(* IEC 61131-3 sources: volt/packages/volt-lsp-iec/test-corpus/pro2193/Device/Plc Logic/Application/04 Physical Interfaces/Ethernet/13 Dashboard, 2 files *)

(* ---- PlcDataType.dut ---- *)
// Complete list of PlcDataTypes for all machines
{attribute 'qualified_only'}
TYPE PlcDataType :
(
	// Last changed (UTC): 17 Dec 2025 13:19
	// Total number of PlcDataTypes: 3778

	Main_RobotStatus := 23,
	Main_EnableIML := 24,
	Main_EnableHMU := 25,
	Main_EnableVision := 26,
	Main_Relays_HighVacuumPumpRunning := 27,
	Main_Relays_LowVacuumPumpRunning := 28,
	Relays_MouldAreaFree := 29,
	Relays_EnableMouldClosure := 30,
	Relays_EnableFullMouldOpening := 31,
	Relays_OperationWithRobot := 32,
	Relays_EnableEjectorBack := 33,
	Relays_EnableEjectorForward := 34,
	Relays_EnableCorePos1Back := 35,
	Relays_EnableCorePos2Forward := 36,
	Relays_GlobalReset := 37,
	Relays_MainAirValve := 38,
	Relays_YUnit_MotorCooling := 39,
	Relays_EnableFrequencyController := 40,
	Relays_SafetyGate := 41,
	YUnit_ActPos := 42,
	YUnit_ErrorId := 43,
	YUnit_AxisErrorId := 44,
	YUnit_DriveErrorId := 45,
	YUnit_DriveUtilisation := 46,
	YUnit_MotorUtilisation := 47,
	XrUnit_ActPos := 48,
	XrUnit_ErrorId := 49,
	XrUnit_AxisErrorId := 50,
	XrUnit_DriveErrorId := 51,
	XrUnit_DriveUtilisation := 52,
	XrUnit_MotorUtilisation := 53,
	XiUnit_ActPos := 54,
	XiUnit_ErrorId := 55,
	XiUnit_AxisErrorId := 56,
	XiUnit_DriveErrorId := 57,
	XiUnit_DriveUtilisation := 58,
	XiUnit_MotorUtilisation := 59,
	XuUnit_ActPos := 60,
	XuUnit_ErrorId := 61,
	XuUnit_AxisErrorId := 62,
	XuUnit_DriveErrorId := 63,
	XuUnit_DriveUtilisation := 64,
	XuUnit_MotorUtilisation := 65,
	Chain_ActPos := 66,
	Chain_ErrorId := 67,
	Chain_AxisErrorId := 68,
	Chain_DriveErrorId := 69,
	Chain_DriveUtilisation := 70,
	Chain_MotorUtilisation := 71,
	Magazine_M1_1_ActPos := 72,
	Magazine_M1_1_ErrorId := 73,
	Magazine_M1_1_AxisErrorId := 74,
	Magazine_M1_1_DriveErrorId := 75,
	Magazine_M1_1_DriveUtilisation := 76,
	Magazine_M1_1_MotorUtilisation := 77,
	Magazine_M1_2_ActPos := 78,
	Magazine_M1_2_ErrorId := 79,
	Magazine_M1_2_AxisErrorId := 80,
	Magazine_M1_2_DriveErrorId := 81,
	Magazine_M1_2_DriveUtilisation := 82,
	Magazine_M1_2_MotorUtilisation := 83,
	ZUnit_ActPos := 84,
	ZUnit_ErrorId := 85,
	ZUnit_AxisErrorId := 86,
	ZUnit_DriveErrorId := 87,
	ZUnit_DriveUtilisation := 88,
	ZUnit_MotorUtilisation := 89,
	YUnit_ActTorque := 90,
	XrUnit_ActTorque := 91,
	XiUnit_ActTorque := 92,
	XuUnit_ActTorque := 93,
	Chain_ActTorque := 94,
	Magazine_M1_1_ActTorque := 95,
	Magazine_M1_2_ActTorque := 96,
	ZUnit_ActTorque := 97,
	YUnit_CoveredDistance := 98,
	XrUnit_CoveredDistance := 99,
	XiUnit_CoveredDistance := 100,
	XuUnit_CoveredDistance := 101,
	Chain_CoveredDistance := 102,
	Magazine_M1_1_CoveredDistance := 103,
	Magazine_M1_2_CoveredDistance := 104,
	ZUnit_CoveredDistance := 105,
	CycleTimes_TimeStopped := 106,
	CycleTimes_TimeResetting := 107,
	CycleTimes_TimeIdle := 108,
	CycleTimes_TimeAutomatic := 109,
	CycleTimes_AutomaticCycleStarts := 110,
	YUnit_Alarms := 111,
	YUnit_Time_Active := 112,
	YUnit_Time_Idle := 113,
	XrUnit_Alarms := 114,
	XrUnit_Time_Active := 115,
	XrUnit_Time_Idle := 116,
	XiUnit_Alarms := 117,
	XiUnit_Time_Active := 118,
	XiUnit_Time_Idle := 119,
	XuUnit_Alarms := 120,
	XuUnit_Time_Active := 121,
	XuUnit_Time_Idle := 122,
	Chain_Alarms := 123,
	Chain_Time_Active := 124,
	Chain_Time_Idle := 125,
	Magazine_M1_1_Alarms := 126,
	Magazine_M1_1_Time_Active := 127,
	Magazine_M1_1_Time_Idle := 128,
	Magazine_M1_2_Alarms := 129,
	Magazine_M1_2_Time_Active := 130,
	Magazine_M1_2_Time_Idle := 131,
	ZUnit_Alarms := 132,
	ZUnit_Time_Active := 133,
	ZUnit_Time_Idle := 134,
	Camera_Alarms := 135,
	Camera_Time_Active := 136,
	Camera_Time_Idle := 137,
	RejectStation_Alarms := 138,
	RejectStation_Time_Active := 139,
	RejectStation_Time_Idle := 140,
	Conveyors_Alarms := 141,
	Conveyors_Time_Active := 142,
	Conveyors_Time_Idle := 143,
	IMM_CycleTimeTakeout := 144,
	IMM_CycleTimeTotal := 145,
	IMM_SavedCycleTimeByEarlyMouldClosing := 146,
	XuUnit_SensorTimes_Vacuum_1 := 147,
	XuUnit_SensorTimes_Vacuum_2 := 148,
	XuUnit_SensorTimes_Vacuum_3 := 149,
	XuUnit_SensorTimes_ShiftIn := 150,
	XuUnit_SensorTimes_ShiftOut := 151,
	Magazine_SensorTimes_Vacuum_1 := 152,
	Magazine_SensorTimes_Vacuum_2 := 153,
	Magazine_SensorTimes_Vacuum_3 := 154,
	Magazine_SensorTimes_Vacuum_4 := 155,
	Magazine_SensorTimes_FlipLabel1In := 156,
	Magazine_SensorTimes_FlipLabel1Out := 157,
	Magazine_SensorTimes_FlipLabel2In := 158,
	Magazine_SensorTimes_FlipLabel2Out := 159,
	Magazine_SensorTimes_ChangeDrawerIn := 160,
	Magazine_SensorTimes_ChangeDrawerOut := 161,
	Magazine_SensorTimes_LockDrawerIn := 162,
	Magazine_SensorTimes_LockDrawerOut := 163,
	ZUnit_SensorTimes_Vacuum_1 := 164,
	ZUnit_SensorTimes_Vacuum_2 := 165,
	ZUnit_SensorTimes_Vacuum_3 := 166,
	ZUnit_SensorTimes_Vacuum_4 := 167,
	ZUnit_SensorTimes_RotateIn := 168,
	ZUnit_SensorTimes_RotateOut := 169,
	ZUnit_SensorTimes_Extend1In := 170,
	ZUnit_SensorTimes_Extend2In := 171,
	ZUnit_SensorTimes_Extend3In := 172,
	ZUnit_SensorTimes_Extend4In := 173,
	RejectStation_SensorTimes_RejectCylinderIn := 174,
	RejectStation_SensorTimes_RejectCylinderOut := 175,
	MetaData_RejectReason_0_Description := 176,
	MetaData_RejectReason_1_Description := 177,
	MetaData_RejectReason_2_Description := 178,
	MetaData_RejectReason_3_Description := 179,
	MetaData_RejectReason_4_Description := 180,
	MetaData_RejectReason_5_Description := 181,
	MetaData_RejectReason_6_Description := 182,
	Productioncounters_Total_Produced := 183,
	Productioncounters_Total_Stacked := 184,
	Productioncounters_Total_Rejected := 185,
	Productioncounters_Total_UncountedReject := 186,
	Productioncounters_Total_RejectReason_0 := 187,
	Productioncounters_Total_RejectReason_1 := 188,
	Productioncounters_Total_RejectReason_2 := 189,
	Productioncounters_Total_RejectReason_3 := 190,
	Productioncounters_Total_RejectReason_4 := 191,
	Productioncounters_Total_RejectReason_5 := 192,
	Productioncounters_Total_RejectReason_6 := 193,
	Productioncounters_Cavity_1_Produced := 194,
	Productioncounters_Cavity_1_Stacked := 195,
	Productioncounters_Cavity_1_Rejected := 196,
	Productioncounters_Cavity_1_UncountedReject := 197,
	Productioncounters_Cavity_1_RejectReason_0 := 198,
	Productioncounters_Cavity_1_RejectReason_1 := 199,
	Productioncounters_Cavity_1_RejectReason_2 := 200,
	Productioncounters_Cavity_1_RejectReason_3 := 201,
	Productioncounters_Cavity_1_RejectReason_4 := 202,
	Productioncounters_Cavity_1_RejectReason_5 := 203,
	Productioncounters_Cavity_1_RejectReason_6 := 204,
	Productioncounters_Cavity_2_Produced := 205,
	Productioncounters_Cavity_2_Stacked := 206,
	Productioncounters_Cavity_2_Rejected := 207,
	Productioncounters_Cavity_2_UncountedReject := 208,
	Productioncounters_Cavity_2_RejectReason_0 := 209,
	Productioncounters_Cavity_2_RejectReason_1 := 210,
	Productioncounters_Cavity_2_RejectReason_2 := 211,
	Productioncounters_Cavity_2_RejectReason_3 := 212,
	Productioncounters_Cavity_2_RejectReason_4 := 213,
	Productioncounters_Cavity_2_RejectReason_5 := 214,
	Productioncounters_Cavity_2_RejectReason_6 := 215,
	Productioncounters_Cavity_3_Produced := 216,
	Productioncounters_Cavity_3_Stacked := 217,
	Productioncounters_Cavity_3_Rejected := 218,
	Productioncounters_Cavity_3_UncountedReject := 219,
	Productioncounters_Cavity_3_RejectReason_0 := 220,
	Productioncounters_Cavity_3_RejectReason_1 := 221,
	Productioncounters_Cavity_3_RejectReason_2 := 222,
	Productioncounters_Cavity_3_RejectReason_3 := 223,
	Productioncounters_Cavity_3_RejectReason_4 := 224,
	Productioncounters_Cavity_3_RejectReason_5 := 225,
	Productioncounters_Cavity_3_RejectReason_6 := 226,
	Productioncounters_Cavity_4_Produced := 227,
	Productioncounters_Cavity_4_Stacked := 228,
	Productioncounters_Cavity_4_Rejected := 229,
	Productioncounters_Cavity_4_UncountedReject := 230,
	Productioncounters_Cavity_4_RejectReason_0 := 231,
	Productioncounters_Cavity_4_RejectReason_1 := 232,
	Productioncounters_Cavity_4_RejectReason_2 := 233,
	Productioncounters_Cavity_4_RejectReason_3 := 234,
	Productioncounters_Cavity_4_RejectReason_4 := 235,
	Productioncounters_Cavity_4_RejectReason_5 := 236,
	Productioncounters_Cavity_4_RejectReason_6 := 237,
	Productioncounters_Cavity_5_Produced := 238,
	Productioncounters_Cavity_5_Stacked := 239,
	Productioncounters_Cavity_5_Rejected := 240,
	Productioncounters_Cavity_5_UncountedReject := 241,
	Productioncounters_Cavity_5_RejectReason_0 := 242,
	Productioncounters_Cavity_5_RejectReason_1 := 243,
	Productioncounters_Cavity_5_RejectReason_2 := 244,
	Productioncounters_Cavity_5_RejectReason_3 := 245,
	Productioncounters_Cavity_5_RejectReason_4 := 246,
	Productioncounters_Cavity_5_RejectReason_5 := 247,
	Productioncounters_Cavity_5_RejectReason_6 := 248,
	Productioncounters_Cavity_6_Produced := 249,
	Productioncounters_Cavity_6_Stacked := 250,
	Productioncounters_Cavity_6_Rejected := 251,
	Productioncounters_Cavity_6_UncountedReject := 252,
	Productioncounters_Cavity_6_RejectReason_0 := 253,
	Productioncounters_Cavity_6_RejectReason_1 := 254,
	Productioncounters_Cavity_6_RejectReason_2 := 255,
	Productioncounters_Cavity_6_RejectReason_3 := 256,
	Productioncounters_Cavity_6_RejectReason_4 := 257,
	Productioncounters_Cavity_6_RejectReason_5 := 258,
	Productioncounters_Cavity_6_RejectReason_6 := 259,
	Main_RecipeName := 260,
	Main_RecipeName_Cassette := 261,
	Main_ParameterChanged := 262,
	Main_AirPressureOk := 263,
	Main_GeneralAlarmActive := 264,
	Main_GeneralWarningActive := 265,
	Main_Alarms := 266,
	Main_AlarmsFuse := 267,
	Main_AlarmsIMM := 268,
	Main_Messages := 269,
	Main_Warnings := 270,
	Magazine_Alarms := 273,
	YUnit_AlarmsMotionControl := 274,
	Main_SafetyPLCStatus1 := 275,
	Main_SafetyPLCStatus2 := 276,
	Main_SafetyPLCStatus3 := 277,
	RobotConnected := 278,
	ZUnit_SensorTimes_Shift1In := 279,
	ZUnit_SensorTimes_Shift1Out := 280,
	Main_SER_State := 281,
	Main_SER_OperationMode := 282,
	Main_RecipeName_Brink := 283,
	RejectStation_SensorTimes_RejectCylinder2In := 284,
	RejectStation_SensorTimes_RejectCylinder2Out := 285,
	XuUnit_SensorTimes_ShiftHorizontalIn := 286,
	XuUnit_SensorTimes_ShiftHorizontalOut := 287,
	XuUnit_SensorTimes_ShiftVerticalIn := 288,
	XuUnit_SensorTimes_ShiftVerticalOut := 289,
	MetaData_RejectReason_7_Description := 290,
	Productioncounters_Total_RejectReason_7 := 291,
	Productioncounters_Cavity_1_RejectReason_7 := 292,
	Productioncounters_Cavity_2_RejectReason_7 := 293,
	Productioncounters_Cavity_3_RejectReason_7 := 294,
	Productioncounters_Cavity_4_RejectReason_7 := 295,
	Productioncounters_Cavity_5_RejectReason_7 := 296,
	Productioncounters_Cavity_6_RejectReason_7 := 297,
	MouldMeasurement_MaxPressure := 298,
	MouldMeasurement_MinPressure := 299,
	MouldMeasurement_IdealPressure := 300,
	MouldMeasurement_AveragePressure := 301,
	MouldMeasurement_CalculatedIdealPressure := 302,
	MouldMeasurement_HoldingPressure_TargetValue := 303,
	MouldMeasurement_HoldingPressure_ActualValue := 304,
	MouldMeasurement_SwitchOverPoint_TargetValue := 305,
	MouldMeasurement_SwitchOverPoint_ActualValue := 306,
	MouldMeasurement_Cavity_1_PeakPressure := 307,
	MouldMeasurement_Cavity_2_PeakPressure := 308,
	MouldMeasurement_Cavity_3_PeakPressure := 309,
	MouldMeasurement_Cavity_4_PeakPressure := 310,
	MouldMeasurement_Cavity_5_PeakPressure := 311,
	MouldMeasurement_Cavity_6_PeakPressure := 312,
	MouldMeasurement_Hotrunner_Cavity_1_TargetValue := 313,
	MouldMeasurement_Hotrunner_Cavity_1_ActualValue := 314,
	MouldMeasurement_Hotrunner_Cavity_2_TargetValue := 315,
	MouldMeasurement_Hotrunner_Cavity_2_ActualValue := 316,
	MouldMeasurement_Hotrunner_Cavity_3_TargetValue := 317,
	MouldMeasurement_Hotrunner_Cavity_3_ActualValue := 318,
	MouldMeasurement_Hotrunner_Cavity_4_TargetValue := 319,
	MouldMeasurement_Hotrunner_Cavity_4_ActualValue := 320,
	MouldMeasurement_Hotrunner_Cavity_5_TargetValue := 321,
	MouldMeasurement_Hotrunner_Cavity_5_ActualValue := 322,
	MouldMeasurement_Hotrunner_Cavity_6_TargetValue := 323,
	MouldMeasurement_Hotrunner_Cavity_6_ActualValue := 324,
	MetaData_RejectReason_8_Description := 325,
	Productioncounters_Total_RejectReason_8 := 326,
	Productioncounters_Cavity_1_RejectReason_8 := 327,
	Productioncounters_Cavity_2_RejectReason_8 := 328,
	Productioncounters_Cavity_3_RejectReason_8 := 329,
	Productioncounters_Cavity_4_RejectReason_8 := 330,
	Productioncounters_Cavity_5_RejectReason_8 := 331,
	Productioncounters_Cavity_6_RejectReason_8 := 332,
	MetaData_RejectReason_9_Description := 333,
	Productioncounters_Total_RejectReason_9 := 334,
	Productioncounters_Cavity_1_RejectReason_9 := 335,
	Productioncounters_Cavity_2_RejectReason_9 := 336,
	Productioncounters_Cavity_3_RejectReason_9 := 337,
	Productioncounters_Cavity_4_RejectReason_9 := 338,
	Productioncounters_Cavity_5_RejectReason_9 := 339,
	Productioncounters_Cavity_6_RejectReason_9 := 340,
	MetaData_RejectReason_10_Description := 341,
	Productioncounters_Total_RejectReason_10 := 342,
	Productioncounters_Cavity_1_RejectReason_10 := 343,
	Productioncounters_Cavity_2_RejectReason_10 := 344,
	Productioncounters_Cavity_3_RejectReason_10 := 345,
	Productioncounters_Cavity_4_RejectReason_10 := 346,
	Productioncounters_Cavity_5_RejectReason_10 := 347,
	Productioncounters_Cavity_6_RejectReason_10 := 348,
	MetaData_RejectReason_11_Description := 349,
	Productioncounters_Total_RejectReason_11 := 350,
	Productioncounters_Cavity_1_RejectReason_11 := 351,
	Productioncounters_Cavity_2_RejectReason_11 := 352,
	Productioncounters_Cavity_3_RejectReason_11 := 353,
	Productioncounters_Cavity_4_RejectReason_11 := 354,
	Productioncounters_Cavity_5_RejectReason_11 := 355,
	Productioncounters_Cavity_6_RejectReason_11 := 356,
	MetaData_RejectReason_12_Description := 357,
	Productioncounters_Total_RejectReason_12 := 358,
	Productioncounters_Cavity_1_RejectReason_12 := 359,
	Productioncounters_Cavity_2_RejectReason_12 := 360,
	Productioncounters_Cavity_3_RejectReason_12 := 361,
	Productioncounters_Cavity_4_RejectReason_12 := 362,
	Productioncounters_Cavity_5_RejectReason_12 := 363,
	Productioncounters_Cavity_6_RejectReason_12 := 364,
	MetaData_RejectReason_13_Description := 365,
	Productioncounters_Total_RejectReason_13 := 366,
	Productioncounters_Cavity_1_RejectReason_13 := 367,
	Productioncounters_Cavity_2_RejectReason_13 := 368,
	Productioncounters_Cavity_3_RejectReason_13 := 369,
	Productioncounters_Cavity_4_RejectReason_13 := 370,
	Productioncounters_Cavity_5_RejectReason_13 := 371,
	Productioncounters_Cavity_6_RejectReason_13 := 372,
	MetaData_RejectReason_14_Description := 373,
	Productioncounters_Total_RejectReason_14 := 374,
	Productioncounters_Cavity_1_RejectReason_14 := 375,
	Productioncounters_Cavity_2_RejectReason_14 := 376,
	Productioncounters_Cavity_3_RejectReason_14 := 377,
	Productioncounters_Cavity_4_RejectReason_14 := 378,
	Productioncounters_Cavity_5_RejectReason_14 := 379,
	Productioncounters_Cavity_6_RejectReason_14 := 380,
	MetaData_RejectReason_15_Description := 381,
	Productioncounters_Total_RejectReason_15 := 382,
	Productioncounters_Cavity_1_RejectReason_15 := 383,
	Productioncounters_Cavity_2_RejectReason_15 := 384,
	Productioncounters_Cavity_3_RejectReason_15 := 385,
	Productioncounters_Cavity_4_RejectReason_15 := 386,
	Productioncounters_Cavity_5_RejectReason_15 := 387,
	Productioncounters_Cavity_6_RejectReason_15 := 388,
	MetaData_RejectReason_16_Description := 389,
	Productioncounters_Total_RejectReason_16 := 390,
	Productioncounters_Cavity_1_RejectReason_16 := 391,
	Productioncounters_Cavity_2_RejectReason_16 := 392,
	Productioncounters_Cavity_3_RejectReason_16 := 393,
	Productioncounters_Cavity_4_RejectReason_16 := 394,
	Productioncounters_Cavity_5_RejectReason_16 := 395,
	Productioncounters_Cavity_6_RejectReason_16 := 396,
	MetaData_RejectReason_17_Description := 397,
	Productioncounters_Total_RejectReason_17 := 398,
	Productioncounters_Cavity_1_RejectReason_17 := 399,
	Productioncounters_Cavity_2_RejectReason_17 := 400,
	Productioncounters_Cavity_3_RejectReason_17 := 401,
	Productioncounters_Cavity_4_RejectReason_17 := 402,
	Productioncounters_Cavity_5_RejectReason_17 := 403,
	Productioncounters_Cavity_6_RejectReason_17 := 404,
	MetaData_RejectReason_18_Description := 405,
	Productioncounters_Total_RejectReason_18 := 406,
	Productioncounters_Cavity_1_RejectReason_18 := 407,
	Productioncounters_Cavity_2_RejectReason_18 := 408,
	Productioncounters_Cavity_3_RejectReason_18 := 409,
	Productioncounters_Cavity_4_RejectReason_18 := 410,
	Productioncounters_Cavity_5_RejectReason_18 := 411,
	Productioncounters_Cavity_6_RejectReason_18 := 412,
	MetaData_RejectReason_19_Description := 413,
	Productioncounters_Total_RejectReason_19 := 414,
	Productioncounters_Cavity_1_RejectReason_19 := 415,
	Productioncounters_Cavity_2_RejectReason_19 := 416,
	Productioncounters_Cavity_3_RejectReason_19 := 417,
	Productioncounters_Cavity_4_RejectReason_19 := 418,
	Productioncounters_Cavity_5_RejectReason_19 := 419,
	Productioncounters_Cavity_6_RejectReason_19 := 420,
	MetaData_RejectReason_20_Description := 421,
	Productioncounters_Total_RejectReason_20 := 422,
	Productioncounters_Cavity_1_RejectReason_20 := 423,
	Productioncounters_Cavity_2_RejectReason_20 := 424,
	Productioncounters_Cavity_3_RejectReason_20 := 425,
	Productioncounters_Cavity_4_RejectReason_20 := 426,
	Productioncounters_Cavity_5_RejectReason_20 := 427,
	Productioncounters_Cavity_6_RejectReason_20 := 428,
	Productioncounters_Cavity_7_Produced := 429,
	Productioncounters_Cavity_7_Stacked := 430,
	Productioncounters_Cavity_7_Rejected := 431,
	Productioncounters_Cavity_7_UncountedReject := 432,
	Productioncounters_Cavity_7_RejectReason_0 := 433,
	Productioncounters_Cavity_7_RejectReason_1 := 434,
	Productioncounters_Cavity_7_RejectReason_2 := 435,
	Productioncounters_Cavity_7_RejectReason_3 := 436,
	Productioncounters_Cavity_7_RejectReason_4 := 437,
	Productioncounters_Cavity_7_RejectReason_5 := 438,
	Productioncounters_Cavity_7_RejectReason_6 := 439,
	Productioncounters_Cavity_7_RejectReason_7 := 440,
	Productioncounters_Cavity_7_RejectReason_8 := 441,
	Productioncounters_Cavity_7_RejectReason_9 := 442,
	Productioncounters_Cavity_7_RejectReason_10 := 443,
	Productioncounters_Cavity_7_RejectReason_11 := 444,
	Productioncounters_Cavity_7_RejectReason_12 := 445,
	Productioncounters_Cavity_7_RejectReason_13 := 446,
	Productioncounters_Cavity_7_RejectReason_14 := 447,
	Productioncounters_Cavity_7_RejectReason_15 := 448,
	Productioncounters_Cavity_7_RejectReason_16 := 449,
	Productioncounters_Cavity_7_RejectReason_17 := 450,
	Productioncounters_Cavity_7_RejectReason_18 := 451,
	Productioncounters_Cavity_7_RejectReason_19 := 452,
	Productioncounters_Cavity_7_RejectReason_20 := 453,
	MouldMeasurement_Cavity_7_PeakPressure := 454,
	MouldMeasurement_Hotrunner_Cavity_7_TargetValue := 455,
	MouldMeasurement_Hotrunner_Cavity_7_ActualValue := 456,
	Productioncounters_Cavity_8_Produced := 457,
	Productioncounters_Cavity_8_Stacked := 458,
	Productioncounters_Cavity_8_Rejected := 459,
	Productioncounters_Cavity_8_UncountedReject := 460,
	Productioncounters_Cavity_8_RejectReason_0 := 461,
	Productioncounters_Cavity_8_RejectReason_1 := 462,
	Productioncounters_Cavity_8_RejectReason_2 := 463,
	Productioncounters_Cavity_8_RejectReason_3 := 464,
	Productioncounters_Cavity_8_RejectReason_4 := 465,
	Productioncounters_Cavity_8_RejectReason_5 := 466,
	Productioncounters_Cavity_8_RejectReason_6 := 467,
	Productioncounters_Cavity_8_RejectReason_7 := 468,
	Productioncounters_Cavity_8_RejectReason_8 := 469,
	Productioncounters_Cavity_8_RejectReason_9 := 470,
	Productioncounters_Cavity_8_RejectReason_10 := 471,
	Productioncounters_Cavity_8_RejectReason_11 := 472,
	Productioncounters_Cavity_8_RejectReason_12 := 473,
	Productioncounters_Cavity_8_RejectReason_13 := 474,
	Productioncounters_Cavity_8_RejectReason_14 := 475,
	Productioncounters_Cavity_8_RejectReason_15 := 476,
	Productioncounters_Cavity_8_RejectReason_16 := 477,
	Productioncounters_Cavity_8_RejectReason_17 := 478,
	Productioncounters_Cavity_8_RejectReason_18 := 479,
	Productioncounters_Cavity_8_RejectReason_19 := 480,
	Productioncounters_Cavity_8_RejectReason_20 := 481,
	MouldMeasurement_Cavity_8_PeakPressure := 482,
	MouldMeasurement_Hotrunner_Cavity_8_TargetValue := 483,
	MouldMeasurement_Hotrunner_Cavity_8_ActualValue := 484,
	Productioncounters_Cavity_9_Produced := 485,
	Productioncounters_Cavity_9_Stacked := 486,
	Productioncounters_Cavity_9_Rejected := 487,
	Productioncounters_Cavity_9_UncountedReject := 488,
	Productioncounters_Cavity_9_RejectReason_0 := 489,
	Productioncounters_Cavity_9_RejectReason_1 := 490,
	Productioncounters_Cavity_9_RejectReason_2 := 491,
	Productioncounters_Cavity_9_RejectReason_3 := 492,
	Productioncounters_Cavity_9_RejectReason_4 := 493,
	Productioncounters_Cavity_9_RejectReason_5 := 494,
	Productioncounters_Cavity_9_RejectReason_6 := 495,
	Productioncounters_Cavity_9_RejectReason_7 := 496,
	Productioncounters_Cavity_9_RejectReason_8 := 497,
	Productioncounters_Cavity_9_RejectReason_9 := 498,
	Productioncounters_Cavity_9_RejectReason_10 := 499,
	Productioncounters_Cavity_9_RejectReason_11 := 500,
	Productioncounters_Cavity_9_RejectReason_12 := 501,
	Productioncounters_Cavity_9_RejectReason_13 := 502,
	Productioncounters_Cavity_9_RejectReason_14 := 503,
	Productioncounters_Cavity_9_RejectReason_15 := 504,
	Productioncounters_Cavity_9_RejectReason_16 := 505,
	Productioncounters_Cavity_9_RejectReason_17 := 506,
	Productioncounters_Cavity_9_RejectReason_18 := 507,
	Productioncounters_Cavity_9_RejectReason_19 := 508,
	Productioncounters_Cavity_9_RejectReason_20 := 509,
	MouldMeasurement_Cavity_9_PeakPressure := 510,
	MouldMeasurement_Hotrunner_Cavity_9_TargetValue := 511,
	MouldMeasurement_Hotrunner_Cavity_9_ActualValue := 512,
	Productioncounters_Cavity_10_Produced := 513,
	Productioncounters_Cavity_10_Stacked := 514,
	Productioncounters_Cavity_10_Rejected := 515,
	Productioncounters_Cavity_10_UncountedReject := 516,
	Productioncounters_Cavity_10_RejectReason_0 := 517,
	Productioncounters_Cavity_10_RejectReason_1 := 518,
	Productioncounters_Cavity_10_RejectReason_2 := 519,
	Productioncounters_Cavity_10_RejectReason_3 := 520,
	Productioncounters_Cavity_10_RejectReason_4 := 521,
	Productioncounters_Cavity_10_RejectReason_5 := 522,
	Productioncounters_Cavity_10_RejectReason_6 := 523,
	Productioncounters_Cavity_10_RejectReason_7 := 524,
	Productioncounters_Cavity_10_RejectReason_8 := 525,
	Productioncounters_Cavity_10_RejectReason_9 := 526,
	Productioncounters_Cavity_10_RejectReason_10 := 527,
	Productioncounters_Cavity_10_RejectReason_11 := 528,
	Productioncounters_Cavity_10_RejectReason_12 := 529,
	Productioncounters_Cavity_10_RejectReason_13 := 530,
	Productioncounters_Cavity_10_RejectReason_14 := 531,
	Productioncounters_Cavity_10_RejectReason_15 := 532,
	Productioncounters_Cavity_10_RejectReason_16 := 533,
	Productioncounters_Cavity_10_RejectReason_17 := 534,
	Productioncounters_Cavity_10_RejectReason_18 := 535,
	Productioncounters_Cavity_10_RejectReason_19 := 536,
	Productioncounters_Cavity_10_RejectReason_20 := 537,
	MouldMeasurement_Cavity_10_PeakPressure := 538,
	MouldMeasurement_Hotrunner_Cavity_10_TargetValue := 539,
	MouldMeasurement_Hotrunner_Cavity_10_ActualValue := 540,
	Productioncounters_Cavity_11_Produced := 541,
	Productioncounters_Cavity_11_Stacked := 542,
	Productioncounters_Cavity_11_Rejected := 543,
	Productioncounters_Cavity_11_UncountedReject := 544,
	Productioncounters_Cavity_11_RejectReason_0 := 545,
	Productioncounters_Cavity_11_RejectReason_1 := 546,
	Productioncounters_Cavity_11_RejectReason_2 := 547,
	Productioncounters_Cavity_11_RejectReason_3 := 548,
	Productioncounters_Cavity_11_RejectReason_4 := 549,
	Productioncounters_Cavity_11_RejectReason_5 := 550,
	Productioncounters_Cavity_11_RejectReason_6 := 551,
	Productioncounters_Cavity_11_RejectReason_7 := 552,
	Productioncounters_Cavity_11_RejectReason_8 := 553,
	Productioncounters_Cavity_11_RejectReason_9 := 554,
	Productioncounters_Cavity_11_RejectReason_10 := 555,
	Productioncounters_Cavity_11_RejectReason_11 := 556,
	Productioncounters_Cavity_11_RejectReason_12 := 557,
	Productioncounters_Cavity_11_RejectReason_13 := 558,
	Productioncounters_Cavity_11_RejectReason_14 := 559,
	Productioncounters_Cavity_11_RejectReason_15 := 560,
	Productioncounters_Cavity_11_RejectReason_16 := 561,
	Productioncounters_Cavity_11_RejectReason_17 := 562,
	Productioncounters_Cavity_11_RejectReason_18 := 563,
	Productioncounters_Cavity_11_RejectReason_19 := 564,
	Productioncounters_Cavity_11_RejectReason_20 := 565,
	MouldMeasurement_Cavity_11_PeakPressure := 566,
	MouldMeasurement_Hotrunner_Cavity_11_TargetValue := 567,
	MouldMeasurement_Hotrunner_Cavity_11_ActualValue := 568,
	Productioncounters_Cavity_12_Produced := 569,
	Productioncounters_Cavity_12_Stacked := 570,
	Productioncounters_Cavity_12_Rejected := 571,
	Productioncounters_Cavity_12_UncountedReject := 572,
	Productioncounters_Cavity_12_RejectReason_0 := 573,
	Productioncounters_Cavity_12_RejectReason_1 := 574,
	Productioncounters_Cavity_12_RejectReason_2 := 575,
	Productioncounters_Cavity_12_RejectReason_3 := 576,
	Productioncounters_Cavity_12_RejectReason_4 := 577,
	Productioncounters_Cavity_12_RejectReason_5 := 578,
	Productioncounters_Cavity_12_RejectReason_6 := 579,
	Productioncounters_Cavity_12_RejectReason_7 := 580,
	Productioncounters_Cavity_12_RejectReason_8 := 581,
	Productioncounters_Cavity_12_RejectReason_9 := 582,
	Productioncounters_Cavity_12_RejectReason_10 := 583,
	Productioncounters_Cavity_12_RejectReason_11 := 584,
	Productioncounters_Cavity_12_RejectReason_12 := 585,
	Productioncounters_Cavity_12_RejectReason_13 := 586,
	Productioncounters_Cavity_12_RejectReason_14 := 587,
	Productioncounters_Cavity_12_RejectReason_15 := 588,
	Productioncounters_Cavity_12_RejectReason_16 := 589,
	Productioncounters_Cavity_12_RejectReason_17 := 590,
	Productioncounters_Cavity_12_RejectReason_18 := 591,
	Productioncounters_Cavity_12_RejectReason_19 := 592,
	Productioncounters_Cavity_12_RejectReason_20 := 593,
	MouldMeasurement_Cavity_12_PeakPressure := 594,
	MouldMeasurement_Hotrunner_Cavity_12_TargetValue := 595,
	MouldMeasurement_Hotrunner_Cavity_12_ActualValue := 596,
	Productioncounters_Cavity_13_Produced := 597,
	Productioncounters_Cavity_13_Stacked := 598,
	Productioncounters_Cavity_13_Rejected := 599,
	Productioncounters_Cavity_13_UncountedReject := 600,
	Productioncounters_Cavity_13_RejectReason_0 := 601,
	Productioncounters_Cavity_13_RejectReason_1 := 602,
	Productioncounters_Cavity_13_RejectReason_2 := 603,
	Productioncounters_Cavity_13_RejectReason_3 := 604,
	Productioncounters_Cavity_13_RejectReason_4 := 605,
	Productioncounters_Cavity_13_RejectReason_5 := 606,
	Productioncounters_Cavity_13_RejectReason_6 := 607,
	Productioncounters_Cavity_13_RejectReason_7 := 608,
	Productioncounters_Cavity_13_RejectReason_8 := 609,
	Productioncounters_Cavity_13_RejectReason_9 := 610,
	Productioncounters_Cavity_13_RejectReason_10 := 611,
	Productioncounters_Cavity_13_RejectReason_11 := 612,
	Productioncounters_Cavity_13_RejectReason_12 := 613,
	Productioncounters_Cavity_13_RejectReason_13 := 614,
	Productioncounters_Cavity_13_RejectReason_14 := 615,
	Productioncounters_Cavity_13_RejectReason_15 := 616,
	Productioncounters_Cavity_13_RejectReason_16 := 617,
	Productioncounters_Cavity_13_RejectReason_17 := 618,
	Productioncounters_Cavity_13_RejectReason_18 := 619,
	Productioncounters_Cavity_13_RejectReason_19 := 620,
	Productioncounters_Cavity_13_RejectReason_20 := 621,
	MouldMeasurement_Cavity_13_PeakPressure := 622,
	MouldMeasurement_Hotrunner_Cavity_13_TargetValue := 623,
	MouldMeasurement_Hotrunner_Cavity_13_ActualValue := 624,
	Productioncounters_Cavity_14_Produced := 625,
	Productioncounters_Cavity_14_Stacked := 626,
	Productioncounters_Cavity_14_Rejected := 627,
	Productioncounters_Cavity_14_UncountedReject := 628,
	Productioncounters_Cavity_14_RejectReason_0 := 629,
	Productioncounters_Cavity_14_RejectReason_1 := 630,
	Productioncounters_Cavity_14_RejectReason_2 := 631,
	Productioncounters_Cavity_14_RejectReason_3 := 632,
	Productioncounters_Cavity_14_RejectReason_4 := 633,
	Productioncounters_Cavity_14_RejectReason_5 := 634,
	Productioncounters_Cavity_14_RejectReason_6 := 635,
	Productioncounters_Cavity_14_RejectReason_7 := 636,
	Productioncounters_Cavity_14_RejectReason_8 := 637,
	Productioncounters_Cavity_14_RejectReason_9 := 638,
	Productioncounters_Cavity_14_RejectReason_10 := 639,
	Productioncounters_Cavity_14_RejectReason_11 := 640,
	Productioncounters_Cavity_14_RejectReason_12 := 641,
	Productioncounters_Cavity_14_RejectReason_13 := 642,
	Productioncounters_Cavity_14_RejectReason_14 := 643,
	Productioncounters_Cavity_14_RejectReason_15 := 644,
	Productioncounters_Cavity_14_RejectReason_16 := 645,
	Productioncounters_Cavity_14_RejectReason_17 := 646,
	Productioncounters_Cavity_14_RejectReason_18 := 647,
	Productioncounters_Cavity_14_RejectReason_19 := 648,
	Productioncounters_Cavity_14_RejectReason_20 := 649,
	MouldMeasurement_Cavity_14_PeakPressure := 650,
	MouldMeasurement_Hotrunner_Cavity_14_TargetValue := 651,
	MouldMeasurement_Hotrunner_Cavity_14_ActualValue := 652,
	Productioncounters_Cavity_15_Produced := 653,
	Productioncounters_Cavity_15_Stacked := 654,
	Productioncounters_Cavity_15_Rejected := 655,
	Productioncounters_Cavity_15_UncountedReject := 656,
	Productioncounters_Cavity_15_RejectReason_0 := 657,
	Productioncounters_Cavity_15_RejectReason_1 := 658,
	Productioncounters_Cavity_15_RejectReason_2 := 659,
	Productioncounters_Cavity_15_RejectReason_3 := 660,
	Productioncounters_Cavity_15_RejectReason_4 := 661,
	Productioncounters_Cavity_15_RejectReason_5 := 662,
	Productioncounters_Cavity_15_RejectReason_6 := 663,
	Productioncounters_Cavity_15_RejectReason_7 := 664,
	Productioncounters_Cavity_15_RejectReason_8 := 665,
	Productioncounters_Cavity_15_RejectReason_9 := 666,
	Productioncounters_Cavity_15_RejectReason_10 := 667,
	Productioncounters_Cavity_15_RejectReason_11 := 668,
	Productioncounters_Cavity_15_RejectReason_12 := 669,
	Productioncounters_Cavity_15_RejectReason_13 := 670,
	Productioncounters_Cavity_15_RejectReason_14 := 671,
	Productioncounters_Cavity_15_RejectReason_15 := 672,
	Productioncounters_Cavity_15_RejectReason_16 := 673,
	Productioncounters_Cavity_15_RejectReason_17 := 674,
	Productioncounters_Cavity_15_RejectReason_18 := 675,
	Productioncounters_Cavity_15_RejectReason_19 := 676,
	Productioncounters_Cavity_15_RejectReason_20 := 677,
	MouldMeasurement_Cavity_15_PeakPressure := 678,
	MouldMeasurement_Hotrunner_Cavity_15_TargetValue := 679,
	MouldMeasurement_Hotrunner_Cavity_15_ActualValue := 680,
	Productioncounters_Cavity_16_Produced := 681,
	Productioncounters_Cavity_16_Stacked := 682,
	Productioncounters_Cavity_16_Rejected := 683,
	Productioncounters_Cavity_16_UncountedReject := 684,
	Productioncounters_Cavity_16_RejectReason_0 := 685,
	Productioncounters_Cavity_16_RejectReason_1 := 686,
	Productioncounters_Cavity_16_RejectReason_2 := 687,
	Productioncounters_Cavity_16_RejectReason_3 := 688,
	Productioncounters_Cavity_16_RejectReason_4 := 689,
	Productioncounters_Cavity_16_RejectReason_5 := 690,
	Productioncounters_Cavity_16_RejectReason_6 := 691,
	Productioncounters_Cavity_16_RejectReason_7 := 692,
	Productioncounters_Cavity_16_RejectReason_8 := 693,
	Productioncounters_Cavity_16_RejectReason_9 := 694,
	Productioncounters_Cavity_16_RejectReason_10 := 695,
	Productioncounters_Cavity_16_RejectReason_11 := 696,
	Productioncounters_Cavity_16_RejectReason_12 := 697,
	Productioncounters_Cavity_16_RejectReason_13 := 698,
	Productioncounters_Cavity_16_RejectReason_14 := 699,
	Productioncounters_Cavity_16_RejectReason_15 := 700,
	Productioncounters_Cavity_16_RejectReason_16 := 701,
	Productioncounters_Cavity_16_RejectReason_17 := 702,
	Productioncounters_Cavity_16_RejectReason_18 := 703,
	Productioncounters_Cavity_16_RejectReason_19 := 704,
	Productioncounters_Cavity_16_RejectReason_20 := 705,
	MouldMeasurement_Cavity_16_PeakPressure := 706,
	MouldMeasurement_Hotrunner_Cavity_16_TargetValue := 707,
	MouldMeasurement_Hotrunner_Cavity_16_ActualValue := 708,
	Productioncounters_Cavity_17_Produced := 709,
	Productioncounters_Cavity_17_Stacked := 710,
	Productioncounters_Cavity_17_Rejected := 711,
	Productioncounters_Cavity_17_UncountedReject := 712,
	Productioncounters_Cavity_17_RejectReason_0 := 713,
	Productioncounters_Cavity_17_RejectReason_1 := 714,
	Productioncounters_Cavity_17_RejectReason_2 := 715,
	Productioncounters_Cavity_17_RejectReason_3 := 716,
	Productioncounters_Cavity_17_RejectReason_4 := 717,
	Productioncounters_Cavity_17_RejectReason_5 := 718,
	Productioncounters_Cavity_17_RejectReason_6 := 719,
	Productioncounters_Cavity_17_RejectReason_7 := 720,
	Productioncounters_Cavity_17_RejectReason_8 := 721,
	Productioncounters_Cavity_17_RejectReason_9 := 722,
	Productioncounters_Cavity_17_RejectReason_10 := 723,
	Productioncounters_Cavity_17_RejectReason_11 := 724,
	Productioncounters_Cavity_17_RejectReason_12 := 725,
	Productioncounters_Cavity_17_RejectReason_13 := 726,
	Productioncounters_Cavity_17_RejectReason_14 := 727,
	Productioncounters_Cavity_17_RejectReason_15 := 728,
	Productioncounters_Cavity_17_RejectReason_16 := 729,
	Productioncounters_Cavity_17_RejectReason_17 := 730,
	Productioncounters_Cavity_17_RejectReason_18 := 731,
	Productioncounters_Cavity_17_RejectReason_19 := 732,
	Productioncounters_Cavity_17_RejectReason_20 := 733,
	MouldMeasurement_Cavity_17_PeakPressure := 734,
	MouldMeasurement_Hotrunner_Cavity_17_TargetValue := 735,
	MouldMeasurement_Hotrunner_Cavity_17_ActualValue := 736,
	Productioncounters_Cavity_18_Produced := 737,
	Productioncounters_Cavity_18_Stacked := 738,
	Productioncounters_Cavity_18_Rejected := 739,
	Productioncounters_Cavity_18_UncountedReject := 740,
	Productioncounters_Cavity_18_RejectReason_0 := 741,
	Productioncounters_Cavity_18_RejectReason_1 := 742,
	Productioncounters_Cavity_18_RejectReason_2 := 743,
	Productioncounters_Cavity_18_RejectReason_3 := 744,
	Productioncounters_Cavity_18_RejectReason_4 := 745,
	Productioncounters_Cavity_18_RejectReason_5 := 746,
	Productioncounters_Cavity_18_RejectReason_6 := 747,
	Productioncounters_Cavity_18_RejectReason_7 := 748,
	Productioncounters_Cavity_18_RejectReason_8 := 749,
	Productioncounters_Cavity_18_RejectReason_9 := 750,
	Productioncounters_Cavity_18_RejectReason_10 := 751,
	Productioncounters_Cavity_18_RejectReason_11 := 752,
	Productioncounters_Cavity_18_RejectReason_12 := 753,
	Productioncounters_Cavity_18_RejectReason_13 := 754,
	Productioncounters_Cavity_18_RejectReason_14 := 755,
	Productioncounters_Cavity_18_RejectReason_15 := 756,
	Productioncounters_Cavity_18_RejectReason_16 := 757,
	Productioncounters_Cavity_18_RejectReason_17 := 758,
	Productioncounters_Cavity_18_RejectReason_18 := 759,
	Productioncounters_Cavity_18_RejectReason_19 := 760,
	Productioncounters_Cavity_18_RejectReason_20 := 761,
	MouldMeasurement_Cavity_18_PeakPressure := 762,
	MouldMeasurement_Hotrunner_Cavity_18_TargetValue := 763,
	MouldMeasurement_Hotrunner_Cavity_18_ActualValue := 764,
	Productioncounters_Cavity_19_Produced := 765,
	Productioncounters_Cavity_19_Stacked := 766,
	Productioncounters_Cavity_19_Rejected := 767,
	Productioncounters_Cavity_19_UncountedReject := 768,
	Productioncounters_Cavity_19_RejectReason_0 := 769,
	Productioncounters_Cavity_19_RejectReason_1 := 770,
	Productioncounters_Cavity_19_RejectReason_2 := 771,
	Productioncounters_Cavity_19_RejectReason_3 := 772,
	Productioncounters_Cavity_19_RejectReason_4 := 773,
	Productioncounters_Cavity_19_RejectReason_5 := 774,
	Productioncounters_Cavity_19_RejectReason_6 := 775,
	Productioncounters_Cavity_19_RejectReason_7 := 776,
	Productioncounters_Cavity_19_RejectReason_8 := 777,
	Productioncounters_Cavity_19_RejectReason_9 := 778,
	Productioncounters_Cavity_19_RejectReason_10 := 779,
	Productioncounters_Cavity_19_RejectReason_11 := 780,
	Productioncounters_Cavity_19_RejectReason_12 := 781,
	Productioncounters_Cavity_19_RejectReason_13 := 782,
	Productioncounters_Cavity_19_RejectReason_14 := 783,
	Productioncounters_Cavity_19_RejectReason_15 := 784,
	Productioncounters_Cavity_19_RejectReason_16 := 785,
	Productioncounters_Cavity_19_RejectReason_17 := 786,
	Productioncounters_Cavity_19_RejectReason_18 := 787,
	Productioncounters_Cavity_19_RejectReason_19 := 788,
	Productioncounters_Cavity_19_RejectReason_20 := 789,
	MouldMeasurement_Cavity_19_PeakPressure := 790,
	MouldMeasurement_Hotrunner_Cavity_19_TargetValue := 791,
	MouldMeasurement_Hotrunner_Cavity_19_ActualValue := 792,
	Productioncounters_Cavity_20_Produced := 793,
	Productioncounters_Cavity_20_Stacked := 794,
	Productioncounters_Cavity_20_Rejected := 795,
	Productioncounters_Cavity_20_UncountedReject := 796,
	Productioncounters_Cavity_20_RejectReason_0 := 797,
	Productioncounters_Cavity_20_RejectReason_1 := 798,
	Productioncounters_Cavity_20_RejectReason_2 := 799,
	Productioncounters_Cavity_20_RejectReason_3 := 800,
	Productioncounters_Cavity_20_RejectReason_4 := 801,
	Productioncounters_Cavity_20_RejectReason_5 := 802,
	Productioncounters_Cavity_20_RejectReason_6 := 803,
	Productioncounters_Cavity_20_RejectReason_7 := 804,
	Productioncounters_Cavity_20_RejectReason_8 := 805,
	Productioncounters_Cavity_20_RejectReason_9 := 806,
	Productioncounters_Cavity_20_RejectReason_10 := 807,
	Productioncounters_Cavity_20_RejectReason_11 := 808,
	Productioncounters_Cavity_20_RejectReason_12 := 809,
	Productioncounters_Cavity_20_RejectReason_13 := 810,
	Productioncounters_Cavity_20_RejectReason_14 := 811,
	Productioncounters_Cavity_20_RejectReason_15 := 812,
	Productioncounters_Cavity_20_RejectReason_16 := 813,
	Productioncounters_Cavity_20_RejectReason_17 := 814,
	Productioncounters_Cavity_20_RejectReason_18 := 815,
	Productioncounters_Cavity_20_RejectReason_19 := 816,
	Productioncounters_Cavity_20_RejectReason_20 := 817,
	MouldMeasurement_Cavity_20_PeakPressure := 818,
	MouldMeasurement_Hotrunner_Cavity_20_TargetValue := 819,
	MouldMeasurement_Hotrunner_Cavity_20_ActualValue := 820,
	Productioncounters_Cavity_21_Produced := 821,
	Productioncounters_Cavity_21_Stacked := 822,
	Productioncounters_Cavity_21_Rejected := 823,
	Productioncounters_Cavity_21_UncountedReject := 824,
	Productioncounters_Cavity_21_RejectReason_0 := 825,
	Productioncounters_Cavity_21_RejectReason_1 := 826,
	Productioncounters_Cavity_21_RejectReason_2 := 827,
	Productioncounters_Cavity_21_RejectReason_3 := 828,
	Productioncounters_Cavity_21_RejectReason_4 := 829,
	Productioncounters_Cavity_21_RejectReason_5 := 830,
	Productioncounters_Cavity_21_RejectReason_6 := 831,
	Productioncounters_Cavity_21_RejectReason_7 := 832,
	Productioncounters_Cavity_21_RejectReason_8 := 833,
	Productioncounters_Cavity_21_RejectReason_9 := 834,
	Productioncounters_Cavity_21_RejectReason_10 := 835,
	Productioncounters_Cavity_21_RejectReason_11 := 836,
	Productioncounters_Cavity_21_RejectReason_12 := 837,
	Productioncounters_Cavity_21_RejectReason_13 := 838,
	Productioncounters_Cavity_21_RejectReason_14 := 839,
	Productioncounters_Cavity_21_RejectReason_15 := 840,
	Productioncounters_Cavity_21_RejectReason_16 := 841,
	Productioncounters_Cavity_21_RejectReason_17 := 842,
	Productioncounters_Cavity_21_RejectReason_18 := 843,
	Productioncounters_Cavity_21_RejectReason_19 := 844,
	Productioncounters_Cavity_21_RejectReason_20 := 845,
	MouldMeasurement_Cavity_21_PeakPressure := 846,
	MouldMeasurement_Hotrunner_Cavity_21_TargetValue := 847,
	MouldMeasurement_Hotrunner_Cavity_21_ActualValue := 848,
	Productioncounters_Cavity_22_Produced := 849,
	Productioncounters_Cavity_22_Stacked := 850,
	Productioncounters_Cavity_22_Rejected := 851,
	Productioncounters_Cavity_22_UncountedReject := 852,
	Productioncounters_Cavity_22_RejectReason_0 := 853,
	Productioncounters_Cavity_22_RejectReason_1 := 854,
	Productioncounters_Cavity_22_RejectReason_2 := 855,
	Productioncounters_Cavity_22_RejectReason_3 := 856,
	Productioncounters_Cavity_22_RejectReason_4 := 857,
	Productioncounters_Cavity_22_RejectReason_5 := 858,
	Productioncounters_Cavity_22_RejectReason_6 := 859,
	Productioncounters_Cavity_22_RejectReason_7 := 860,
	Productioncounters_Cavity_22_RejectReason_8 := 861,
	Productioncounters_Cavity_22_RejectReason_9 := 862,
	Productioncounters_Cavity_22_RejectReason_10 := 863,
	Productioncounters_Cavity_22_RejectReason_11 := 864,
	Productioncounters_Cavity_22_RejectReason_12 := 865,
	Productioncounters_Cavity_22_RejectReason_13 := 866,
	Productioncounters_Cavity_22_RejectReason_14 := 867,
	Productioncounters_Cavity_22_RejectReason_15 := 868,
	Productioncounters_Cavity_22_RejectReason_16 := 869,
	Productioncounters_Cavity_22_RejectReason_17 := 870,
	Productioncounters_Cavity_22_RejectReason_18 := 871,
	Productioncounters_Cavity_22_RejectReason_19 := 872,
	Productioncounters_Cavity_22_RejectReason_20 := 873,
	MouldMeasurement_Cavity_22_PeakPressure := 874,
	MouldMeasurement_Hotrunner_Cavity_22_TargetValue := 875,
	MouldMeasurement_Hotrunner_Cavity_22_ActualValue := 876,
	Productioncounters_Cavity_23_Produced := 877,
	Productioncounters_Cavity_23_Stacked := 878,
	Productioncounters_Cavity_23_Rejected := 879,
	Productioncounters_Cavity_23_UncountedReject := 880,
	Productioncounters_Cavity_23_RejectReason_0 := 881,
	Productioncounters_Cavity_23_RejectReason_1 := 882,
	Productioncounters_Cavity_23_RejectReason_2 := 883,
	Productioncounters_Cavity_23_RejectReason_3 := 884,
	Productioncounters_Cavity_23_RejectReason_4 := 885,
	Productioncounters_Cavity_23_RejectReason_5 := 886,
	Productioncounters_Cavity_23_RejectReason_6 := 887,
	Productioncounters_Cavity_23_RejectReason_7 := 888,
	Productioncounters_Cavity_23_RejectReason_8 := 889,
	Productioncounters_Cavity_23_RejectReason_9 := 890,
	Productioncounters_Cavity_23_RejectReason_10 := 891,
	Productioncounters_Cavity_23_RejectReason_11 := 892,
	Productioncounters_Cavity_23_RejectReason_12 := 893,
	Productioncounters_Cavity_23_RejectReason_13 := 894,
	Productioncounters_Cavity_23_RejectReason_14 := 895,
	Productioncounters_Cavity_23_RejectReason_15 := 896,
	Productioncounters_Cavity_23_RejectReason_16 := 897,
	Productioncounters_Cavity_23_RejectReason_17 := 898,
	Productioncounters_Cavity_23_RejectReason_18 := 899,
	Productioncounters_Cavity_23_RejectReason_19 := 900,
	Productioncounters_Cavity_23_RejectReason_20 := 901,
	MouldMeasurement_Cavity_23_PeakPressure := 902,
	MouldMeasurement_Hotrunner_Cavity_23_TargetValue := 903,
	MouldMeasurement_Hotrunner_Cavity_23_ActualValue := 904,
	Productioncounters_Cavity_24_Produced := 905,
	Productioncounters_Cavity_24_Stacked := 906,
	Productioncounters_Cavity_24_Rejected := 907,
	Productioncounters_Cavity_24_UncountedReject := 908,
	Productioncounters_Cavity_24_RejectReason_0 := 909,
	Productioncounters_Cavity_24_RejectReason_1 := 910,
	Productioncounters_Cavity_24_RejectReason_2 := 911,
	Productioncounters_Cavity_24_RejectReason_3 := 912,
	Productioncounters_Cavity_24_RejectReason_4 := 913,
	Productioncounters_Cavity_24_RejectReason_5 := 914,
	Productioncounters_Cavity_24_RejectReason_6 := 915,
	Productioncounters_Cavity_24_RejectReason_7 := 916,
	Productioncounters_Cavity_24_RejectReason_8 := 917,
	Productioncounters_Cavity_24_RejectReason_9 := 918,
	Productioncounters_Cavity_24_RejectReason_10 := 919,
	Productioncounters_Cavity_24_RejectReason_11 := 920,
	Productioncounters_Cavity_24_RejectReason_12 := 921,
	Productioncounters_Cavity_24_RejectReason_13 := 922,
	Productioncounters_Cavity_24_RejectReason_14 := 923,
	Productioncounters_Cavity_24_RejectReason_15 := 924,
	Productioncounters_Cavity_24_RejectReason_16 := 925,
	Productioncounters_Cavity_24_RejectReason_17 := 926,
	Productioncounters_Cavity_24_RejectReason_18 := 927,
	Productioncounters_Cavity_24_RejectReason_19 := 928,
	Productioncounters_Cavity_24_RejectReason_20 := 929,
	MouldMeasurement_Cavity_24_PeakPressure := 930,
	MouldMeasurement_Hotrunner_Cavity_24_TargetValue := 931,
	MouldMeasurement_Hotrunner_Cavity_24_ActualValue := 932,
	Productioncounters_Cavity_25_Produced := 933,
	Productioncounters_Cavity_25_Stacked := 934,
	Productioncounters_Cavity_25_Rejected := 935,
	Productioncounters_Cavity_25_UncountedReject := 936,
	Productioncounters_Cavity_25_RejectReason_0 := 937,
	Productioncounters_Cavity_25_RejectReason_1 := 938,
	Productioncounters_Cavity_25_RejectReason_2 := 939,
	Productioncounters_Cavity_25_RejectReason_3 := 940,
	Productioncounters_Cavity_25_RejectReason_4 := 941,
	Productioncounters_Cavity_25_RejectReason_5 := 942,
	Productioncounters_Cavity_25_RejectReason_6 := 943,
	Productioncounters_Cavity_25_RejectReason_7 := 944,
	Productioncounters_Cavity_25_RejectReason_8 := 945,
	Productioncounters_Cavity_25_RejectReason_9 := 946,
	Productioncounters_Cavity_25_RejectReason_10 := 947,
	Productioncounters_Cavity_25_RejectReason_11 := 948,
	Productioncounters_Cavity_25_RejectReason_12 := 949,
	Productioncounters_Cavity_25_RejectReason_13 := 950,
	Productioncounters_Cavity_25_RejectReason_14 := 951,
	Productioncounters_Cavity_25_RejectReason_15 := 952,
	Productioncounters_Cavity_25_RejectReason_16 := 953,
	Productioncounters_Cavity_25_RejectReason_17 := 954,
	Productioncounters_Cavity_25_RejectReason_18 := 955,
	Productioncounters_Cavity_25_RejectReason_19 := 956,
	Productioncounters_Cavity_25_RejectReason_20 := 957,
	MouldMeasurement_Cavity_25_PeakPressure := 958,
	MouldMeasurement_Hotrunner_Cavity_25_TargetValue := 959,
	MouldMeasurement_Hotrunner_Cavity_25_ActualValue := 960,
	Productioncounters_Cavity_26_Produced := 961,
	Productioncounters_Cavity_26_Stacked := 962,
	Productioncounters_Cavity_26_Rejected := 963,
	Productioncounters_Cavity_26_UncountedReject := 964,
	Productioncounters_Cavity_26_RejectReason_0 := 965,
	Productioncounters_Cavity_26_RejectReason_1 := 966,
	Productioncounters_Cavity_26_RejectReason_2 := 967,
	Productioncounters_Cavity_26_RejectReason_3 := 968,
	Productioncounters_Cavity_26_RejectReason_4 := 969,
	Productioncounters_Cavity_26_RejectReason_5 := 970,
	Productioncounters_Cavity_26_RejectReason_6 := 971,
	Productioncounters_Cavity_26_RejectReason_7 := 972,
	Productioncounters_Cavity_26_RejectReason_8 := 973,
	Productioncounters_Cavity_26_RejectReason_9 := 974,
	Productioncounters_Cavity_26_RejectReason_10 := 975,
	Productioncounters_Cavity_26_RejectReason_11 := 976,
	Productioncounters_Cavity_26_RejectReason_12 := 977,
	Productioncounters_Cavity_26_RejectReason_13 := 978,
	Productioncounters_Cavity_26_RejectReason_14 := 979,
	Productioncounters_Cavity_26_RejectReason_15 := 980,
	Productioncounters_Cavity_26_RejectReason_16 := 981,
	Productioncounters_Cavity_26_RejectReason_17 := 982,
	Productioncounters_Cavity_26_RejectReason_18 := 983,
	Productioncounters_Cavity_26_RejectReason_19 := 984,
	Productioncounters_Cavity_26_RejectReason_20 := 985,
	MouldMeasurement_Cavity_26_PeakPressure := 986,
	MouldMeasurement_Hotrunner_Cavity_26_TargetValue := 987,
	MouldMeasurement_Hotrunner_Cavity_26_ActualValue := 988,
	Productioncounters_Cavity_27_Produced := 989,
	Productioncounters_Cavity_27_Stacked := 990,
	Productioncounters_Cavity_27_Rejected := 991,
	Productioncounters_Cavity_27_UncountedReject := 992,
	Productioncounters_Cavity_27_RejectReason_0 := 993,
	Productioncounters_Cavity_27_RejectReason_1 := 994,
	Productioncounters_Cavity_27_RejectReason_2 := 995,
	Productioncounters_Cavity_27_RejectReason_3 := 996,
	Productioncounters_Cavity_27_RejectReason_4 := 997,
	Productioncounters_Cavity_27_RejectReason_5 := 998,
	Productioncounters_Cavity_27_RejectReason_6 := 999,
	Productioncounters_Cavity_27_RejectReason_7 := 1000,
	Productioncounters_Cavity_27_RejectReason_8 := 1001,
	Productioncounters_Cavity_27_RejectReason_9 := 1002,
	Productioncounters_Cavity_27_RejectReason_10 := 1003,
	Productioncounters_Cavity_27_RejectReason_11 := 1004,
	Productioncounters_Cavity_27_RejectReason_12 := 1005,
	Productioncounters_Cavity_27_RejectReason_13 := 1006,
	Productioncounters_Cavity_27_RejectReason_14 := 1007,
	Productioncounters_Cavity_27_RejectReason_15 := 1008,
	Productioncounters_Cavity_27_RejectReason_16 := 1009,
	Productioncounters_Cavity_27_RejectReason_17 := 1010,
	Productioncounters_Cavity_27_RejectReason_18 := 1011,
	Productioncounters_Cavity_27_RejectReason_19 := 1012,
	Productioncounters_Cavity_27_RejectReason_20 := 1013,
	MouldMeasurement_Cavity_27_PeakPressure := 1014,
	MouldMeasurement_Hotrunner_Cavity_27_TargetValue := 1015,
	MouldMeasurement_Hotrunner_Cavity_27_ActualValue := 1016,
	Productioncounters_Cavity_28_Produced := 1017,
	Productioncounters_Cavity_28_Stacked := 1018,
	Productioncounters_Cavity_28_Rejected := 1019,
	Productioncounters_Cavity_28_UncountedReject := 1020,
	Productioncounters_Cavity_28_RejectReason_0 := 1021,
	Productioncounters_Cavity_28_RejectReason_1 := 1022,
	Productioncounters_Cavity_28_RejectReason_2 := 1023,
	Productioncounters_Cavity_28_RejectReason_3 := 1024,
	Productioncounters_Cavity_28_RejectReason_4 := 1025,
	Productioncounters_Cavity_28_RejectReason_5 := 1026,
	Productioncounters_Cavity_28_RejectReason_6 := 1027,
	Productioncounters_Cavity_28_RejectReason_7 := 1028,
	Productioncounters_Cavity_28_RejectReason_8 := 1029,
	Productioncounters_Cavity_28_RejectReason_9 := 1030,
	Productioncounters_Cavity_28_RejectReason_10 := 1031,
	Productioncounters_Cavity_28_RejectReason_11 := 1032,
	Productioncounters_Cavity_28_RejectReason_12 := 1033,
	Productioncounters_Cavity_28_RejectReason_13 := 1034,
	Productioncounters_Cavity_28_RejectReason_14 := 1035,
	Productioncounters_Cavity_28_RejectReason_15 := 1036,
	Productioncounters_Cavity_28_RejectReason_16 := 1037,
	Productioncounters_Cavity_28_RejectReason_17 := 1038,
	Productioncounters_Cavity_28_RejectReason_18 := 1039,
	Productioncounters_Cavity_28_RejectReason_19 := 1040,
	Productioncounters_Cavity_28_RejectReason_20 := 1041,
	MouldMeasurement_Cavity_28_PeakPressure := 1042,
	MouldMeasurement_Hotrunner_Cavity_28_TargetValue := 1043,
	MouldMeasurement_Hotrunner_Cavity_28_ActualValue := 1044,
	Productioncounters_Cavity_29_Produced := 1045,
	Productioncounters_Cavity_29_Stacked := 1046,
	Productioncounters_Cavity_29_Rejected := 1047,
	Productioncounters_Cavity_29_UncountedReject := 1048,
	Productioncounters_Cavity_29_RejectReason_0 := 1049,
	Productioncounters_Cavity_29_RejectReason_1 := 1050,
	Productioncounters_Cavity_29_RejectReason_2 := 1051,
	Productioncounters_Cavity_29_RejectReason_3 := 1052,
	Productioncounters_Cavity_29_RejectReason_4 := 1053,
	Productioncounters_Cavity_29_RejectReason_5 := 1054,
	Productioncounters_Cavity_29_RejectReason_6 := 1055,
	Productioncounters_Cavity_29_RejectReason_7 := 1056,
	Productioncounters_Cavity_29_RejectReason_8 := 1057,
	Productioncounters_Cavity_29_RejectReason_9 := 1058,
	Productioncounters_Cavity_29_RejectReason_10 := 1059,
	Productioncounters_Cavity_29_RejectReason_11 := 1060,
	Productioncounters_Cavity_29_RejectReason_12 := 1061,
	Productioncounters_Cavity_29_RejectReason_13 := 1062,
	Productioncounters_Cavity_29_RejectReason_14 := 1063,
	Productioncounters_Cavity_29_RejectReason_15 := 1064,
	Productioncounters_Cavity_29_RejectReason_16 := 1065,
	Productioncounters_Cavity_29_RejectReason_17 := 1066,
	Productioncounters_Cavity_29_RejectReason_18 := 1067,
	Productioncounters_Cavity_29_RejectReason_19 := 1068,
	Productioncounters_Cavity_29_RejectReason_20 := 1069,
	MouldMeasurement_Cavity_29_PeakPressure := 1070,
	MouldMeasurement_Hotrunner_Cavity_29_TargetValue := 1071,
	MouldMeasurement_Hotrunner_Cavity_29_ActualValue := 1072,
	Productioncounters_Cavity_30_Produced := 1073,
	Productioncounters_Cavity_30_Stacked := 1074,
	Productioncounters_Cavity_30_Rejected := 1075,
	Productioncounters_Cavity_30_UncountedReject := 1076,
	Productioncounters_Cavity_30_RejectReason_0 := 1077,
	Productioncounters_Cavity_30_RejectReason_1 := 1078,
	Productioncounters_Cavity_30_RejectReason_2 := 1079,
	Productioncounters_Cavity_30_RejectReason_3 := 1080,
	Productioncounters_Cavity_30_RejectReason_4 := 1081,
	Productioncounters_Cavity_30_RejectReason_5 := 1082,
	Productioncounters_Cavity_30_RejectReason_6 := 1083,
	Productioncounters_Cavity_30_RejectReason_7 := 1084,
	Productioncounters_Cavity_30_RejectReason_8 := 1085,
	Productioncounters_Cavity_30_RejectReason_9 := 1086,
	Productioncounters_Cavity_30_RejectReason_10 := 1087,
	Productioncounters_Cavity_30_RejectReason_11 := 1088,
	Productioncounters_Cavity_30_RejectReason_12 := 1089,
	Productioncounters_Cavity_30_RejectReason_13 := 1090,
	Productioncounters_Cavity_30_RejectReason_14 := 1091,
	Productioncounters_Cavity_30_RejectReason_15 := 1092,
	Productioncounters_Cavity_30_RejectReason_16 := 1093,
	Productioncounters_Cavity_30_RejectReason_17 := 1094,
	Productioncounters_Cavity_30_RejectReason_18 := 1095,
	Productioncounters_Cavity_30_RejectReason_19 := 1096,
	Productioncounters_Cavity_30_RejectReason_20 := 1097,
	MouldMeasurement_Cavity_30_PeakPressure := 1098,
	MouldMeasurement_Hotrunner_Cavity_30_TargetValue := 1099,
	MouldMeasurement_Hotrunner_Cavity_30_ActualValue := 1100,
	Productioncounters_Cavity_31_Produced := 1101,
	Productioncounters_Cavity_31_Stacked := 1102,
	Productioncounters_Cavity_31_Rejected := 1103,
	Productioncounters_Cavity_31_UncountedReject := 1104,
	Productioncounters_Cavity_31_RejectReason_0 := 1105,
	Productioncounters_Cavity_31_RejectReason_1 := 1106,
	Productioncounters_Cavity_31_RejectReason_2 := 1107,
	Productioncounters_Cavity_31_RejectReason_3 := 1108,
	Productioncounters_Cavity_31_RejectReason_4 := 1109,
	Productioncounters_Cavity_31_RejectReason_5 := 1110,
	Productioncounters_Cavity_31_RejectReason_6 := 1111,
	Productioncounters_Cavity_31_RejectReason_7 := 1112,
	Productioncounters_Cavity_31_RejectReason_8 := 1113,
	Productioncounters_Cavity_31_RejectReason_9 := 1114,
	Productioncounters_Cavity_31_RejectReason_10 := 1115,
	Productioncounters_Cavity_31_RejectReason_11 := 1116,
	Productioncounters_Cavity_31_RejectReason_12 := 1117,
	Productioncounters_Cavity_31_RejectReason_13 := 1118,
	Productioncounters_Cavity_31_RejectReason_14 := 1119,
	Productioncounters_Cavity_31_RejectReason_15 := 1120,
	Productioncounters_Cavity_31_RejectReason_16 := 1121,
	Productioncounters_Cavity_31_RejectReason_17 := 1122,
	Productioncounters_Cavity_31_RejectReason_18 := 1123,
	Productioncounters_Cavity_31_RejectReason_19 := 1124,
	Productioncounters_Cavity_31_RejectReason_20 := 1125,
	MouldMeasurement_Cavity_31_PeakPressure := 1126,
	MouldMeasurement_Hotrunner_Cavity_31_TargetValue := 1127,
	MouldMeasurement_Hotrunner_Cavity_31_ActualValue := 1128,
	Productioncounters_Cavity_32_Produced := 1129,
	Productioncounters_Cavity_32_Stacked := 1130,
	Productioncounters_Cavity_32_Rejected := 1131,
	Productioncounters_Cavity_32_UncountedReject := 1132,
	Productioncounters_Cavity_32_RejectReason_0 := 1133,
	Productioncounters_Cavity_32_RejectReason_1 := 1134,
	Productioncounters_Cavity_32_RejectReason_2 := 1135,
	Productioncounters_Cavity_32_RejectReason_3 := 1136,
	Productioncounters_Cavity_32_RejectReason_4 := 1137,
	Productioncounters_Cavity_32_RejectReason_5 := 1138,
	Productioncounters_Cavity_32_RejectReason_6 := 1139,
	Productioncounters_Cavity_32_RejectReason_7 := 1140,
	Productioncounters_Cavity_32_RejectReason_8 := 1141,
	Productioncounters_Cavity_32_RejectReason_9 := 1142,
	Productioncounters_Cavity_32_RejectReason_10 := 1143,
	Productioncounters_Cavity_32_RejectReason_11 := 1144,
	Productioncounters_Cavity_32_RejectReason_12 := 1145,
	Productioncounters_Cavity_32_RejectReason_13 := 1146,
	Productioncounters_Cavity_32_RejectReason_14 := 1147,
	Productioncounters_Cavity_32_RejectReason_15 := 1148,
	Productioncounters_Cavity_32_RejectReason_16 := 1149,
	Productioncounters_Cavity_32_RejectReason_17 := 1150,
	Productioncounters_Cavity_32_RejectReason_18 := 1151,
	Productioncounters_Cavity_32_RejectReason_19 := 1152,
	Productioncounters_Cavity_32_RejectReason_20 := 1153,
	MouldMeasurement_Cavity_32_PeakPressure := 1154,
	MouldMeasurement_Hotrunner_Cavity_32_TargetValue := 1155,
	MouldMeasurement_Hotrunner_Cavity_32_ActualValue := 1156,
	Productioncounters_Cavity_33_Produced := 1157,
	Productioncounters_Cavity_33_Stacked := 1158,
	Productioncounters_Cavity_33_Rejected := 1159,
	Productioncounters_Cavity_33_UncountedReject := 1160,
	Productioncounters_Cavity_33_RejectReason_0 := 1161,
	Productioncounters_Cavity_33_RejectReason_1 := 1162,
	Productioncounters_Cavity_33_RejectReason_2 := 1163,
	Productioncounters_Cavity_33_RejectReason_3 := 1164,
	Productioncounters_Cavity_33_RejectReason_4 := 1165,
	Productioncounters_Cavity_33_RejectReason_5 := 1166,
	Productioncounters_Cavity_33_RejectReason_6 := 1167,
	Productioncounters_Cavity_33_RejectReason_7 := 1168,
	Productioncounters_Cavity_33_RejectReason_8 := 1169,
	Productioncounters_Cavity_33_RejectReason_9 := 1170,
	Productioncounters_Cavity_33_RejectReason_10 := 1171,
	Productioncounters_Cavity_33_RejectReason_11 := 1172,
	Productioncounters_Cavity_33_RejectReason_12 := 1173,
	Productioncounters_Cavity_33_RejectReason_13 := 1174,
	Productioncounters_Cavity_33_RejectReason_14 := 1175,
	Productioncounters_Cavity_33_RejectReason_15 := 1176,
	Productioncounters_Cavity_33_RejectReason_16 := 1177,
	Productioncounters_Cavity_33_RejectReason_17 := 1178,
	Productioncounters_Cavity_33_RejectReason_18 := 1179,
	Productioncounters_Cavity_33_RejectReason_19 := 1180,
	Productioncounters_Cavity_33_RejectReason_20 := 1181,
	MouldMeasurement_Cavity_33_PeakPressure := 1182,
	MouldMeasurement_Hotrunner_Cavity_33_TargetValue := 1183,
	MouldMeasurement_Hotrunner_Cavity_33_ActualValue := 1184,
	Productioncounters_Cavity_34_Produced := 1185,
	Productioncounters_Cavity_34_Stacked := 1186,
	Productioncounters_Cavity_34_Rejected := 1187,
	Productioncounters_Cavity_34_UncountedReject := 1188,
	Productioncounters_Cavity_34_RejectReason_0 := 1189,
	Productioncounters_Cavity_34_RejectReason_1 := 1190,
	Productioncounters_Cavity_34_RejectReason_2 := 1191,
	Productioncounters_Cavity_34_RejectReason_3 := 1192,
	Productioncounters_Cavity_34_RejectReason_4 := 1193,
	Productioncounters_Cavity_34_RejectReason_5 := 1194,
	Productioncounters_Cavity_34_RejectReason_6 := 1195,
	Productioncounters_Cavity_34_RejectReason_7 := 1196,
	Productioncounters_Cavity_34_RejectReason_8 := 1197,
	Productioncounters_Cavity_34_RejectReason_9 := 1198,
	Productioncounters_Cavity_34_RejectReason_10 := 1199,
	Productioncounters_Cavity_34_RejectReason_11 := 1200,
	Productioncounters_Cavity_34_RejectReason_12 := 1201,
	Productioncounters_Cavity_34_RejectReason_13 := 1202,
	Productioncounters_Cavity_34_RejectReason_14 := 1203,
	Productioncounters_Cavity_34_RejectReason_15 := 1204,
	Productioncounters_Cavity_34_RejectReason_16 := 1205,
	Productioncounters_Cavity_34_RejectReason_17 := 1206,
	Productioncounters_Cavity_34_RejectReason_18 := 1207,
	Productioncounters_Cavity_34_RejectReason_19 := 1208,
	Productioncounters_Cavity_34_RejectReason_20 := 1209,
	MouldMeasurement_Cavity_34_PeakPressure := 1210,
	MouldMeasurement_Hotrunner_Cavity_34_TargetValue := 1211,
	MouldMeasurement_Hotrunner_Cavity_34_ActualValue := 1212,
	Productioncounters_Cavity_35_Produced := 1213,
	Productioncounters_Cavity_35_Stacked := 1214,
	Productioncounters_Cavity_35_Rejected := 1215,
	Productioncounters_Cavity_35_UncountedReject := 1216,
	Productioncounters_Cavity_35_RejectReason_0 := 1217,
	Productioncounters_Cavity_35_RejectReason_1 := 1218,
	Productioncounters_Cavity_35_RejectReason_2 := 1219,
	Productioncounters_Cavity_35_RejectReason_3 := 1220,
	Productioncounters_Cavity_35_RejectReason_4 := 1221,
	Productioncounters_Cavity_35_RejectReason_5 := 1222,
	Productioncounters_Cavity_35_RejectReason_6 := 1223,
	Productioncounters_Cavity_35_RejectReason_7 := 1224,
	Productioncounters_Cavity_35_RejectReason_8 := 1225,
	Productioncounters_Cavity_35_RejectReason_9 := 1226,
	Productioncounters_Cavity_35_RejectReason_10 := 1227,
	Productioncounters_Cavity_35_RejectReason_11 := 1228,
	Productioncounters_Cavity_35_RejectReason_12 := 1229,
	Productioncounters_Cavity_35_RejectReason_13 := 1230,
	Productioncounters_Cavity_35_RejectReason_14 := 1231,
	Productioncounters_Cavity_35_RejectReason_15 := 1232,
	Productioncounters_Cavity_35_RejectReason_16 := 1233,
	Productioncounters_Cavity_35_RejectReason_17 := 1234,
	Productioncounters_Cavity_35_RejectReason_18 := 1235,
	Productioncounters_Cavity_35_RejectReason_19 := 1236,
	Productioncounters_Cavity_35_RejectReason_20 := 1237,
	MouldMeasurement_Cavity_35_PeakPressure := 1238,
	MouldMeasurement_Hotrunner_Cavity_35_TargetValue := 1239,
	MouldMeasurement_Hotrunner_Cavity_35_ActualValue := 1240,
	Productioncounters_Cavity_36_Produced := 1241,
	Productioncounters_Cavity_36_Stacked := 1242,
	Productioncounters_Cavity_36_Rejected := 1243,
	Productioncounters_Cavity_36_UncountedReject := 1244,
	Productioncounters_Cavity_36_RejectReason_0 := 1245,
	Productioncounters_Cavity_36_RejectReason_1 := 1246,
	Productioncounters_Cavity_36_RejectReason_2 := 1247,
	Productioncounters_Cavity_36_RejectReason_3 := 1248,
	Productioncounters_Cavity_36_RejectReason_4 := 1249,
	Productioncounters_Cavity_36_RejectReason_5 := 1250,
	Productioncounters_Cavity_36_RejectReason_6 := 1251,
	Productioncounters_Cavity_36_RejectReason_7 := 1252,
	Productioncounters_Cavity_36_RejectReason_8 := 1253,
	Productioncounters_Cavity_36_RejectReason_9 := 1254,
	Productioncounters_Cavity_36_RejectReason_10 := 1255,
	Productioncounters_Cavity_36_RejectReason_11 := 1256,
	Productioncounters_Cavity_36_RejectReason_12 := 1257,
	Productioncounters_Cavity_36_RejectReason_13 := 1258,
	Productioncounters_Cavity_36_RejectReason_14 := 1259,
	Productioncounters_Cavity_36_RejectReason_15 := 1260,
	Productioncounters_Cavity_36_RejectReason_16 := 1261,
	Productioncounters_Cavity_36_RejectReason_17 := 1262,
	Productioncounters_Cavity_36_RejectReason_18 := 1263,
	Productioncounters_Cavity_36_RejectReason_19 := 1264,
	Productioncounters_Cavity_36_RejectReason_20 := 1265,
	MouldMeasurement_Cavity_36_PeakPressure := 1266,
	MouldMeasurement_Hotrunner_Cavity_36_TargetValue := 1267,
	MouldMeasurement_Hotrunner_Cavity_36_ActualValue := 1268,
	Productioncounters_Cavity_37_Produced := 1269,
	Productioncounters_Cavity_37_Stacked := 1270,
	Productioncounters_Cavity_37_Rejected := 1271,
	Productioncounters_Cavity_37_UncountedReject := 1272,
	Productioncounters_Cavity_37_RejectReason_0 := 1273,
	Productioncounters_Cavity_37_RejectReason_1 := 1274,
	Productioncounters_Cavity_37_RejectReason_2 := 1275,
	Productioncounters_Cavity_37_RejectReason_3 := 1276,
	Productioncounters_Cavity_37_RejectReason_4 := 1277,
	Productioncounters_Cavity_37_RejectReason_5 := 1278,
	Productioncounters_Cavity_37_RejectReason_6 := 1279,
	Productioncounters_Cavity_37_RejectReason_7 := 1280,
	Productioncounters_Cavity_37_RejectReason_8 := 1281,
	Productioncounters_Cavity_37_RejectReason_9 := 1282,
	Productioncounters_Cavity_37_RejectReason_10 := 1283,
	Productioncounters_Cavity_37_RejectReason_11 := 1284,
	Productioncounters_Cavity_37_RejectReason_12 := 1285,
	Productioncounters_Cavity_37_RejectReason_13 := 1286,
	Productioncounters_Cavity_37_RejectReason_14 := 1287,
	Productioncounters_Cavity_37_RejectReason_15 := 1288,
	Productioncounters_Cavity_37_RejectReason_16 := 1289,
	Productioncounters_Cavity_37_RejectReason_17 := 1290,
	Productioncounters_Cavity_37_RejectReason_18 := 1291,
	Productioncounters_Cavity_37_RejectReason_19 := 1292,
	Productioncounters_Cavity_37_RejectReason_20 := 1293,
	MouldMeasurement_Cavity_37_PeakPressure := 1294,
	MouldMeasurement_Hotrunner_Cavity_37_TargetValue := 1295,
	MouldMeasurement_Hotrunner_Cavity_37_ActualValue := 1296,
	Productioncounters_Cavity_38_Produced := 1297,
	Productioncounters_Cavity_38_Stacked := 1298,
	Productioncounters_Cavity_38_Rejected := 1299,
	Productioncounters_Cavity_38_UncountedReject := 1300,
	Productioncounters_Cavity_38_RejectReason_0 := 1301,
	Productioncounters_Cavity_38_RejectReason_1 := 1302,
	Productioncounters_Cavity_38_RejectReason_2 := 1303,
	Productioncounters_Cavity_38_RejectReason_3 := 1304,
	Productioncounters_Cavity_38_RejectReason_4 := 1305,
	Productioncounters_Cavity_38_RejectReason_5 := 1306,
	Productioncounters_Cavity_38_RejectReason_6 := 1307,
	Productioncounters_Cavity_38_RejectReason_7 := 1308,
	Productioncounters_Cavity_38_RejectReason_8 := 1309,
	Productioncounters_Cavity_38_RejectReason_9 := 1310,
	Productioncounters_Cavity_38_RejectReason_10 := 1311,
	Productioncounters_Cavity_38_RejectReason_11 := 1312,
	Productioncounters_Cavity_38_RejectReason_12 := 1313,
	Productioncounters_Cavity_38_RejectReason_13 := 1314,
	Productioncounters_Cavity_38_RejectReason_14 := 1315,
	Productioncounters_Cavity_38_RejectReason_15 := 1316,
	Productioncounters_Cavity_38_RejectReason_16 := 1317,
	Productioncounters_Cavity_38_RejectReason_17 := 1318,
	Productioncounters_Cavity_38_RejectReason_18 := 1319,
	Productioncounters_Cavity_38_RejectReason_19 := 1320,
	Productioncounters_Cavity_38_RejectReason_20 := 1321,
	MouldMeasurement_Cavity_38_PeakPressure := 1322,
	MouldMeasurement_Hotrunner_Cavity_38_TargetValue := 1323,
	MouldMeasurement_Hotrunner_Cavity_38_ActualValue := 1324,
	Productioncounters_Cavity_39_Produced := 1325,
	Productioncounters_Cavity_39_Stacked := 1326,
	Productioncounters_Cavity_39_Rejected := 1327,
	Productioncounters_Cavity_39_UncountedReject := 1328,
	Productioncounters_Cavity_39_RejectReason_0 := 1329,
	Productioncounters_Cavity_39_RejectReason_1 := 1330,
	Productioncounters_Cavity_39_RejectReason_2 := 1331,
	Productioncounters_Cavity_39_RejectReason_3 := 1332,
	Productioncounters_Cavity_39_RejectReason_4 := 1333,
	Productioncounters_Cavity_39_RejectReason_5 := 1334,
	Productioncounters_Cavity_39_RejectReason_6 := 1335,
	Productioncounters_Cavity_39_RejectReason_7 := 1336,
	Productioncounters_Cavity_39_RejectReason_8 := 1337,
	Productioncounters_Cavity_39_RejectReason_9 := 1338,
	Productioncounters_Cavity_39_RejectReason_10 := 1339,
	Productioncounters_Cavity_39_RejectReason_11 := 1340,
	Productioncounters_Cavity_39_RejectReason_12 := 1341,
	Productioncounters_Cavity_39_RejectReason_13 := 1342,
	Productioncounters_Cavity_39_RejectReason_14 := 1343,
	Productioncounters_Cavity_39_RejectReason_15 := 1344,
	Productioncounters_Cavity_39_RejectReason_16 := 1345,
	Productioncounters_Cavity_39_RejectReason_17 := 1346,
	Productioncounters_Cavity_39_RejectReason_18 := 1347,
	Productioncounters_Cavity_39_RejectReason_19 := 1348,
	Productioncounters_Cavity_39_RejectReason_20 := 1349,
	MouldMeasurement_Cavity_39_PeakPressure := 1350,
	MouldMeasurement_Hotrunner_Cavity_39_TargetValue := 1351,
	MouldMeasurement_Hotrunner_Cavity_39_ActualValue := 1352,
	Productioncounters_Cavity_40_Produced := 1353,
	Productioncounters_Cavity_40_Stacked := 1354,
	Productioncounters_Cavity_40_Rejected := 1355,
	Productioncounters_Cavity_40_UncountedReject := 1356,
	Productioncounters_Cavity_40_RejectReason_0 := 1357,
	Productioncounters_Cavity_40_RejectReason_1 := 1358,
	Productioncounters_Cavity_40_RejectReason_2 := 1359,
	Productioncounters_Cavity_40_RejectReason_3 := 1360,
	Productioncounters_Cavity_40_RejectReason_4 := 1361,
	Productioncounters_Cavity_40_RejectReason_5 := 1362,
	Productioncounters_Cavity_40_RejectReason_6 := 1363,
	Productioncounters_Cavity_40_RejectReason_7 := 1364,
	Productioncounters_Cavity_40_RejectReason_8 := 1365,
	Productioncounters_Cavity_40_RejectReason_9 := 1366,
	Productioncounters_Cavity_40_RejectReason_10 := 1367,
	Productioncounters_Cavity_40_RejectReason_11 := 1368,
	Productioncounters_Cavity_40_RejectReason_12 := 1369,
	Productioncounters_Cavity_40_RejectReason_13 := 1370,
	Productioncounters_Cavity_40_RejectReason_14 := 1371,
	Productioncounters_Cavity_40_RejectReason_15 := 1372,
	Productioncounters_Cavity_40_RejectReason_16 := 1373,
	Productioncounters_Cavity_40_RejectReason_17 := 1374,
	Productioncounters_Cavity_40_RejectReason_18 := 1375,
	Productioncounters_Cavity_40_RejectReason_19 := 1376,
	Productioncounters_Cavity_40_RejectReason_20 := 1377,
	MouldMeasurement_Cavity_40_PeakPressure := 1378,
	MouldMeasurement_Hotrunner_Cavity_40_TargetValue := 1379,
	MouldMeasurement_Hotrunner_Cavity_40_ActualValue := 1380,
	Productioncounters_Cavity_41_Produced := 1381,
	Productioncounters_Cavity_41_Stacked := 1382,
	Productioncounters_Cavity_41_Rejected := 1383,
	Productioncounters_Cavity_41_UncountedReject := 1384,
	Productioncounters_Cavity_41_RejectReason_0 := 1385,
	Productioncounters_Cavity_41_RejectReason_1 := 1386,
	Productioncounters_Cavity_41_RejectReason_2 := 1387,
	Productioncounters_Cavity_41_RejectReason_3 := 1388,
	Productioncounters_Cavity_41_RejectReason_4 := 1389,
	Productioncounters_Cavity_41_RejectReason_5 := 1390,
	Productioncounters_Cavity_41_RejectReason_6 := 1391,
	Productioncounters_Cavity_41_RejectReason_7 := 1392,
	Productioncounters_Cavity_41_RejectReason_8 := 1393,
	Productioncounters_Cavity_41_RejectReason_9 := 1394,
	Productioncounters_Cavity_41_RejectReason_10 := 1395,
	Productioncounters_Cavity_41_RejectReason_11 := 1396,
	Productioncounters_Cavity_41_RejectReason_12 := 1397,
	Productioncounters_Cavity_41_RejectReason_13 := 1398,
	Productioncounters_Cavity_41_RejectReason_14 := 1399,
	Productioncounters_Cavity_41_RejectReason_15 := 1400,
	Productioncounters_Cavity_41_RejectReason_16 := 1401,
	Productioncounters_Cavity_41_RejectReason_17 := 1402,
	Productioncounters_Cavity_41_RejectReason_18 := 1403,
	Productioncounters_Cavity_41_RejectReason_19 := 1404,
	Productioncounters_Cavity_41_RejectReason_20 := 1405,
	MouldMeasurement_Cavity_41_PeakPressure := 1406,
	MouldMeasurement_Hotrunner_Cavity_41_TargetValue := 1407,
	MouldMeasurement_Hotrunner_Cavity_41_ActualValue := 1408,
	Productioncounters_Cavity_42_Produced := 1409,
	Productioncounters_Cavity_42_Stacked := 1410,
	Productioncounters_Cavity_42_Rejected := 1411,
	Productioncounters_Cavity_42_UncountedReject := 1412,
	Productioncounters_Cavity_42_RejectReason_0 := 1413,
	Productioncounters_Cavity_42_RejectReason_1 := 1414,
	Productioncounters_Cavity_42_RejectReason_2 := 1415,
	Productioncounters_Cavity_42_RejectReason_3 := 1416,
	Productioncounters_Cavity_42_RejectReason_4 := 1417,
	Productioncounters_Cavity_42_RejectReason_5 := 1418,
	Productioncounters_Cavity_42_RejectReason_6 := 1419,
	Productioncounters_Cavity_42_RejectReason_7 := 1420,
	Productioncounters_Cavity_42_RejectReason_8 := 1421,
	Productioncounters_Cavity_42_RejectReason_9 := 1422,
	Productioncounters_Cavity_42_RejectReason_10 := 1423,
	Productioncounters_Cavity_42_RejectReason_11 := 1424,
	Productioncounters_Cavity_42_RejectReason_12 := 1425,
	Productioncounters_Cavity_42_RejectReason_13 := 1426,
	Productioncounters_Cavity_42_RejectReason_14 := 1427,
	Productioncounters_Cavity_42_RejectReason_15 := 1428,
	Productioncounters_Cavity_42_RejectReason_16 := 1429,
	Productioncounters_Cavity_42_RejectReason_17 := 1430,
	Productioncounters_Cavity_42_RejectReason_18 := 1431,
	Productioncounters_Cavity_42_RejectReason_19 := 1432,
	Productioncounters_Cavity_42_RejectReason_20 := 1433,
	MouldMeasurement_Cavity_42_PeakPressure := 1434,
	MouldMeasurement_Hotrunner_Cavity_42_TargetValue := 1435,
	MouldMeasurement_Hotrunner_Cavity_42_ActualValue := 1436,
	Productioncounters_Cavity_43_Produced := 1437,
	Productioncounters_Cavity_43_Stacked := 1438,
	Productioncounters_Cavity_43_Rejected := 1439,
	Productioncounters_Cavity_43_UncountedReject := 1440,
	Productioncounters_Cavity_43_RejectReason_0 := 1441,
	Productioncounters_Cavity_43_RejectReason_1 := 1442,
	Productioncounters_Cavity_43_RejectReason_2 := 1443,
	Productioncounters_Cavity_43_RejectReason_3 := 1444,
	Productioncounters_Cavity_43_RejectReason_4 := 1445,
	Productioncounters_Cavity_43_RejectReason_5 := 1446,
	Productioncounters_Cavity_43_RejectReason_6 := 1447,
	Productioncounters_Cavity_43_RejectReason_7 := 1448,
	Productioncounters_Cavity_43_RejectReason_8 := 1449,
	Productioncounters_Cavity_43_RejectReason_9 := 1450,
	Productioncounters_Cavity_43_RejectReason_10 := 1451,
	Productioncounters_Cavity_43_RejectReason_11 := 1452,
	Productioncounters_Cavity_43_RejectReason_12 := 1453,
	Productioncounters_Cavity_43_RejectReason_13 := 1454,
	Productioncounters_Cavity_43_RejectReason_14 := 1455,
	Productioncounters_Cavity_43_RejectReason_15 := 1456,
	Productioncounters_Cavity_43_RejectReason_16 := 1457,
	Productioncounters_Cavity_43_RejectReason_17 := 1458,
	Productioncounters_Cavity_43_RejectReason_18 := 1459,
	Productioncounters_Cavity_43_RejectReason_19 := 1460,
	Productioncounters_Cavity_43_RejectReason_20 := 1461,
	MouldMeasurement_Cavity_43_PeakPressure := 1462,
	MouldMeasurement_Hotrunner_Cavity_43_TargetValue := 1463,
	MouldMeasurement_Hotrunner_Cavity_43_ActualValue := 1464,
	Productioncounters_Cavity_44_Produced := 1465,
	Productioncounters_Cavity_44_Stacked := 1466,
	Productioncounters_Cavity_44_Rejected := 1467,
	Productioncounters_Cavity_44_UncountedReject := 1468,
	Productioncounters_Cavity_44_RejectReason_0 := 1469,
	Productioncounters_Cavity_44_RejectReason_1 := 1470,
	Productioncounters_Cavity_44_RejectReason_2 := 1471,
	Productioncounters_Cavity_44_RejectReason_3 := 1472,
	Productioncounters_Cavity_44_RejectReason_4 := 1473,
	Productioncounters_Cavity_44_RejectReason_5 := 1474,
	Productioncounters_Cavity_44_RejectReason_6 := 1475,
	Productioncounters_Cavity_44_RejectReason_7 := 1476,
	Productioncounters_Cavity_44_RejectReason_8 := 1477,
	Productioncounters_Cavity_44_RejectReason_9 := 1478,
	Productioncounters_Cavity_44_RejectReason_10 := 1479,
	Productioncounters_Cavity_44_RejectReason_11 := 1480,
	Productioncounters_Cavity_44_RejectReason_12 := 1481,
	Productioncounters_Cavity_44_RejectReason_13 := 1482,
	Productioncounters_Cavity_44_RejectReason_14 := 1483,
	Productioncounters_Cavity_44_RejectReason_15 := 1484,
	Productioncounters_Cavity_44_RejectReason_16 := 1485,
	Productioncounters_Cavity_44_RejectReason_17 := 1486,
	Productioncounters_Cavity_44_RejectReason_18 := 1487,
	Productioncounters_Cavity_44_RejectReason_19 := 1488,
	Productioncounters_Cavity_44_RejectReason_20 := 1489,
	MouldMeasurement_Cavity_44_PeakPressure := 1490,
	MouldMeasurement_Hotrunner_Cavity_44_TargetValue := 1491,
	MouldMeasurement_Hotrunner_Cavity_44_ActualValue := 1492,
	Productioncounters_Cavity_45_Produced := 1493,
	Productioncounters_Cavity_45_Stacked := 1494,
	Productioncounters_Cavity_45_Rejected := 1495,
	Productioncounters_Cavity_45_UncountedReject := 1496,
	Productioncounters_Cavity_45_RejectReason_0 := 1497,
	Productioncounters_Cavity_45_RejectReason_1 := 1498,
	Productioncounters_Cavity_45_RejectReason_2 := 1499,
	Productioncounters_Cavity_45_RejectReason_3 := 1500,
	Productioncounters_Cavity_45_RejectReason_4 := 1501,
	Productioncounters_Cavity_45_RejectReason_5 := 1502,
	Productioncounters_Cavity_45_RejectReason_6 := 1503,
	Productioncounters_Cavity_45_RejectReason_7 := 1504,
	Productioncounters_Cavity_45_RejectReason_8 := 1505,
	Productioncounters_Cavity_45_RejectReason_9 := 1506,
	Productioncounters_Cavity_45_RejectReason_10 := 1507,
	Productioncounters_Cavity_45_RejectReason_11 := 1508,
	Productioncounters_Cavity_45_RejectReason_12 := 1509,
	Productioncounters_Cavity_45_RejectReason_13 := 1510,
	Productioncounters_Cavity_45_RejectReason_14 := 1511,
	Productioncounters_Cavity_45_RejectReason_15 := 1512,
	Productioncounters_Cavity_45_RejectReason_16 := 1513,
	Productioncounters_Cavity_45_RejectReason_17 := 1514,
	Productioncounters_Cavity_45_RejectReason_18 := 1515,
	Productioncounters_Cavity_45_RejectReason_19 := 1516,
	Productioncounters_Cavity_45_RejectReason_20 := 1517,
	MouldMeasurement_Cavity_45_PeakPressure := 1518,
	MouldMeasurement_Hotrunner_Cavity_45_TargetValue := 1519,
	MouldMeasurement_Hotrunner_Cavity_45_ActualValue := 1520,
	Productioncounters_Cavity_46_Produced := 1521,
	Productioncounters_Cavity_46_Stacked := 1522,
	Productioncounters_Cavity_46_Rejected := 1523,
	Productioncounters_Cavity_46_UncountedReject := 1524,
	Productioncounters_Cavity_46_RejectReason_0 := 1525,
	Productioncounters_Cavity_46_RejectReason_1 := 1526,
	Productioncounters_Cavity_46_RejectReason_2 := 1527,
	Productioncounters_Cavity_46_RejectReason_3 := 1528,
	Productioncounters_Cavity_46_RejectReason_4 := 1529,
	Productioncounters_Cavity_46_RejectReason_5 := 1530,
	Productioncounters_Cavity_46_RejectReason_6 := 1531,
	Productioncounters_Cavity_46_RejectReason_7 := 1532,
	Productioncounters_Cavity_46_RejectReason_8 := 1533,
	Productioncounters_Cavity_46_RejectReason_9 := 1534,
	Productioncounters_Cavity_46_RejectReason_10 := 1535,
	Productioncounters_Cavity_46_RejectReason_11 := 1536,
	Productioncounters_Cavity_46_RejectReason_12 := 1537,
	Productioncounters_Cavity_46_RejectReason_13 := 1538,
	Productioncounters_Cavity_46_RejectReason_14 := 1539,
	Productioncounters_Cavity_46_RejectReason_15 := 1540,
	Productioncounters_Cavity_46_RejectReason_16 := 1541,
	Productioncounters_Cavity_46_RejectReason_17 := 1542,
	Productioncounters_Cavity_46_RejectReason_18 := 1543,
	Productioncounters_Cavity_46_RejectReason_19 := 1544,
	Productioncounters_Cavity_46_RejectReason_20 := 1545,
	MouldMeasurement_Cavity_46_PeakPressure := 1546,
	MouldMeasurement_Hotrunner_Cavity_46_TargetValue := 1547,
	MouldMeasurement_Hotrunner_Cavity_46_ActualValue := 1548,
	Productioncounters_Cavity_47_Produced := 1549,
	Productioncounters_Cavity_47_Stacked := 1550,
	Productioncounters_Cavity_47_Rejected := 1551,
	Productioncounters_Cavity_47_UncountedReject := 1552,
	Productioncounters_Cavity_47_RejectReason_0 := 1553,
	Productioncounters_Cavity_47_RejectReason_1 := 1554,
	Productioncounters_Cavity_47_RejectReason_2 := 1555,
	Productioncounters_Cavity_47_RejectReason_3 := 1556,
	Productioncounters_Cavity_47_RejectReason_4 := 1557,
	Productioncounters_Cavity_47_RejectReason_5 := 1558,
	Productioncounters_Cavity_47_RejectReason_6 := 1559,
	Productioncounters_Cavity_47_RejectReason_7 := 1560,
	Productioncounters_Cavity_47_RejectReason_8 := 1561,
	Productioncounters_Cavity_47_RejectReason_9 := 1562,
	Productioncounters_Cavity_47_RejectReason_10 := 1563,
	Productioncounters_Cavity_47_RejectReason_11 := 1564,
	Productioncounters_Cavity_47_RejectReason_12 := 1565,
	Productioncounters_Cavity_47_RejectReason_13 := 1566,
	Productioncounters_Cavity_47_RejectReason_14 := 1567,
	Productioncounters_Cavity_47_RejectReason_15 := 1568,
	Productioncounters_Cavity_47_RejectReason_16 := 1569,
	Productioncounters_Cavity_47_RejectReason_17 := 1570,
	Productioncounters_Cavity_47_RejectReason_18 := 1571,
	Productioncounters_Cavity_47_RejectReason_19 := 1572,
	Productioncounters_Cavity_47_RejectReason_20 := 1573,
	MouldMeasurement_Cavity_47_PeakPressure := 1574,
	MouldMeasurement_Hotrunner_Cavity_47_TargetValue := 1575,
	MouldMeasurement_Hotrunner_Cavity_47_ActualValue := 1576,
	Productioncounters_Cavity_48_Produced := 1577,
	Productioncounters_Cavity_48_Stacked := 1578,
	Productioncounters_Cavity_48_Rejected := 1579,
	Productioncounters_Cavity_48_UncountedReject := 1580,
	Productioncounters_Cavity_48_RejectReason_0 := 1581,
	Productioncounters_Cavity_48_RejectReason_1 := 1582,
	Productioncounters_Cavity_48_RejectReason_2 := 1583,
	Productioncounters_Cavity_48_RejectReason_3 := 1584,
	Productioncounters_Cavity_48_RejectReason_4 := 1585,
	Productioncounters_Cavity_48_RejectReason_5 := 1586,
	Productioncounters_Cavity_48_RejectReason_6 := 1587,
	Productioncounters_Cavity_48_RejectReason_7 := 1588,
	Productioncounters_Cavity_48_RejectReason_8 := 1589,
	Productioncounters_Cavity_48_RejectReason_9 := 1590,
	Productioncounters_Cavity_48_RejectReason_10 := 1591,
	Productioncounters_Cavity_48_RejectReason_11 := 1592,
	Productioncounters_Cavity_48_RejectReason_12 := 1593,
	Productioncounters_Cavity_48_RejectReason_13 := 1594,
	Productioncounters_Cavity_48_RejectReason_14 := 1595,
	Productioncounters_Cavity_48_RejectReason_15 := 1596,
	Productioncounters_Cavity_48_RejectReason_16 := 1597,
	Productioncounters_Cavity_48_RejectReason_17 := 1598,
	Productioncounters_Cavity_48_RejectReason_18 := 1599,
	Productioncounters_Cavity_48_RejectReason_19 := 1600,
	Productioncounters_Cavity_48_RejectReason_20 := 1601,
	MouldMeasurement_Cavity_48_PeakPressure := 1602,
	MouldMeasurement_Hotrunner_Cavity_48_TargetValue := 1603,
	MouldMeasurement_Hotrunner_Cavity_48_ActualValue := 1604,
	Productioncounters_Cavity_49_Produced := 1605,
	Productioncounters_Cavity_49_Stacked := 1606,
	Productioncounters_Cavity_49_Rejected := 1607,
	Productioncounters_Cavity_49_UncountedReject := 1608,
	Productioncounters_Cavity_49_RejectReason_0 := 1609,
	Productioncounters_Cavity_49_RejectReason_1 := 1610,
	Productioncounters_Cavity_49_RejectReason_2 := 1611,
	Productioncounters_Cavity_49_RejectReason_3 := 1612,
	Productioncounters_Cavity_49_RejectReason_4 := 1613,
	Productioncounters_Cavity_49_RejectReason_5 := 1614,
	Productioncounters_Cavity_49_RejectReason_6 := 1615,
	Productioncounters_Cavity_49_RejectReason_7 := 1616,
	Productioncounters_Cavity_49_RejectReason_8 := 1617,
	Productioncounters_Cavity_49_RejectReason_9 := 1618,
	Productioncounters_Cavity_49_RejectReason_10 := 1619,
	Productioncounters_Cavity_49_RejectReason_11 := 1620,
	Productioncounters_Cavity_49_RejectReason_12 := 1621,
	Productioncounters_Cavity_49_RejectReason_13 := 1622,
	Productioncounters_Cavity_49_RejectReason_14 := 1623,
	Productioncounters_Cavity_49_RejectReason_15 := 1624,
	Productioncounters_Cavity_49_RejectReason_16 := 1625,
	Productioncounters_Cavity_49_RejectReason_17 := 1626,
	Productioncounters_Cavity_49_RejectReason_18 := 1627,
	Productioncounters_Cavity_49_RejectReason_19 := 1628,
	Productioncounters_Cavity_49_RejectReason_20 := 1629,
	MouldMeasurement_Cavity_49_PeakPressure := 1630,
	MouldMeasurement_Hotrunner_Cavity_49_TargetValue := 1631,
	MouldMeasurement_Hotrunner_Cavity_49_ActualValue := 1632,
	Productioncounters_Cavity_50_Produced := 1633,
	Productioncounters_Cavity_50_Stacked := 1634,
	Productioncounters_Cavity_50_Rejected := 1635,
	Productioncounters_Cavity_50_UncountedReject := 1636,
	Productioncounters_Cavity_50_RejectReason_0 := 1637,
	Productioncounters_Cavity_50_RejectReason_1 := 1638,
	Productioncounters_Cavity_50_RejectReason_2 := 1639,
	Productioncounters_Cavity_50_RejectReason_3 := 1640,
	Productioncounters_Cavity_50_RejectReason_4 := 1641,
	Productioncounters_Cavity_50_RejectReason_5 := 1642,
	Productioncounters_Cavity_50_RejectReason_6 := 1643,
	Productioncounters_Cavity_50_RejectReason_7 := 1644,
	Productioncounters_Cavity_50_RejectReason_8 := 1645,
	Productioncounters_Cavity_50_RejectReason_9 := 1646,
	Productioncounters_Cavity_50_RejectReason_10 := 1647,
	Productioncounters_Cavity_50_RejectReason_11 := 1648,
	Productioncounters_Cavity_50_RejectReason_12 := 1649,
	Productioncounters_Cavity_50_RejectReason_13 := 1650,
	Productioncounters_Cavity_50_RejectReason_14 := 1651,
	Productioncounters_Cavity_50_RejectReason_15 := 1652,
	Productioncounters_Cavity_50_RejectReason_16 := 1653,
	Productioncounters_Cavity_50_RejectReason_17 := 1654,
	Productioncounters_Cavity_50_RejectReason_18 := 1655,
	Productioncounters_Cavity_50_RejectReason_19 := 1656,
	Productioncounters_Cavity_50_RejectReason_20 := 1657,
	MouldMeasurement_Cavity_50_PeakPressure := 1658,
	MouldMeasurement_Hotrunner_Cavity_50_TargetValue := 1659,
	MouldMeasurement_Hotrunner_Cavity_50_ActualValue := 1660,
	Productioncounters_Cavity_51_Produced := 1661,
	Productioncounters_Cavity_51_Stacked := 1662,
	Productioncounters_Cavity_51_Rejected := 1663,
	Productioncounters_Cavity_51_UncountedReject := 1664,
	Productioncounters_Cavity_51_RejectReason_0 := 1665,
	Productioncounters_Cavity_51_RejectReason_1 := 1666,
	Productioncounters_Cavity_51_RejectReason_2 := 1667,
	Productioncounters_Cavity_51_RejectReason_3 := 1668,
	Productioncounters_Cavity_51_RejectReason_4 := 1669,
	Productioncounters_Cavity_51_RejectReason_5 := 1670,
	Productioncounters_Cavity_51_RejectReason_6 := 1671,
	Productioncounters_Cavity_51_RejectReason_7 := 1672,
	Productioncounters_Cavity_51_RejectReason_8 := 1673,
	Productioncounters_Cavity_51_RejectReason_9 := 1674,
	Productioncounters_Cavity_51_RejectReason_10 := 1675,
	Productioncounters_Cavity_51_RejectReason_11 := 1676,
	Productioncounters_Cavity_51_RejectReason_12 := 1677,
	Productioncounters_Cavity_51_RejectReason_13 := 1678,
	Productioncounters_Cavity_51_RejectReason_14 := 1679,
	Productioncounters_Cavity_51_RejectReason_15 := 1680,
	Productioncounters_Cavity_51_RejectReason_16 := 1681,
	Productioncounters_Cavity_51_RejectReason_17 := 1682,
	Productioncounters_Cavity_51_RejectReason_18 := 1683,
	Productioncounters_Cavity_51_RejectReason_19 := 1684,
	Productioncounters_Cavity_51_RejectReason_20 := 1685,
	MouldMeasurement_Cavity_51_PeakPressure := 1686,
	MouldMeasurement_Hotrunner_Cavity_51_TargetValue := 1687,
	MouldMeasurement_Hotrunner_Cavity_51_ActualValue := 1688,
	Productioncounters_Cavity_52_Produced := 1689,
	Productioncounters_Cavity_52_Stacked := 1690,
	Productioncounters_Cavity_52_Rejected := 1691,
	Productioncounters_Cavity_52_UncountedReject := 1692,
	Productioncounters_Cavity_52_RejectReason_0 := 1693,
	Productioncounters_Cavity_52_RejectReason_1 := 1694,
	Productioncounters_Cavity_52_RejectReason_2 := 1695,
	Productioncounters_Cavity_52_RejectReason_3 := 1696,
	Productioncounters_Cavity_52_RejectReason_4 := 1697,
	Productioncounters_Cavity_52_RejectReason_5 := 1698,
	Productioncounters_Cavity_52_RejectReason_6 := 1699,
	Productioncounters_Cavity_52_RejectReason_7 := 1700,
	Productioncounters_Cavity_52_RejectReason_8 := 1701,
	Productioncounters_Cavity_52_RejectReason_9 := 1702,
	Productioncounters_Cavity_52_RejectReason_10 := 1703,
	Productioncounters_Cavity_52_RejectReason_11 := 1704,
	Productioncounters_Cavity_52_RejectReason_12 := 1705,
	Productioncounters_Cavity_52_RejectReason_13 := 1706,
	Productioncounters_Cavity_52_RejectReason_14 := 1707,
	Productioncounters_Cavity_52_RejectReason_15 := 1708,
	Productioncounters_Cavity_52_RejectReason_16 := 1709,
	Productioncounters_Cavity_52_RejectReason_17 := 1710,
	Productioncounters_Cavity_52_RejectReason_18 := 1711,
	Productioncounters_Cavity_52_RejectReason_19 := 1712,
	Productioncounters_Cavity_52_RejectReason_20 := 1713,
	MouldMeasurement_Cavity_52_PeakPressure := 1714,
	MouldMeasurement_Hotrunner_Cavity_52_TargetValue := 1715,
	MouldMeasurement_Hotrunner_Cavity_52_ActualValue := 1716,
	Productioncounters_Cavity_53_Produced := 1717,
	Productioncounters_Cavity_53_Stacked := 1718,
	Productioncounters_Cavity_53_Rejected := 1719,
	Productioncounters_Cavity_53_UncountedReject := 1720,
	Productioncounters_Cavity_53_RejectReason_0 := 1721,
	Productioncounters_Cavity_53_RejectReason_1 := 1722,
	Productioncounters_Cavity_53_RejectReason_2 := 1723,
	Productioncounters_Cavity_53_RejectReason_3 := 1724,
	Productioncounters_Cavity_53_RejectReason_4 := 1725,
	Productioncounters_Cavity_53_RejectReason_5 := 1726,
	Productioncounters_Cavity_53_RejectReason_6 := 1727,
	Productioncounters_Cavity_53_RejectReason_7 := 1728,
	Productioncounters_Cavity_53_RejectReason_8 := 1729,
	Productioncounters_Cavity_53_RejectReason_9 := 1730,
	Productioncounters_Cavity_53_RejectReason_10 := 1731,
	Productioncounters_Cavity_53_RejectReason_11 := 1732,
	Productioncounters_Cavity_53_RejectReason_12 := 1733,
	Productioncounters_Cavity_53_RejectReason_13 := 1734,
	Productioncounters_Cavity_53_RejectReason_14 := 1735,
	Productioncounters_Cavity_53_RejectReason_15 := 1736,
	Productioncounters_Cavity_53_RejectReason_16 := 1737,
	Productioncounters_Cavity_53_RejectReason_17 := 1738,
	Productioncounters_Cavity_53_RejectReason_18 := 1739,
	Productioncounters_Cavity_53_RejectReason_19 := 1740,
	Productioncounters_Cavity_53_RejectReason_20 := 1741,
	MouldMeasurement_Cavity_53_PeakPressure := 1742,
	MouldMeasurement_Hotrunner_Cavity_53_TargetValue := 1743,
	MouldMeasurement_Hotrunner_Cavity_53_ActualValue := 1744,
	Productioncounters_Cavity_54_Produced := 1745,
	Productioncounters_Cavity_54_Stacked := 1746,
	Productioncounters_Cavity_54_Rejected := 1747,
	Productioncounters_Cavity_54_UncountedReject := 1748,
	Productioncounters_Cavity_54_RejectReason_0 := 1749,
	Productioncounters_Cavity_54_RejectReason_1 := 1750,
	Productioncounters_Cavity_54_RejectReason_2 := 1751,
	Productioncounters_Cavity_54_RejectReason_3 := 1752,
	Productioncounters_Cavity_54_RejectReason_4 := 1753,
	Productioncounters_Cavity_54_RejectReason_5 := 1754,
	Productioncounters_Cavity_54_RejectReason_6 := 1755,
	Productioncounters_Cavity_54_RejectReason_7 := 1756,
	Productioncounters_Cavity_54_RejectReason_8 := 1757,
	Productioncounters_Cavity_54_RejectReason_9 := 1758,
	Productioncounters_Cavity_54_RejectReason_10 := 1759,
	Productioncounters_Cavity_54_RejectReason_11 := 1760,
	Productioncounters_Cavity_54_RejectReason_12 := 1761,
	Productioncounters_Cavity_54_RejectReason_13 := 1762,
	Productioncounters_Cavity_54_RejectReason_14 := 1763,
	Productioncounters_Cavity_54_RejectReason_15 := 1764,
	Productioncounters_Cavity_54_RejectReason_16 := 1765,
	Productioncounters_Cavity_54_RejectReason_17 := 1766,
	Productioncounters_Cavity_54_RejectReason_18 := 1767,
	Productioncounters_Cavity_54_RejectReason_19 := 1768,
	Productioncounters_Cavity_54_RejectReason_20 := 1769,
	MouldMeasurement_Cavity_54_PeakPressure := 1770,
	MouldMeasurement_Hotrunner_Cavity_54_TargetValue := 1771,
	MouldMeasurement_Hotrunner_Cavity_54_ActualValue := 1772,
	Productioncounters_Cavity_55_Produced := 1773,
	Productioncounters_Cavity_55_Stacked := 1774,
	Productioncounters_Cavity_55_Rejected := 1775,
	Productioncounters_Cavity_55_UncountedReject := 1776,
	Productioncounters_Cavity_55_RejectReason_0 := 1777,
	Productioncounters_Cavity_55_RejectReason_1 := 1778,
	Productioncounters_Cavity_55_RejectReason_2 := 1779,
	Productioncounters_Cavity_55_RejectReason_3 := 1780,
	Productioncounters_Cavity_55_RejectReason_4 := 1781,
	Productioncounters_Cavity_55_RejectReason_5 := 1782,
	Productioncounters_Cavity_55_RejectReason_6 := 1783,
	Productioncounters_Cavity_55_RejectReason_7 := 1784,
	Productioncounters_Cavity_55_RejectReason_8 := 1785,
	Productioncounters_Cavity_55_RejectReason_9 := 1786,
	Productioncounters_Cavity_55_RejectReason_10 := 1787,
	Productioncounters_Cavity_55_RejectReason_11 := 1788,
	Productioncounters_Cavity_55_RejectReason_12 := 1789,
	Productioncounters_Cavity_55_RejectReason_13 := 1790,
	Productioncounters_Cavity_55_RejectReason_14 := 1791,
	Productioncounters_Cavity_55_RejectReason_15 := 1792,
	Productioncounters_Cavity_55_RejectReason_16 := 1793,
	Productioncounters_Cavity_55_RejectReason_17 := 1794,
	Productioncounters_Cavity_55_RejectReason_18 := 1795,
	Productioncounters_Cavity_55_RejectReason_19 := 1796,
	Productioncounters_Cavity_55_RejectReason_20 := 1797,
	MouldMeasurement_Cavity_55_PeakPressure := 1798,
	MouldMeasurement_Hotrunner_Cavity_55_TargetValue := 1799,
	MouldMeasurement_Hotrunner_Cavity_55_ActualValue := 1800,
	Productioncounters_Cavity_56_Produced := 1801,
	Productioncounters_Cavity_56_Stacked := 1802,
	Productioncounters_Cavity_56_Rejected := 1803,
	Productioncounters_Cavity_56_UncountedReject := 1804,
	Productioncounters_Cavity_56_RejectReason_0 := 1805,
	Productioncounters_Cavity_56_RejectReason_1 := 1806,
	Productioncounters_Cavity_56_RejectReason_2 := 1807,
	Productioncounters_Cavity_56_RejectReason_3 := 1808,
	Productioncounters_Cavity_56_RejectReason_4 := 1809,
	Productioncounters_Cavity_56_RejectReason_5 := 1810,
	Productioncounters_Cavity_56_RejectReason_6 := 1811,
	Productioncounters_Cavity_56_RejectReason_7 := 1812,
	Productioncounters_Cavity_56_RejectReason_8 := 1813,
	Productioncounters_Cavity_56_RejectReason_9 := 1814,
	Productioncounters_Cavity_56_RejectReason_10 := 1815,
	Productioncounters_Cavity_56_RejectReason_11 := 1816,
	Productioncounters_Cavity_56_RejectReason_12 := 1817,
	Productioncounters_Cavity_56_RejectReason_13 := 1818,
	Productioncounters_Cavity_56_RejectReason_14 := 1819,
	Productioncounters_Cavity_56_RejectReason_15 := 1820,
	Productioncounters_Cavity_56_RejectReason_16 := 1821,
	Productioncounters_Cavity_56_RejectReason_17 := 1822,
	Productioncounters_Cavity_56_RejectReason_18 := 1823,
	Productioncounters_Cavity_56_RejectReason_19 := 1824,
	Productioncounters_Cavity_56_RejectReason_20 := 1825,
	MouldMeasurement_Cavity_56_PeakPressure := 1826,
	MouldMeasurement_Hotrunner_Cavity_56_TargetValue := 1827,
	MouldMeasurement_Hotrunner_Cavity_56_ActualValue := 1828,
	Productioncounters_Cavity_57_Produced := 1829,
	Productioncounters_Cavity_57_Stacked := 1830,
	Productioncounters_Cavity_57_Rejected := 1831,
	Productioncounters_Cavity_57_UncountedReject := 1832,
	Productioncounters_Cavity_57_RejectReason_0 := 1833,
	Productioncounters_Cavity_57_RejectReason_1 := 1834,
	Productioncounters_Cavity_57_RejectReason_2 := 1835,
	Productioncounters_Cavity_57_RejectReason_3 := 1836,
	Productioncounters_Cavity_57_RejectReason_4 := 1837,
	Productioncounters_Cavity_57_RejectReason_5 := 1838,
	Productioncounters_Cavity_57_RejectReason_6 := 1839,
	Productioncounters_Cavity_57_RejectReason_7 := 1840,
	Productioncounters_Cavity_57_RejectReason_8 := 1841,
	Productioncounters_Cavity_57_RejectReason_9 := 1842,
	Productioncounters_Cavity_57_RejectReason_10 := 1843,
	Productioncounters_Cavity_57_RejectReason_11 := 1844,
	Productioncounters_Cavity_57_RejectReason_12 := 1845,
	Productioncounters_Cavity_57_RejectReason_13 := 1846,
	Productioncounters_Cavity_57_RejectReason_14 := 1847,
	Productioncounters_Cavity_57_RejectReason_15 := 1848,
	Productioncounters_Cavity_57_RejectReason_16 := 1849,
	Productioncounters_Cavity_57_RejectReason_17 := 1850,
	Productioncounters_Cavity_57_RejectReason_18 := 1851,
	Productioncounters_Cavity_57_RejectReason_19 := 1852,
	Productioncounters_Cavity_57_RejectReason_20 := 1853,
	MouldMeasurement_Cavity_57_PeakPressure := 1854,
	MouldMeasurement_Hotrunner_Cavity_57_TargetValue := 1855,
	MouldMeasurement_Hotrunner_Cavity_57_ActualValue := 1856,
	Productioncounters_Cavity_58_Produced := 1857,
	Productioncounters_Cavity_58_Stacked := 1858,
	Productioncounters_Cavity_58_Rejected := 1859,
	Productioncounters_Cavity_58_UncountedReject := 1860,
	Productioncounters_Cavity_58_RejectReason_0 := 1861,
	Productioncounters_Cavity_58_RejectReason_1 := 1862,
	Productioncounters_Cavity_58_RejectReason_2 := 1863,
	Productioncounters_Cavity_58_RejectReason_3 := 1864,
	Productioncounters_Cavity_58_RejectReason_4 := 1865,
	Productioncounters_Cavity_58_RejectReason_5 := 1866,
	Productioncounters_Cavity_58_RejectReason_6 := 1867,
	Productioncounters_Cavity_58_RejectReason_7 := 1868,
	Productioncounters_Cavity_58_RejectReason_8 := 1869,
	Productioncounters_Cavity_58_RejectReason_9 := 1870,
	Productioncounters_Cavity_58_RejectReason_10 := 1871,
	Productioncounters_Cavity_58_RejectReason_11 := 1872,
	Productioncounters_Cavity_58_RejectReason_12 := 1873,
	Productioncounters_Cavity_58_RejectReason_13 := 1874,
	Productioncounters_Cavity_58_RejectReason_14 := 1875,
	Productioncounters_Cavity_58_RejectReason_15 := 1876,
	Productioncounters_Cavity_58_RejectReason_16 := 1877,
	Productioncounters_Cavity_58_RejectReason_17 := 1878,
	Productioncounters_Cavity_58_RejectReason_18 := 1879,
	Productioncounters_Cavity_58_RejectReason_19 := 1880,
	Productioncounters_Cavity_58_RejectReason_20 := 1881,
	MouldMeasurement_Cavity_58_PeakPressure := 1882,
	MouldMeasurement_Hotrunner_Cavity_58_TargetValue := 1883,
	MouldMeasurement_Hotrunner_Cavity_58_ActualValue := 1884,
	Productioncounters_Cavity_59_Produced := 1885,
	Productioncounters_Cavity_59_Stacked := 1886,
	Productioncounters_Cavity_59_Rejected := 1887,
	Productioncounters_Cavity_59_UncountedReject := 1888,
	Productioncounters_Cavity_59_RejectReason_0 := 1889,
	Productioncounters_Cavity_59_RejectReason_1 := 1890,
	Productioncounters_Cavity_59_RejectReason_2 := 1891,
	Productioncounters_Cavity_59_RejectReason_3 := 1892,
	Productioncounters_Cavity_59_RejectReason_4 := 1893,
	Productioncounters_Cavity_59_RejectReason_5 := 1894,
	Productioncounters_Cavity_59_RejectReason_6 := 1895,
	Productioncounters_Cavity_59_RejectReason_7 := 1896,
	Productioncounters_Cavity_59_RejectReason_8 := 1897,
	Productioncounters_Cavity_59_RejectReason_9 := 1898,
	Productioncounters_Cavity_59_RejectReason_10 := 1899,
	Productioncounters_Cavity_59_RejectReason_11 := 1900,
	Productioncounters_Cavity_59_RejectReason_12 := 1901,
	Productioncounters_Cavity_59_RejectReason_13 := 1902,
	Productioncounters_Cavity_59_RejectReason_14 := 1903,
	Productioncounters_Cavity_59_RejectReason_15 := 1904,
	Productioncounters_Cavity_59_RejectReason_16 := 1905,
	Productioncounters_Cavity_59_RejectReason_17 := 1906,
	Productioncounters_Cavity_59_RejectReason_18 := 1907,
	Productioncounters_Cavity_59_RejectReason_19 := 1908,
	Productioncounters_Cavity_59_RejectReason_20 := 1909,
	MouldMeasurement_Cavity_59_PeakPressure := 1910,
	MouldMeasurement_Hotrunner_Cavity_59_TargetValue := 1911,
	MouldMeasurement_Hotrunner_Cavity_59_ActualValue := 1912,
	Productioncounters_Cavity_60_Produced := 1913,
	Productioncounters_Cavity_60_Stacked := 1914,
	Productioncounters_Cavity_60_Rejected := 1915,
	Productioncounters_Cavity_60_UncountedReject := 1916,
	Productioncounters_Cavity_60_RejectReason_0 := 1917,
	Productioncounters_Cavity_60_RejectReason_1 := 1918,
	Productioncounters_Cavity_60_RejectReason_2 := 1919,
	Productioncounters_Cavity_60_RejectReason_3 := 1920,
	Productioncounters_Cavity_60_RejectReason_4 := 1921,
	Productioncounters_Cavity_60_RejectReason_5 := 1922,
	Productioncounters_Cavity_60_RejectReason_6 := 1923,
	Productioncounters_Cavity_60_RejectReason_7 := 1924,
	Productioncounters_Cavity_60_RejectReason_8 := 1925,
	Productioncounters_Cavity_60_RejectReason_9 := 1926,
	Productioncounters_Cavity_60_RejectReason_10 := 1927,
	Productioncounters_Cavity_60_RejectReason_11 := 1928,
	Productioncounters_Cavity_60_RejectReason_12 := 1929,
	Productioncounters_Cavity_60_RejectReason_13 := 1930,
	Productioncounters_Cavity_60_RejectReason_14 := 1931,
	Productioncounters_Cavity_60_RejectReason_15 := 1932,
	Productioncounters_Cavity_60_RejectReason_16 := 1933,
	Productioncounters_Cavity_60_RejectReason_17 := 1934,
	Productioncounters_Cavity_60_RejectReason_18 := 1935,
	Productioncounters_Cavity_60_RejectReason_19 := 1936,
	Productioncounters_Cavity_60_RejectReason_20 := 1937,
	MouldMeasurement_Cavity_60_PeakPressure := 1938,
	MouldMeasurement_Hotrunner_Cavity_60_TargetValue := 1939,
	MouldMeasurement_Hotrunner_Cavity_60_ActualValue := 1940,
	Productioncounters_Cavity_61_Produced := 1941,
	Productioncounters_Cavity_61_Stacked := 1942,
	Productioncounters_Cavity_61_Rejected := 1943,
	Productioncounters_Cavity_61_UncountedReject := 1944,
	Productioncounters_Cavity_61_RejectReason_0 := 1945,
	Productioncounters_Cavity_61_RejectReason_1 := 1946,
	Productioncounters_Cavity_61_RejectReason_2 := 1947,
	Productioncounters_Cavity_61_RejectReason_3 := 1948,
	Productioncounters_Cavity_61_RejectReason_4 := 1949,
	Productioncounters_Cavity_61_RejectReason_5 := 1950,
	Productioncounters_Cavity_61_RejectReason_6 := 1951,
	Productioncounters_Cavity_61_RejectReason_7 := 1952,
	Productioncounters_Cavity_61_RejectReason_8 := 1953,
	Productioncounters_Cavity_61_RejectReason_9 := 1954,
	Productioncounters_Cavity_61_RejectReason_10 := 1955,
	Productioncounters_Cavity_61_RejectReason_11 := 1956,
	Productioncounters_Cavity_61_RejectReason_12 := 1957,
	Productioncounters_Cavity_61_RejectReason_13 := 1958,
	Productioncounters_Cavity_61_RejectReason_14 := 1959,
	Productioncounters_Cavity_61_RejectReason_15 := 1960,
	Productioncounters_Cavity_61_RejectReason_16 := 1961,
	Productioncounters_Cavity_61_RejectReason_17 := 1962,
	Productioncounters_Cavity_61_RejectReason_18 := 1963,
	Productioncounters_Cavity_61_RejectReason_19 := 1964,
	Productioncounters_Cavity_61_RejectReason_20 := 1965,
	MouldMeasurement_Cavity_61_PeakPressure := 1966,
	MouldMeasurement_Hotrunner_Cavity_61_TargetValue := 1967,
	MouldMeasurement_Hotrunner_Cavity_61_ActualValue := 1968,
	Productioncounters_Cavity_62_Produced := 1969,
	Productioncounters_Cavity_62_Stacked := 1970,
	Productioncounters_Cavity_62_Rejected := 1971,
	Productioncounters_Cavity_62_UncountedReject := 1972,
	Productioncounters_Cavity_62_RejectReason_0 := 1973,
	Productioncounters_Cavity_62_RejectReason_1 := 1974,
	Productioncounters_Cavity_62_RejectReason_2 := 1975,
	Productioncounters_Cavity_62_RejectReason_3 := 1976,
	Productioncounters_Cavity_62_RejectReason_4 := 1977,
	Productioncounters_Cavity_62_RejectReason_5 := 1978,
	Productioncounters_Cavity_62_RejectReason_6 := 1979,
	Productioncounters_Cavity_62_RejectReason_7 := 1980,
	Productioncounters_Cavity_62_RejectReason_8 := 1981,
	Productioncounters_Cavity_62_RejectReason_9 := 1982,
	Productioncounters_Cavity_62_RejectReason_10 := 1983,
	Productioncounters_Cavity_62_RejectReason_11 := 1984,
	Productioncounters_Cavity_62_RejectReason_12 := 1985,
	Productioncounters_Cavity_62_RejectReason_13 := 1986,
	Productioncounters_Cavity_62_RejectReason_14 := 1987,
	Productioncounters_Cavity_62_RejectReason_15 := 1988,
	Productioncounters_Cavity_62_RejectReason_16 := 1989,
	Productioncounters_Cavity_62_RejectReason_17 := 1990,
	Productioncounters_Cavity_62_RejectReason_18 := 1991,
	Productioncounters_Cavity_62_RejectReason_19 := 1992,
	Productioncounters_Cavity_62_RejectReason_20 := 1993,
	MouldMeasurement_Cavity_62_PeakPressure := 1994,
	MouldMeasurement_Hotrunner_Cavity_62_TargetValue := 1995,
	MouldMeasurement_Hotrunner_Cavity_62_ActualValue := 1996,
	Productioncounters_Cavity_63_Produced := 1997,
	Productioncounters_Cavity_63_Stacked := 1998,
	Productioncounters_Cavity_63_Rejected := 1999,
	Productioncounters_Cavity_63_UncountedReject := 2000,
	Productioncounters_Cavity_63_RejectReason_0 := 2001,
	Productioncounters_Cavity_63_RejectReason_1 := 2002,
	Productioncounters_Cavity_63_RejectReason_2 := 2003,
	Productioncounters_Cavity_63_RejectReason_3 := 2004,
	Productioncounters_Cavity_63_RejectReason_4 := 2005,
	Productioncounters_Cavity_63_RejectReason_5 := 2006,
	Productioncounters_Cavity_63_RejectReason_6 := 2007,
	Productioncounters_Cavity_63_RejectReason_7 := 2008,
	Productioncounters_Cavity_63_RejectReason_8 := 2009,
	Productioncounters_Cavity_63_RejectReason_9 := 2010,
	Productioncounters_Cavity_63_RejectReason_10 := 2011,
	Productioncounters_Cavity_63_RejectReason_11 := 2012,
	Productioncounters_Cavity_63_RejectReason_12 := 2013,
	Productioncounters_Cavity_63_RejectReason_13 := 2014,
	Productioncounters_Cavity_63_RejectReason_14 := 2015,
	Productioncounters_Cavity_63_RejectReason_15 := 2016,
	Productioncounters_Cavity_63_RejectReason_16 := 2017,
	Productioncounters_Cavity_63_RejectReason_17 := 2018,
	Productioncounters_Cavity_63_RejectReason_18 := 2019,
	Productioncounters_Cavity_63_RejectReason_19 := 2020,
	Productioncounters_Cavity_63_RejectReason_20 := 2021,
	MouldMeasurement_Cavity_63_PeakPressure := 2022,
	MouldMeasurement_Hotrunner_Cavity_63_TargetValue := 2023,
	MouldMeasurement_Hotrunner_Cavity_63_ActualValue := 2024,
	Productioncounters_Cavity_64_Produced := 2025,
	Productioncounters_Cavity_64_Stacked := 2026,
	Productioncounters_Cavity_64_Rejected := 2027,
	Productioncounters_Cavity_64_UncountedReject := 2028,
	Productioncounters_Cavity_64_RejectReason_0 := 2029,
	Productioncounters_Cavity_64_RejectReason_1 := 2030,
	Productioncounters_Cavity_64_RejectReason_2 := 2031,
	Productioncounters_Cavity_64_RejectReason_3 := 2032,
	Productioncounters_Cavity_64_RejectReason_4 := 2033,
	Productioncounters_Cavity_64_RejectReason_5 := 2034,
	Productioncounters_Cavity_64_RejectReason_6 := 2035,
	Productioncounters_Cavity_64_RejectReason_7 := 2036,
	Productioncounters_Cavity_64_RejectReason_8 := 2037,
	Productioncounters_Cavity_64_RejectReason_9 := 2038,
	Productioncounters_Cavity_64_RejectReason_10 := 2039,
	Productioncounters_Cavity_64_RejectReason_11 := 2040,
	Productioncounters_Cavity_64_RejectReason_12 := 2041,
	Productioncounters_Cavity_64_RejectReason_13 := 2042,
	Productioncounters_Cavity_64_RejectReason_14 := 2043,
	Productioncounters_Cavity_64_RejectReason_15 := 2044,
	Productioncounters_Cavity_64_RejectReason_16 := 2045,
	Productioncounters_Cavity_64_RejectReason_17 := 2046,
	Productioncounters_Cavity_64_RejectReason_18 := 2047,
	Productioncounters_Cavity_64_RejectReason_19 := 2048,
	Productioncounters_Cavity_64_RejectReason_20 := 2049,
	MouldMeasurement_Cavity_64_PeakPressure := 2050,
	MouldMeasurement_Hotrunner_Cavity_64_TargetValue := 2051,
	MouldMeasurement_Hotrunner_Cavity_64_ActualValue := 2052,
	CycleTimes_TargetCycleTime := 2053,
	Magazine_SensorTimes_Vacuum_5 := 2054,
	Magazine_SensorTimes_Vacuum_6 := 2055,
	Magazine_SensorTimes_Vacuum_7 := 2056,
	Magazine_SensorTimes_Vacuum_8 := 2057,
	BoxConveyor_Alarms := 2058,
	Fanuc_Alarms := 2059,
	Magazine_SensorTimes_RotateIn := 2060,
	Magazine_SensorTimes_RotateOut := 2061,
	Magazine_SensorTimes_ShiftIn := 2062,
	Magazine_SensorTimes_ShiftOut := 2063,
	YUnit_BFU_CoveredDistance := 2064,
	ZUnit_BFU_CoveredDistance := 2065,
	ZUnit_BFU_ErrorId := 2066,
	YUnit_BFU_ErrorId := 2067,
	ZUnit_BFU_AxisErrorId := 2068,
	YUnit_BFU_AxisErrorId := 2069,
	ZUnit_BFU_DriveUtilisation := 2070,
	YUnit_BFU_DriveUtilisation := 2071,
	YUnit_BFU_MotorUtilisation := 2072,
	ZUnit_BFU_MotorUtilisation := 2073,
	YUnit_BFU_Alarms := 2074,
	ZUnit_BFU_Alarms := 2075,
	BoxConveyor_SensorTimes_LiftIn := 2076,
	BoxConveyor_SensorTimes_LiftOut := 2077,
	BoxConveyor_SensorTimes_OpenBoxLongSideIn := 2078,
	BoxConveyor_SensorTimes_OpenBoxLongSideOut := 2079,
	BoxConveyor_SensorTimes_OpenBoxShortSideIn := 2080,
	BoxConveyor_SensorTimes_OpenBoxShortSideOut := 2081,
	BFU_PickAndPlace_SensorTimes_ClampIn := 2082,
	BFU_PickAndPlace_SensorTimes_ClampOut := 2083,
	BFU_PickAndPlace_SensorTimes_PatternizerPusherIn := 2084,
	BFU_PickAndPlace_SensorTimes_PatternizerPusherOut := 2085,
	BFU_PickAndPlace_SensorTimes_PatternizerExtendIn := 2086,
	BFU_PickAndPlace_SensorTimes_PatternizerExtendOut := 2087,
	YUnit_BFU_DriveErrorId := 2088,
	ZUnit_BFU_DriveErrorId := 2089,
	BFU_PickAndPlace_Alarms := 2090,
	BoxConveyor_SensorTimes_ClampSecondBoxOut := 2091,
	BoxConveyor_SensorTimes_ClampSecondBoxIn := 2092,
	BoxConveyor_SensorTimes_BoxStopperOut := 2093,
	BoxConveyor_SensorTimes_BoxStopperIn := 2094,
	Conveyors_BFU_DriveUtilisation := 2095,
	Conveyors_BFU_MotorUtilisation := 2096,
	Conveyors_BFU_DriveErrorId := 2097,
	Conveyors_BFU_AxisErrorId := 2098,
	Conveyors_BFU_ErrorId := 2099,
	Conveyors_BFU_CoveredDistance := 2100,
	Magazine_ActiveDrawer := 2101,
	Main_ProductWeight := 2102,
	Patternizer_Alarms := 2103,
	OutfeedTransfer_Alarms := 2104,
	Camera_YUnit_Alarms := 2105,
	ZUnit_SensorTimes_Extend1Out := 2106,
	ZUnit_SensorTimes_Extend2Out := 2107,
	ZUnit_SensorTimes_Extend3Out := 2108,
	ZUnit_SensorTimes_Extend4Out := 2109,
	ZUnit_SensorTimes_BlockStackIn := 2110,
	ZUnit_SensorTimes_BlockStackOut := 2111,
	Camera_2_Alarms := 2112,
	Camera_2_Time_Active := 2113,
	Camera_2_Time_Idle := 2114,
	Z1Unit_Alarms := 2115,
	Z2Unit_Alarms := 2116,
	ZrUnit_Zr1_Alarms := 2117,
	HMU_Alarms := 2118,
	ZrUnit_Zr2_Alarms := 2119,
	PrUnit_Alarms := 2120,
	LUnit_Alarms := 2121,
	Magazine_CoveredDistance := 2122,
	Z1Unit_CoveredDistance := 2123,
	PrUnit_CoveredDistance := 2124,
	Z2Unit_CoveredDistance := 2125,
	LUnit_L1_CoveredDistance := 2126,
	LUnit_L2_CoveredDistance := 2127,
	LUnit_L3_CoveredDistance := 2128,
	LUnit_L4_CoveredDistance := 2129,
	Magazine_ErrorId := 2130,
	Z1Unit_ErrorId := 2131,
	PrUnit_ErrorId := 2132,
	Z2Unit_ErrorId := 2133,
	LUnit_L1_ErrorId := 2134,
	LUnit_L2_ErrorId := 2135,
	LUnit_L3_ErrorId := 2136,
	LUnit_L4_ErrorId := 2137,
	ZrUnit_Zr3_Alarms := 2138,
	ZrUnit_Zr4_Alarms := 2139,
	Magazine_AxisErrorId := 2140,
	Z1Unit_AxisErrorId := 2141,
	ZrUnit_Zr1_AxisErrorId := 2142,
	ZrUnit_Zr2_AxisErrorId := 2143,
	ZrUnit_Zr3_AxisErrorId := 2144,
	ZrUnit_Zr4_AxisErrorId := 2145,
	PrUnit_AxisErrorId := 2146,
	Z2Unit_AxisErrorId := 2147,
	LUnit_L1_AxisErrorId := 2148,
	LUnit_L2_AxisErrorId := 2149,
	LUnit_L3_AxisErrorId := 2150,
	LUnit_L4_AxisErrorId := 2151,
	Magazine_DriveErrorId := 2152,
	Z1Unit_DriveErrorId := 2153,
	ZrUnit_Zr1_DriveErrorId := 2154,
	ZrUnit_Zr2_DriveErrorId := 2155,
	ZrUnit_Zr3_DriveErrorId := 2156,
	ZrUnit_Zr4_DriveErrorId := 2157,
	PrUnit_DriveErrorId := 2158,
	Z2Unit_DriveErrorId := 2159,
	LUnit_L1_DriveErrorId := 2160,
	LUnit_L2_DriveErrorId := 2161,
	LUnit_L3_DriveErrorId := 2162,
	LUnit_L4_DriveErrorId := 2163,
	Magazine_DriveUtilisation := 2164,
	Z1Unit_DriveUtilisation := 2165,
	PrUnit_DriveUtilisation := 2166,
	Z2Unit_DriveUtilisation := 2167,
	LUnit_L1_DriveUtilisation := 2168,
	LUnit_L2_DriveUtilisation := 2169,
	LUnit_L3_DriveUtilisation := 2170,
	LUnit_L4_DriveUtilisation := 2171,
	Magazine_MotorUtilisation := 2172,
	Z1Unit_MotorUtilisation := 2173,
	PrUnit_MotorUtilisation := 2174,
	Z2Unit_MotorUtilisation := 2175,
	LUnit_L1_MotorUtilisation := 2176,
	LUnit_L2_MotorUtilisation := 2177,
	LUnit_L3_MotorUtilisation := 2178,
	LUnit_L4_MotorUtilisation := 2179,
	Magazine_SensorTimes_ExtendIn := 2180,
	Magazine_SensorTimes_ExtendOut := 2181,
	HMU_SensorTimes_FixedBufferIn := 2182,
	HMU_SensorTimes_FixedBufferOut := 2183,
	HMU_SensorTimes_MovingBufferIn := 2184,
	HMU_SensorTimes_MovingBufferOut := 2185,
	HMU_SensorTimes_BufferUpDownIn := 2186,
	HMU_SensorTimes_BufferUpDownOut := 2187,
	HMU_SensorTimes_LockCylinderIn := 2188,
	HMU_SensorTimes_LockCylinderOut := 2189,
	Chain_SensorTimes_Vacuum_1 := 2190,
	Chain_SensorTimes_Vacuum_2 := 2191,
	Chain_SensorTimes_Vacuum_3 := 2192,
	Chain_SensorTimes_Vacuum_4 := 2193,
	Chain_SensorTimes_ExtendIn := 2194,
	Chain_SensorTimes_ExtendOut := 2195,
	Z2Unit_SensorTimes_Vacuum_1 := 2196,
	Z2Unit_SensorTimes_Vacuum_2 := 2197,
	Z2Unit_SensorTimes_Vacuum_3 := 2198,
	Z2Unit_SensorTimes_Vacuum_4 := 2199,
	Z2Unit_SensorTimes_RejectVacuum_1 := 2200,
	Z2Unit_SensorTimes_RejectVacuum_2 := 2201,
	Z2Unit_SensorTimes_RejectVacuum_3 := 2202,
	Z2Unit_SensorTimes_RejectVacuum_4 := 2203,
	Magazine_Time_Idle := 2204,
	HMU_Time_Idle := 2205,
	Z1Unit_Time_Idle := 2206,
	PrUnit_Time_Idle := 2207,
	Z2Unit_Time_Idle := 2208,
	LUnit_L1_Time_Idle := 2209,
	LUnit_L2_Time_Idle := 2210,
	LUnit_L3_Time_Idle := 2211,
	LUnit_L4_Time_Idle := 2212,
	Conveyors_C1_Time_Idle := 2213,
	Conveyors_C2_Time_Idle := 2214,
	Conveyors_C3_Time_Idle := 2215,
	Conveyors_C4_Time_Idle := 2216,
	Magazine_Time_Active := 2217,
	HMU_Time_Active := 2218,
	Z1Unit_Time_Active := 2219,
	PrUnit_Time_Active := 2220,
	Z2Unit_Time_Active := 2221,
	LUnit_L1_Time_Active := 2222,
	LUnit_L2_Time_Active := 2223,
	LUnit_L3_Time_Active := 2224,
	LUnit_L4_Time_Active := 2225,
	Conveyors_C1_Time_Active := 2226,
	Conveyors_C2_Time_Active := 2227,
	Conveyors_C3_Time_Active := 2228,
	Conveyors_C4_Time_Active := 2229,
	Conveyors_C2_Alarms := 2230,
	Conveyors_C3_Alarms := 2231,
	Conveyors_C4_Alarms := 2232,
	LUnit_L2_Alarms := 2233,
	LUnit_L3_Alarms := 2234,
	LUnit_L4_Alarms := 2235,
	Productioncounters_Total_CratesProduced := 2236,
	Productioncounters_Total_ReceivedPatterns := 2237,
	Productioncounters_Total_ReceivedPackablePatterns := 2238,
	Productioncounters_Total_PacksPlacedInCrate := 2239,
	Productioncounters_Total_PacksSealed := 2240,
	Productioncounters_Total_StacksPlacedInPusher := 2241,
	DrawerMagazine_Alarms := 2242,
	Main_BSF_EnableSealbar := 2243,
	Illig_EnablePlaceNewPattern := 2244,
	Illig_EnablePlaceNewPatternBusy := 2245,
	Illig_PackablePatternPlaced := 2246,
	Illig_RequestPlaceNewPattern := 2247,
	Relays_MainAirValve2 := 2248,
	Relays_MainAirValveCrate1 := 2249,
	Relays_MainAirValveCrate2 := 2250,
	Relays_SafetyGateCrate1 := 2251,
	Relays_SafetyGateCrate2 := 2252,
	InfeedConveyor_StackTooHighSensor := 2253,
	InfeedConveyor_Alarms := 2256,
	StackUnit_Alarms := 2257,
	Fanuc1_Alarms := 2258,
	Pusher_Alarms := 2259,
	RejectStation_BSF_Alarms := 2260,
	SealUnit_FoilMagazine_Alarms := 2261,
	SealUnit_TransportAndSealBag_Alarms := 2262,
	SealUnit_PrepareAndFillBag_Alarms := 2263,
	SealUnit_Frame_Alarms := 2264,
	CrateUnit_Fanuc2_Alarms := 2265,
	CrateUnit_Crates_Alarms := 2266,
	InfeedConveyor_CoveredDistance := 2267,
	StackUnit_CoveredDistance := 2268,
	Pusher_CoveredDistance := 2269,
	SealUnit_FoilMagazine_CoveredDistance := 2270,
	SealUnit_TransportAndSealBag_Motor1_CoveredDistance := 2271,
	SealUnit_TransportAndSealBag_Motor2_CoveredDistance := 2272,
	SealUnit_PrepareAndFillBag_CoveredDistance := 2273,
	InfeedConveyor_ErrorId := 2274,
	StackUnit_ErrorId := 2275,
	Pusher_ErrorId := 2276,
	SealUnit_FoilMagazine_ErrorId := 2277,
	SealUnit_TransportAndSealBag_Motor1_ErrorId := 2278,
	SealUnit_TransportAndSealBag_Motor2_ErrorId := 2279,
	SealUnit_PrepareAndFillBag_ErrorId := 2280,
	InfeedConveyor_AxisErrorId := 2281,
	StackUnit_AxisErrorId := 2282,
	Pusher_AxisErrorId := 2283,
	SealUnit_FoilMagazine_AxisErrorId := 2284,
	SealUnit_PrepareAndFillBag_AxisErrorId := 2285,
	SealUnit_TransportAndSealBag_Motor1_AxisErrorId := 2286,
	SealUnit_TransportAndSealBag_Motor2_AxisErrorId := 2287,
	InfeedConveyor_DriveErrorId := 2288,
	StackUnit_DriveErrorId := 2289,
	Pusher_DriveErrorId := 2290,
	SealUnit_FoilMagazine_DriveErrorId := 2291,
	SealUnit_PrepareAndFillBag_DriveErrorId := 2292,
	SealUnit_TransportAndSealBag_Main_DriveErrorId := 2293,
	SealUnit_TransportAndSealBag_Motor2_DriveErrorId := 2294,
	SealUnit_TransportAndSealBag_Motor1_DriveErrorId := 2295,
	InfeedConveyor_DriveUtilisation := 2296,
	StackUnit_DriveUtilisation := 2297,
	Pusher_DriveUtilisation := 2298,
	SealUnit_FoilMagazine_DriveUtilisation := 2299,
	SealUnit_PrepareAndFillBag_DriveUtilisation := 2300,
	SealUnit_TransportAndSealBag_Motor1_DriveUtilisation := 2301,
	SealUnit_TransportAndSealBag_Motor2_DriveUtilisation := 2302,
	InfeedConveyor_MotorUtilisation := 2303,
	StackUnit_MotorUtilisation := 2304,
	Pusher_MotorUtilisation := 2305,
	SealUnit_FoilMagazine_MotorUtilisation := 2306,
	SealUnit_PrepareAndFillBag_MotorUtilisation := 2307,
	SealUnit_TransportAndSealBag_Motor1_MotorUtilisation := 2308,
	SealUnit_TransportAndSealBag_Motor2_MotorUtilisation := 2309,
	StackUnit_SensorTimes_StackPlate1In := 2310,
	StackUnit_SensorTimes_StackPlate1Out := 2311,
	StackUnit_SensorTimes_StackPlate2In := 2312,
	StackUnit_SensorTimes_StackPlate2Out := 2313,
	StackUnit_SensorTimes_BufferPlate1In := 2314,
	StackUnit_SensorTimes_BufferPlate1Out := 2315,
	StackUnit_SensorTimes_BufferPlate2In := 2316,
	StackUnit_SensorTimes_BufferPlate2Out := 2317,
	StackUnit_SensorTimes_RejectStackIn := 2318,
	StackUnit_SensorTimes_RejectStackOut := 2319,
	StackUnit_SensorTimes_ShiftStackUnitIn := 2320,
	StackUnit_SensorTimes_ShiftStackUnitOut := 2321,
	Fanuc1_SensorTimes_ClampIn := 2322,
	Fanuc1_SensorTimes_ClampOut := 2323,
	Pusher_SensorTimes_PusherPlateIn := 2324,
	Pusher_SensorTimes_PusherPlateOut := 2325,
	SealUnit_FoilMagazine_FoilRoll1_SensorTimes_ClampFoilOut := 2326,
	SealUnit_FoilMagazine_FoilRoll1_SensorTimes_ClampFoilIn := 2327,
	SealUnit_FoilMagazine_FoilRoll2_SensorTimes_ClampFoilOut := 2328,
	SealUnit_FoilMagazine_FoilRoll2_SensorTimes_ClampFoilIn := 2329,
	SealUnit_FoilMagazine_FoilRoll1_SensorTimes_EnableFoilOut := 2330,
	SealUnit_FoilMagazine_FoilRoll1_SensorTimes_EnableFoilIn := 2331,
	SealUnit_FoilMagazine_FoilRoll2_SensorTimes_EnableFoilOut := 2332,
	SealUnit_FoilMagazine_FoilRoll2_SensorTimes_EnableFoilIn := 2333,
	SealUnit_TransportAndSealBag_SensorTimes_ShiftVacuumBar1In := 2334,
	SealUnit_TransportAndSealBag_SensorTimes_ShiftVacuumBar1Out := 2335,
	SealUnit_TransportAndSealBag_SensorTimes_ShiftVacuumBar2In := 2336,
	SealUnit_TransportAndSealBag_SensorTimes_ShiftVacuumBar2Out := 2337,
	SealUnit_TransportAndSealBag_SensorTimes_ExtendVacuumBarIn := 2338,
	SealUnit_TransportAndSealBag_SensorTimes_ExtendVacuumBarOut := 2339,
	SealUnit_TransportAndSealBag_SensorTimes_ExtendSealBar1In := 2340,
	SealUnit_TransportAndSealBag_SensorTimes_ExtendSealBar1Out := 2341,
	SealUnit_TransportAndSealBag_SensorTimes_ExtendSealBar2In := 2342,
	SealUnit_TransportAndSealBag_SensorTimes_ExtendSealBar2Out := 2343,
	SealUnit_TransportAndSealBag_SensorTimes_KnifeIn := 2344,
	SealUnit_TransportAndSealBag_SensorTimes_KnifeOut := 2345,
	SealUnit_TransportAndSealBag_SensorTimes_LockSealBarIn := 2346,
	SealUnit_TransportAndSealBag_SensorTimes_LockSealBarOut := 2347,
	SealUnit_TransportAndSealBag_SensorTimes_FoldBagSupportIn := 2348,
	SealUnit_TransportAndSealBag_SensorTimes_FoldBagSupportOut := 2349,
	SealUnit_PrepareAndFillBag_SensorTimes_ExtendFormBagIn := 2350,
	SealUnit_PrepareAndFillBag_SensorTimes_ExtendFormBagOut := 2351,
	SealUnit_PrepareAndFillBag_SensorTimes_RotateFormBagIn := 2352,
	SealUnit_PrepareAndFillBag_SensorTimes_RotateFormBagOut := 2353,
	SealUnit_PrepareAndFillBag_SensorTimes_RotateBlowPanelIn := 2354,
	SealUnit_PrepareAndFillBag_SensorTimes_RotateBlowPanelOut := 2355,
	SealUnit_PrepareAndFillBag_SensorTimes_ExtendBlowPanelIn := 2356,
	SealUnit_PrepareAndFillBag_SensorTimes_ExtendBlowPanelOut := 2357,
	SealUnit_PrepareAndFillBag_SensorTimes_RotateVacuumUnitIn := 2358,
	SealUnit_PrepareAndFillBag_SensorTimes_RotateVacuumUnitOut := 2359,
	SealUnit_PrepareAndFillBag_SensorTimes_ExtendVacuumHeadIn := 2360,
	SealUnit_PrepareAndFillBag_SensorTimes_ExtendVacuumHeadOut := 2361,
	SealUnit_PrepareAndFillBag_SensorTimes_FoldUpBagIn := 2362,
	SealUnit_PrepareAndFillBag_SensorTimes_FoldUpBagOut := 2363,
	SealUnit_Frame_SensorTimes_TiltSealUnitIn := 2364,
	SealUnit_Frame_SensorTimes_TiltSealUnitOut := 2365,
	CrateUnit_Fanuc2_SensorTimes_ExtendIn := 2366,
	CrateUnit_Fanuc2_SensorTimes_ExtendOut := 2367,
	CrateUnit_Fanuc2_SensorTimes_ClampIn := 2368,
	CrateUnit_Fanuc2_SensorTimes_ClampOut := 2369,
	CrateUnit_Crates_SensorTimes_GateCrateCoverIn := 2370,
	CrateUnit_Crates_SensorTimes_GateCrateCoverOut := 2371,
	CrateUnit_Crates_Crate1_SensorTimes_LiftIn := 2372,
	CrateUnit_Crates_Crate1_SensorTimes_LiftOut := 2373,
	CrateUnit_Crates_Crate1_SensorTimes_BlockHorizontalIn := 2374,
	CrateUnit_Crates_Crate1_SensorTimes_BlockHorizontalOut := 2375,
	CrateUnit_Crates_Crate1_SensorTimes_BlockVerticalIn := 2376,
	CrateUnit_Crates_Crate1_SensorTimes_BlockVerticalOut := 2377,
	CrateUnit_Crates_Crate2_SensorTimes_LiftIn := 2378,
	CrateUnit_Crates_Crate2_SensorTimes_LiftOut := 2379,
	CrateUnit_Crates_Crate2_SensorTimes_BlockHorizontalIn := 2380,
	CrateUnit_Crates_Crate2_SensorTimes_BlockHorizontalOut := 2381,
	CrateUnit_Crates_Crate2_SensorTimes_BlockVerticalIn := 2382,
	CrateUnit_Crates_Crate2_SensorTimes_BlockVerticalOut := 2383,
	InfeedConveyor_Time_Idle := 2384,
	StackUnit_Time_Idle := 2385,
	Pusher_Time_Idle := 2386,
	SealUnit_FoilMagazine_Time_Idle := 2387,
	Fanuc1_Time_Idle := 2388,
	SealUnit_TransportAndSealBag_Time_Idle := 2389,
	SealUnit_PrepareAndFillBag_Time_Idle := 2390,
	SealUnit_Frame_Time_Idle := 2391,
	CrateUnit_Fanuc2_Time_Idle := 2392,
	CrateUnit_Crates_Time_Idle := 2393,
	InfeedConveyor_Time_Active := 2394,
	StackUnit_Time_Active := 2395,
	Fanuc1_Time_Active := 2396,
	Pusher_Time_Active := 2397,
	SealUnit_TransportAndSealBag_Time_Active := 2398,
	SealUnit_FoilMagazine_Time_Active := 2399,
	SealUnit_PrepareAndFillBag_Time_Active := 2400,
	SealUnit_Frame_Time_Active := 2401,
	CrateUnit_Fanuc2_Time_Active := 2402,
	CrateUnit_Crates_Time_Active := 2403,
	SealUnit_TransportAndSealBag_SealBarActTemperature := 2404,
	SealUnit_TransportAndSealBag_SealBarSetTemperature := 2405,
	SealUnit_TransportAndSealBag_SensorTimes_VacuumFoil := 2406,
	SealUnit_PrepareAndFillBag_SensorTimes_VacuumBag := 2407,
	SealUnit_FoilMagazine_FoilRoll1_UnrolledFoilLength := 2408,
	SealUnit_FoilMagazine_FoilRoll2_UnrolledFoilLength := 2409,
	SealUnit_FoilMagazine_FoilRoll1_TakeFoilFailed := 2410,
	SealUnit_FoilMagazine_FoilRoll2_TakeFoilFailed := 2411,
	SealUnit_FoilMagazine_FoilRoll1_State := 2412,
	SealUnit_FoilMagazine_FoilRoll2_State := 2413,
	SealUnit_FoilMagazine_FoilRoll1_RollSupportMotor1 := 2414,
	SealUnit_FoilMagazine_FoilRoll1_RollSupportMotor2 := 2415,
	SealUnit_FoilMagazine_FoilRoll2_RollSupportMotor1 := 2416,
	SealUnit_FoilMagazine_FoilRoll2_RollSupportMotor2 := 2417,
	CrateUnit_Crates_Crate1_State := 2418,
	CrateUnit_Crates_Crate2_State := 2419,
	CrateUnit_Crates_RecipeName_Crate := 2420,
	RejectStation_RejectCount := 2421,
	SealUnit_TransportAndSealBag_Motor1_Alarms := 2422,
	SealUnit_TransportAndSealBag_Motor2_Alarms := 2423,
	CrateDataProvider_Alarms := 2424,
	Magazine_2_ActiveDrawer := 2425,
	BFU_PickAndPlace_SensorTimes_GuidingIn := 2426,
	BFU_PickAndPlace_SensorTimes_GuidingOut := 2427,
	BFU_PickAndPlace_Messages := 2428,
	ZUnit_SensorTimes_Shift2In := 2429,
	ZUnit_SensorTimes_Shift2Out := 2430,
	Main_DCbusVoltage := 2431,
	Main_DCbusVoltageFiltered := 2432,
	Main_Relays_HighVacuumPump2Running := 2433,
	Relays_RequestForOpeningSafetyGate := 2434,
	Relays_AcknowledgeSafetyGates := 2435,
	Y2Unit_Alarms := 2436,
	Xi2Unit_Alarms := 2437,
	Xu2Unit_Alarms := 2438,
	Magazine_2_Alarms := 2439,
	Magazine_2_M2_1_Alarms := 2440,
	Magazine_2_M2_2_Alarms := 2441,
	SUnit_Alarms := 2442,
	Y3Unit_Alarms := 2443,
	TUnit_Alarms := 2444,
	AUnit_Alarms := 2445,
	BoxFillStation_Alarms := 2446,
	BoxInfeed_Alarms := 2447,
	BoxOutfeed_Alarms := 2448,
	SheetMagazine_Alarms := 2449,
	Upstacker_Alarms := 2450,
	Y2Unit_CoveredDistance := 2451,
	Xi2Unit_CoveredDistance := 2452,
	Xu2Unit_CoveredDistance := 2453,
	Magazine_2_M2_1_CoveredDistance := 2454,
	Magazine_2_M2_2_CoveredDistance := 2455,
	SUnit_CoveredDistance := 2456,
	Y3Unit_CoveredDistance := 2457,
	TUnit_CoveredDistance := 2458,
	AUnit_CoveredDistance := 2459,
	Y2Unit_ErrorId := 2460,
	Xi2Unit_ErrorId := 2461,
	Xu2Unit_ErrorId := 2462,
	Magazine_2_M2_1_ErrorId := 2463,
	Magazine_2_M2_2_ErrorId := 2464,
	SUnit_ErrorId := 2465,
	Y3Unit_ErrorId := 2466,
	TUnit_ErrorId := 2467,
	AUnit_ErrorId := 2468,
	Y2Unit_AxisErrorId := 2469,
	Xi2Unit_AxisErrorId := 2470,
	Xu2Unit_AxisErrorId := 2471,
	Magazine_2_M2_1_AxisErrorId := 2472,
	Magazine_2_M2_2_AxisErrorId := 2473,
	TUnit_AxisErrorId := 2474,
	Y3Unit_AxisErrorId := 2475,
	AUnit_AxisErrorId := 2476,
	SUnit_AxisErrorId := 2477,
	Y2Unit_DriveErrorId := 2478,
	Xi2Unit_DriveErrorId := 2479,
	Xu2Unit_DriveErrorId := 2480,
	Magazine_2_M2_1_DriveErrorId := 2481,
	Magazine_2_M2_2_DriveErrorId := 2482,
	SUnit_DriveErrorId := 2483,
	TUnit_DriveErrorId := 2484,
	Y3Unit_DriveErrorId := 2485,
	AUnit_DriveErrorId := 2486,
	Y2Unit_DriveUtilisation := 2487,
	Xi2Unit_DriveUtilisation := 2488,
	Xu2Unit_DriveUtilisation := 2489,
	Magazine_2_M2_1_DriveUtilisation := 2490,
	Magazine_2_M2_2_DriveUtilisation := 2491,
	SUnit_DriveUtilisation := 2492,
	Y3Unit_DriveUtilisation := 2493,
	TUnit_DriveUtilisation := 2494,
	AUnit_DriveUtilisation := 2495,
	Y2Unit_MotorUtilisation := 2496,
	Xi2Unit_MotorUtilisation := 2497,
	Xu2Unit_MotorUtilisation := 2498,
	Magazine_2_M2_1_MotorUtilisation := 2499,
	Magazine_2_M2_2_MotorUtilisation := 2500,
	TUnit_MotorUtilisation := 2501,
	SUnit_MotorUtilisation := 2502,
	Y3Unit_MotorUtilisation := 2503,
	AUnit_MotorUtilisation := 2504,
	XuUnit_SensorTimes_Vacuum_4 := 2505,
	XuUnit_SensorTimes_Vacuum_5 := 2506,
	XuUnit_SensorTimes_Vacuum_6 := 2507,
	XuUnit_SensorTimes_Vacuum_7 := 2508,
	XuUnit_SensorTimes_Vacuum_8 := 2509,
	XuUnit_SensorTimes_Vacuum_9 := 2510,
	XuUnit_SensorTimes_Vacuum_10 := 2511,
	XuUnit_SensorTimes_Vacuum_11 := 2512,
	XuUnit_SensorTimes_Vacuum_12 := 2513,
	XuUnit_SensorTimes_Vacuum_13 := 2514,
	XuUnit_SensorTimes_Vacuum_14 := 2515,
	XuUnit_SensorTimes_Vacuum_15 := 2516,
	XuUnit_SensorTimes_Vacuum_16 := 2517,
	XuUnit_SensorTimes_Vacuum_17 := 2518,
	XuUnit_SensorTimes_Vacuum_18 := 2519,
	XuUnit_SensorTimes_Vacuum_19 := 2520,
	XuUnit_SensorTimes_Vacuum_20 := 2521,
	XuUnit_SensorTimes_Vacuum_21 := 2522,
	XuUnit_SensorTimes_Vacuum_22 := 2523,
	XuUnit_SensorTimes_Vacuum_23 := 2524,
	XuUnit_SensorTimes_Vacuum_24 := 2525,
	XuUnit_SensorTimes_Vacuum_25 := 2526,
	XuUnit_SensorTimes_Vacuum_26 := 2527,
	XuUnit_SensorTimes_Vacuum_27 := 2528,
	XuUnit_SensorTimes_Vacuum_28 := 2529,
	XuUnit_SensorTimes_Vacuum_29 := 2530,
	XuUnit_SensorTimes_Vacuum_30 := 2531,
	XuUnit_SensorTimes_Vacuum_31 := 2532,
	XuUnit_SensorTimes_Vacuum_32 := 2533,
	Xu2Unit_SensorTimes_Vacuum_1 := 2534,
	Xu2Unit_SensorTimes_Vacuum_2 := 2535,
	Xu2Unit_SensorTimes_Vacuum_3 := 2536,
	Xu2Unit_SensorTimes_Vacuum_4 := 2537,
	Xu2Unit_SensorTimes_Vacuum_5 := 2538,
	Xu2Unit_SensorTimes_Vacuum_6 := 2539,
	Xu2Unit_SensorTimes_Vacuum_7 := 2540,
	Xu2Unit_SensorTimes_Vacuum_8 := 2541,
	Xu2Unit_SensorTimes_Vacuum_9 := 2542,
	Xu2Unit_SensorTimes_Vacuum_10 := 2543,
	Xu2Unit_SensorTimes_Vacuum_11 := 2544,
	Xu2Unit_SensorTimes_Vacuum_12 := 2545,
	Xu2Unit_SensorTimes_Vacuum_13 := 2546,
	Xu2Unit_SensorTimes_Vacuum_14 := 2547,
	Xu2Unit_SensorTimes_Vacuum_15 := 2548,
	Xu2Unit_SensorTimes_Vacuum_16 := 2549,
	Xu2Unit_SensorTimes_Vacuum_17 := 2550,
	Xu2Unit_SensorTimes_Vacuum_18 := 2551,
	Xu2Unit_SensorTimes_Vacuum_19 := 2552,
	Xu2Unit_SensorTimes_Vacuum_20 := 2553,
	Xu2Unit_SensorTimes_Vacuum_21 := 2554,
	Xu2Unit_SensorTimes_Vacuum_22 := 2555,
	Xu2Unit_SensorTimes_Vacuum_23 := 2556,
	Xu2Unit_SensorTimes_Vacuum_24 := 2557,
	Xu2Unit_SensorTimes_Vacuum_25 := 2558,
	Xu2Unit_SensorTimes_Vacuum_26 := 2559,
	Xu2Unit_SensorTimes_Vacuum_27 := 2560,
	Xu2Unit_SensorTimes_Vacuum_28 := 2561,
	Xu2Unit_SensorTimes_Vacuum_29 := 2562,
	Xu2Unit_SensorTimes_Vacuum_30 := 2563,
	Xu2Unit_SensorTimes_Vacuum_31 := 2564,
	Xu2Unit_SensorTimes_Vacuum_32 := 2565,
	Magazine_SensorTimes_Vacuum_9 := 2566,
	Magazine_SensorTimes_Vacuum_10 := 2567,
	Magazine_SensorTimes_Vacuum_11 := 2568,
	Magazine_SensorTimes_Vacuum_12 := 2569,
	Magazine_SensorTimes_Vacuum_13 := 2570,
	Magazine_SensorTimes_Vacuum_14 := 2571,
	Magazine_SensorTimes_Vacuum_15 := 2572,
	Magazine_SensorTimes_Vacuum_16 := 2573,
	Magazine_SensorTimes_Vacuum_17 := 2574,
	Magazine_SensorTimes_Vacuum_18 := 2575,
	Magazine_SensorTimes_Vacuum_19 := 2576,
	Magazine_SensorTimes_Vacuum_20 := 2577,
	Magazine_SensorTimes_Vacuum_21 := 2578,
	Magazine_SensorTimes_Vacuum_22 := 2579,
	Magazine_SensorTimes_Vacuum_23 := 2580,
	Magazine_SensorTimes_Vacuum_24 := 2581,
	Magazine_SensorTimes_Vacuum_25 := 2582,
	Magazine_SensorTimes_Vacuum_26 := 2583,
	Magazine_SensorTimes_Vacuum_27 := 2584,
	Magazine_SensorTimes_Vacuum_28 := 2585,
	Magazine_SensorTimes_Vacuum_29 := 2586,
	Magazine_SensorTimes_Vacuum_30 := 2587,
	Magazine_SensorTimes_Vacuum_31 := 2588,
	Magazine_SensorTimes_Vacuum_32 := 2589,
	Magazine_2_SensorTimes_Vacuum_1 := 2590,
	Magazine_2_SensorTimes_Vacuum_2 := 2591,
	Magazine_2_SensorTimes_Vacuum_3 := 2592,
	Magazine_2_SensorTimes_Vacuum_4 := 2593,
	Magazine_2_SensorTimes_Vacuum_5 := 2594,
	Magazine_2_SensorTimes_Vacuum_6 := 2595,
	Magazine_2_SensorTimes_Vacuum_7 := 2596,
	Magazine_2_SensorTimes_Vacuum_8 := 2597,
	Magazine_2_SensorTimes_Vacuum_9 := 2598,
	Magazine_2_SensorTimes_Vacuum_10 := 2599,
	Magazine_2_SensorTimes_Vacuum_11 := 2600,
	Magazine_2_SensorTimes_Vacuum_12 := 2601,
	Magazine_2_SensorTimes_Vacuum_13 := 2602,
	Magazine_2_SensorTimes_Vacuum_14 := 2603,
	Magazine_2_SensorTimes_Vacuum_15 := 2604,
	Magazine_2_SensorTimes_Vacuum_16 := 2605,
	Magazine_2_SensorTimes_Vacuum_17 := 2606,
	Magazine_2_SensorTimes_Vacuum_18 := 2607,
	Magazine_2_SensorTimes_Vacuum_19 := 2608,
	Magazine_2_SensorTimes_Vacuum_20 := 2609,
	Magazine_2_SensorTimes_Vacuum_22 := 2610,
	Magazine_2_SensorTimes_Vacuum_21 := 2611,
	Magazine_2_SensorTimes_Vacuum_26 := 2612,
	Magazine_2_SensorTimes_Vacuum_23 := 2613,
	Magazine_2_SensorTimes_Vacuum_24 := 2614,
	Magazine_2_SensorTimes_Vacuum_25 := 2615,
	Magazine_2_SensorTimes_Vacuum_27 := 2616,
	Magazine_2_SensorTimes_Vacuum_28 := 2617,
	Magazine_2_SensorTimes_Vacuum_29 := 2618,
	Magazine_2_SensorTimes_Vacuum_30 := 2619,
	Magazine_2_SensorTimes_Vacuum_31 := 2620,
	Magazine_2_SensorTimes_Vacuum_32 := 2621,
	Magazine_2_SensorTimes_ShiftIn := 2622,
	Magazine_2_SensorTimes_ShiftOut := 2623,
	Magazine_2_SensorTimes_ChangeDrawerIn := 2624,
	Magazine_2_SensorTimes_ChangeDrawerOut := 2625,
	Magazine_2_SensorTimes_LockDrawerIn := 2626,
	Magazine_2_SensorTimes_LockDrawerOut := 2627,
	Y3Unit_SensorTimes_ShiftIn := 2628,
	Y3Unit_SensorTimes_ShiftOut := 2629,
	TUnit_SensorTimes_Vacuum_2_2 := 2630,
	TUnit_SensorTimes_Vacuum_1_1 := 2631,
	TUnit_SensorTimes_Vacuum_1_2 := 2632,
	TUnit_SensorTimes_Vacuum_1_3 := 2633,
	TUnit_SensorTimes_Vacuum_1_4 := 2634,
	TUnit_SensorTimes_Vacuum_2_1 := 2635,
	TUnit_SensorTimes_Vacuum_2_3 := 2636,
	TUnit_SensorTimes_Vacuum_2_4 := 2637,
	TUnit_SensorTimes_ExtendIn := 2638,
	TUnit_SensorTimes_ExtendOut := 2639,
	TUnit_SensorTimes_RotateIn := 2640,
	TUnit_SensorTimes_RotateOut := 2641,
	TUnit_SensorTimes_CloseLidIn := 2642,
	TUnit_SensorTimes_CloseLidOut := 2643,
	Upstacker_1_1_SensorTimes_LiftIn := 2644,
	Upstacker_1_1_SensorTimes_LiftOut := 2645,
	Upstacker_1_1_SensorTimes_LowerStackPlateIn := 2646,
	Upstacker_1_1_SensorTimes_LowerStackPlateOut := 2647,
	Upstacker_1_1_SensorTimes_UpperStackPlateOut := 2648,
	Upstacker_1_1_SensorTimes_UpperStackPlateIn := 2649,
	Upstacker_2_1_SensorTimes_LiftIn := 2650,
	Upstacker_2_1_SensorTimes_LiftOut := 2651,
	Upstacker_2_1_SensorTimes_LowerStackPlateIn := 2652,
	Upstacker_2_1_SensorTimes_LowerStackPlateOut := 2653,
	Upstacker_2_1_SensorTimes_UpperStackPlateOut := 2654,
	Upstacker_2_1_SensorTimes_UpperStackPlateIn := 2655,
	Upstacker_3_1_SensorTimes_LiftIn := 2656,
	Upstacker_3_1_SensorTimes_LiftOut := 2657,
	Upstacker_3_1_SensorTimes_LowerStackPlateIn := 2658,
	Upstacker_3_1_SensorTimes_LowerStackPlateOut := 2659,
	Upstacker_3_1_SensorTimes_UpperStackPlateOut := 2660,
	Upstacker_3_1_SensorTimes_UpperStackPlateIn := 2661,
	Upstacker_4_1_SensorTimes_LiftIn := 2662,
	Upstacker_4_1_SensorTimes_LiftOut := 2663,
	Upstacker_4_1_SensorTimes_LowerStackPlateIn := 2664,
	Upstacker_4_1_SensorTimes_LowerStackPlateOut := 2665,
	Upstacker_4_1_SensorTimes_UpperStackPlateOut := 2666,
	Upstacker_4_1_SensorTimes_UpperStackPlateIn := 2667,
	Upstacker_5_1_SensorTimes_LiftIn := 2668,
	Upstacker_5_1_SensorTimes_LiftOut := 2669,
	Upstacker_5_1_SensorTimes_LowerStackPlateIn := 2670,
	Upstacker_5_1_SensorTimes_LowerStackPlateOut := 2671,
	Upstacker_5_1_SensorTimes_UpperStackPlateOut := 2672,
	Upstacker_5_1_SensorTimes_UpperStackPlateIn := 2673,
	Upstacker_6_1_SensorTimes_LiftIn := 2674,
	Upstacker_6_1_SensorTimes_LiftOut := 2675,
	Upstacker_6_1_SensorTimes_LowerStackPlateIn := 2676,
	Upstacker_6_1_SensorTimes_LowerStackPlateOut := 2677,
	Upstacker_6_1_SensorTimes_UpperStackPlateOut := 2678,
	Upstacker_6_1_SensorTimes_UpperStackPlateIn := 2679,
	Upstacker_7_1_SensorTimes_LiftIn := 2680,
	Upstacker_7_1_SensorTimes_LiftOut := 2681,
	Upstacker_7_1_SensorTimes_LowerStackPlateIn := 2682,
	Upstacker_7_1_SensorTimes_LowerStackPlateOut := 2683,
	Upstacker_7_1_SensorTimes_UpperStackPlateOut := 2684,
	Upstacker_7_1_SensorTimes_UpperStackPlateIn := 2685,
	Upstacker_8_1_SensorTimes_LiftIn := 2686,
	Upstacker_8_1_SensorTimes_LiftOut := 2687,
	Upstacker_8_1_SensorTimes_LowerStackPlateIn := 2688,
	Upstacker_8_1_SensorTimes_LowerStackPlateOut := 2689,
	Upstacker_8_1_SensorTimes_UpperStackPlateOut := 2690,
	Upstacker_8_1_SensorTimes_UpperStackPlateIn := 2691,
	Upstacker_1_2_SensorTimes_LiftIn := 2692,
	Upstacker_1_2_SensorTimes_LiftOut := 2693,
	Upstacker_1_2_SensorTimes_LowerStackPlateIn := 2694,
	Upstacker_1_2_SensorTimes_LowerStackPlateOut := 2695,
	Upstacker_1_2_SensorTimes_UpperStackPlateOut := 2696,
	Upstacker_1_2_SensorTimes_UpperStackPlateIn := 2697,
	Upstacker_2_2_SensorTimes_LiftIn := 2698,
	Upstacker_2_2_SensorTimes_LiftOut := 2699,
	Upstacker_2_2_SensorTimes_LowerStackPlateIn := 2700,
	Upstacker_2_2_SensorTimes_LowerStackPlateOut := 2701,
	Upstacker_2_2_SensorTimes_UpperStackPlateOut := 2702,
	Upstacker_2_2_SensorTimes_UpperStackPlateIn := 2703,
	Upstacker_3_2_SensorTimes_LiftIn := 2704,
	Upstacker_3_2_SensorTimes_LiftOut := 2705,
	Upstacker_3_2_SensorTimes_LowerStackPlateIn := 2706,
	Upstacker_3_2_SensorTimes_LowerStackPlateOut := 2707,
	Upstacker_3_2_SensorTimes_UpperStackPlateOut := 2708,
	Upstacker_3_2_SensorTimes_UpperStackPlateIn := 2709,
	Upstacker_4_2_SensorTimes_LiftIn := 2710,
	Upstacker_4_2_SensorTimes_LiftOut := 2711,
	Upstacker_4_2_SensorTimes_LowerStackPlateIn := 2712,
	Upstacker_4_2_SensorTimes_LowerStackPlateOut := 2713,
	Upstacker_4_2_SensorTimes_UpperStackPlateOut := 2714,
	Upstacker_4_2_SensorTimes_UpperStackPlateIn := 2715,
	Upstacker_5_2_SensorTimes_LiftIn := 2716,
	Upstacker_5_2_SensorTimes_LiftOut := 2717,
	Upstacker_5_2_SensorTimes_LowerStackPlateIn := 2718,
	Upstacker_5_2_SensorTimes_LowerStackPlateOut := 2719,
	Upstacker_5_2_SensorTimes_UpperStackPlateOut := 2720,
	Upstacker_5_2_SensorTimes_UpperStackPlateIn := 2721,
	Upstacker_6_2_SensorTimes_LiftIn := 2722,
	Upstacker_6_2_SensorTimes_LiftOut := 2723,
	Upstacker_6_2_SensorTimes_LowerStackPlateIn := 2724,
	Upstacker_6_2_SensorTimes_LowerStackPlateOut := 2725,
	Upstacker_6_2_SensorTimes_UpperStackPlateOut := 2726,
	Upstacker_6_2_SensorTimes_UpperStackPlateIn := 2727,
	Upstacker_7_2_SensorTimes_LiftIn := 2728,
	Upstacker_7_2_SensorTimes_LiftOut := 2729,
	Upstacker_7_2_SensorTimes_LowerStackPlateIn := 2730,
	Upstacker_7_2_SensorTimes_LowerStackPlateOut := 2731,
	Upstacker_7_2_SensorTimes_UpperStackPlateOut := 2732,
	Upstacker_7_2_SensorTimes_UpperStackPlateIn := 2733,
	Upstacker_8_2_SensorTimes_LiftIn := 2734,
	Upstacker_8_2_SensorTimes_LiftOut := 2735,
	Upstacker_8_2_SensorTimes_LowerStackPlateIn := 2736,
	Upstacker_8_2_SensorTimes_LowerStackPlateOut := 2737,
	Upstacker_8_2_SensorTimes_UpperStackPlateOut := 2738,
	Upstacker_8_2_SensorTimes_UpperStackPlateIn := 2739,
	Fanuc_SensorTimes_ClampLongSideIn := 2740,
	Fanuc_SensorTimes_ClampLongSideOut := 2741,
	Fanuc_SensorTimes_ClampShortSideIn := 2742,
	Fanuc_SensorTimes_ClampShortSideOut := 2743,
	Patternizer_SensorTimes_ClampStack1In := 2744,
	Patternizer_SensorTimes_ClampStack2In := 2745,
	Patternizer_SensorTimes_ClampStack3In := 2746,
	Patternizer_SensorTimes_ClampStack4In := 2747,
	Patternizer_SensorTimes_ClampStack1Out := 2748,
	Patternizer_SensorTimes_ClampStack2Out := 2749,
	Patternizer_SensorTimes_ClampStack3Out := 2750,
	Patternizer_SensorTimes_ClampStack4Out := 2751,
	Gripper_SensorTimes_ExtendIn := 2752,
	Gripper_SensorTimes_ExtendOut := 2753,
	Gripper_SensorTimes_PusherIn := 2754,
	Gripper_SensorTimes_PusherOut := 2755,
	Gripper_SensorTimes_ClampStack10mmIn := 2756,
	Gripper_SensorTimes_ClampStack10mmOut := 2757,
	Gripper_SensorTimes_ClampStack20mmIn := 2758,
	Gripper_SensorTimes_ClampStack20mmOut := 2759,
	Gripper_SensorTimes_ClampStackLongSideIn := 2760,
	Gripper_SensorTimes_ClampStackLongSideOut := 2761,
	Gripper_SensorTimes_Vacuum := 2762,
	SheetMagazine_SensorTimes_SlidingPanelIn := 2763,
	ExtendOut1_dontUse1 := 2764,
	ExtendOut1_dontUse := 2765,
	SheetMagazine_SensorTimes_SlidingPanelOut := 2766,
	BoxInfeed_SensorTimes_ClampSecondBoxIn := 2767,
	BoxInfeed_SensorTimes_ClampSecondBoxOut := 2768,
	BoxInfeed_SensorTimes_PusherOut := 2769,
	BoxInfeed_SensorTimes_PusherIn := 2770,
	BoxFillStation_SensorTimes_OpenBoxSide1In := 2771,
	BoxFillStation_SensorTimes_OpenBoxSide1Out := 2772,
	BoxFillStation_SensorTimes_OpenBoxSide2In := 2773,
	BoxFillStation_SensorTimes_OpenBoxSide2Out := 2774,
	BoxFillStation_SensorTimes_OpenBoxSide3In := 2775,
	BoxFillStation_SensorTimes_OpenBoxSide3Out := 2776,
	BoxFillStation_SensorTimes_OpenBoxSide4In := 2777,
	BoxFillStation_SensorTimes_OpenBoxSide4Out := 2778,
	Y2Unit_Time_Idle := 2779,
	Y3Unit_Time_Idle := 2780,
	Xi2Unit_Time_Idle := 2781,
	Xu2Unit_Time_Idle := 2782,
	Magazine_2_Time_Idle := 2783,
	SUnit_Time_Idle := 2784,
	TUnit_Time_Idle := 2785,
	AUnit_Time_Idle := 2786,
	Upstacker_1_1_Time_Idle := 2787,
	Upstacker_2_1_Time_Idle := 2788,
	Upstacker_3_1_Time_Idle := 2789,
	Upstacker_4_1_Time_Idle := 2790,
	Upstacker_5_1_Time_Idle := 2791,
	Upstacker_6_1_Time_Idle := 2792,
	Upstacker_7_1_Time_Idle := 2793,
	Upstacker_8_1_Time_Idle := 2794,
	Upstacker_1_2_Time_Idle := 2795,
	Upstacker_2_2_Time_Idle := 2796,
	Upstacker_3_2_Time_Idle := 2797,
	Upstacker_4_2_Time_Idle := 2798,
	Upstacker_5_2_Time_Idle := 2799,
	Upstacker_6_2_Time_Idle := 2800,
	Upstacker_7_2_Time_Idle := 2801,
	Upstacker_8_2_Time_Idle := 2802,
	Fanuc_Time_Idle := 2803,
	Patternizer_Time_Idle := 2804,
	Gripper_Time_Idle := 2805,
	BFU_YUnit_Time_Idle := 2806,
	SheetMagazine_Time_Idle := 2807,
	BoxInfeed_Time_Idle := 2808,
	BoxFillStation_Time_Idle := 2809,
	BoxOutfeed_Time_Idle := 2810,
	PickProductsFromUpstacker_Time_Idle := 2811,
	PlaceProductsOnPatternizer_Time_Idle := 2812,
	RejectProducts_Time_Idle := 2813,
	PickPlaceProducts_Time_Idle := 2814,
	PickPlaceY_Time_Idle := 2815,
	PickPlaceSheets_Time_Idle := 2816,
	SheetRefilling_Time_Idle := 2817,
	BoxFilling_Time_Idle := 2818,
	BoxTransport_Time_Idle := 2819,
	Y2Unit_Time_Active := 2820,
	Xi2Unit_Time_Active := 2821,
	Magazine_2_Time_Active := 2822,
	Xu2Unit_Time_Active := 2823,
	SUnit_Time_Active := 2824,
	Y3Unit_Time_Active := 2825,
	TUnit_Time_Active := 2826,
	AUnit_Time_Active := 2827,
	BoxFillStation_Time_Active := 2828,
	BoxInfeed_Time_Active := 2829,
	BoxOutfeed_Time_Active := 2830,
	SheetMagazine_Time_Active := 2831,
	Upstacker_1_1_Time_Active := 2832,
	Upstacker_2_1_Time_Active := 2833,
	Upstacker_3_1_Time_Active := 2834,
	Upstacker_4_1_Time_Active := 2835,
	Upstacker_5_1_Time_Active := 2836,
	Upstacker_6_1_Time_Active := 2837,
	Upstacker_7_1_Time_Active := 2838,
	Upstacker_8_1_Time_Active := 2839,
	Upstacker_1_2_Time_Active := 2840,
	Upstacker_2_2_Time_Active := 2841,
	Upstacker_3_2_Time_Active := 2842,
	Upstacker_4_2_Time_Active := 2843,
	Upstacker_5_2_Time_Active := 2844,
	Upstacker_6_2_Time_Active := 2845,
	Upstacker_7_2_Time_Active := 2846,
	Upstacker_8_2_Time_Active := 2847,
	Fanuc_Time_Active := 2848,
	Patternizer_Time_Active := 2849,
	Gripper_Time_Active := 2850,
	BFU_YUnit_Time_Active := 2851,
	PickProductsFromUpstacker_Time_Active := 2852,
	PlaceProductsOnPatternizer_Time_Active := 2853,
	RejectProducts_Time_Active := 2854,
	PickPlaceProducts_Time_Active := 2855,
	PickPlaceY_Time_Active := 2856,
	PickPlaceSheets_Time_Active := 2857,
	SheetRefilling_Time_Active := 2858,
	BoxFilling_Time_Active := 2859,
	BoxTransport_Time_Active := 2860,
	DrawerMagazine_2_Alarms := 2861,
	XUnit_Alarms := 2862,
	BFU_Turner_Alarms := 2863,
	XUnit_BFU_Alarms := 2864,
	Conveyors_BFU_Alarms := 2865,
	XUnit_CoveredDistance := 2866,
	ZrUnit_Zr1_CoveredDistance := 2867,
	XUnit_BFU_CoveredDistance := 2868,
	XUnit_ErrorID := 2869,
	ZrUnit_Zr1_ErrorID := 2870,
	XUnit_BFU_ErrorID := 2871,
	XUnit_AxisErrorId := 2872,
	XUnit_BFU_AxisErrorId := 2873,
	XUnit_DriveErrorId := 2874,
	XUnit_BFU_DriveErrorId := 2875,
	XUnit_DriveUtilisation := 2876,
	ZrUnit_Zr1_DriveUtilisation := 2877,
	XUnit_BFU_DriveUtilisation := 2878,
	XUnit_MotorUtilisation := 2879,
	ZrUnit_Zr1_MotorUtilisation := 2880,
	XUnit_BFU_MotorUtilisation := 2881,
	XUnit_SensorTimes_VacuumLid_1 := 2882,
	XUnit_SensorTimes_VacuumLid_2 := 2883,
	XUnit_SensorTimes_VacuumScoop_1 := 2884,
	XUnit_SensorTimes_VacuumScoop_2 := 2885,
	XUnit_SensorTimes_RotateScoopIn := 2886,
	XUnit_SensorTimes_RotateScoopOut := 2887,
	XUnit_SensorTimes_ClampLidIn_1 := 2888,
	XUnit_SensorTimes_ClampLidIn_2 := 2889,
	TXUnit_Alarms := 2890,
	TXUnit_CoveredDistance := 2891,
	TXUnit_ErrorID := 2892,
	TXUnit_AxisErrorId := 2893,
	TXUnit_DriveErrorId := 2894,
	TXUnit_DriveUtilisation := 2895,
	TXUnit_MotorUtilisation := 2896,
	ZUnit_SensorTimes_CloseLidIn := 2897,
	ZUnit_SensorTimes_CloseLidOut := 2898,
	ZUnit_SensorTimes_FlipCapIn := 2899,
	ZUnit_SensorTimes_FlipCapOut := 2900,
	TXUnit_SensorTimes_LiftIn_1 := 2901,
	TXUnit_SensorTimes_LiftIn_2 := 2902,
	TXUnit_SensorTimes_LiftIn_3 := 2903,
	TXUnit_SensorTimes_LiftOut_1 := 2904,
	TXUnit_SensorTimes_LiftOut_2 := 2905,
	TXUnit_SensorTimes_LiftOut_3 := 2906,
	TXUnit_SensorTimes_ExtendIn := 2907,
	TXUnit_SensorTimes_ExtendOut := 2908,
	ZUnit_SensorTimes_LockZrIn := 2909,
	ZUnit_SensorTimes_LockZrOut := 2910,
	BFU_PickAndPlace_SensorTimes_Vacuum_1 := 2911,
	BFU_PickAndPlace_SensorTimes_Shift := 2912,
	BFU_PickAndPlace_SensorTimes_ShiftCenterIn := 2913,
	BFU_PickAndPlace_SensorTimes_ShiftCenterOut := 2914,
	BoxConveyor_SensorTimes_ClampBoxIn := 2915,
	BoxConveyor_SensorTimes_ClampBoxOut := 2916,
	BoxConveyor_SensorTimes_VacuumPusher := 2917,
	BoxConveyor_SensorTimes_PusherInfeedIn := 2918,
	BoxConveyor_SensorTimes_PusherInfeedOut := 2919,
	BoxConveyor_SensorTimes_PusherOutfeedIn := 2920,
	BoxConveyor_SensorTimes_PusherOutfeedOut := 2921,
	Turner_BFU_SensorTimes_Vacuum := 2922,
	Turner_BFU_SensorTimes_RotateIn := 2923,
	Turner_BFU_SensorTimes_RotateOut := 2924,
	BoxConveyor_SensorTimes_BoxCenterIn := 2925,
	BoxConveyor_SensorTimes_BoxCenterOut := 2926,
	XUnit_Time_Idle := 2927,
	Camera_YUnit_Time_Idle := 2928,
	ZrUnit_Zr1_Time_Idle := 2929,
	BFU_PickAndPlace_Time_Idle := 2930,
	Turner_BFU_Time_Idle := 2931,
	BoxConveyor_Time_Idle := 2932,
	XUnit_Time_Active := 2933,
	Camera_YUnit_Time_Active := 2934,
	ZrUnit_Zr1_Time_Active := 2935,
	BFU_PickAndPlace_Time_Active := 2936,
	Turner_BFU_Time_Active := 2937,
	BoxConveyor_Time_Active := 2938,
	Conveyors_CoveredDistance := 2939,
	Conveyors_ErrorId := 2940,
	Conveyors_AxisErrorId := 2941,
	Conveyors_DriveErrorId := 2942,
	Conveyors_DriveUtilisation := 2943,
	Conveyors_MotorUtilisation := 2944,
	Main_StepByStepActive := 2945,
	LabelAdjustment_Magazine_Drawer_1_Cassette_1_Position_1 := 2947,
	LabelAdjustment_Magazine_Drawer_1_Cassette_1_Position_2 := 2948,
	LabelAdjustment_Magazine_Drawer_1_Cassette_1_Position_3 := 2949,
	LabelAdjustment_Magazine_Drawer_1_Cassette_2_Position_1 := 2950,
	LabelAdjustment_Magazine_Drawer_1_Cassette_2_Position_2 := 2951,
	LabelAdjustment_Magazine_Drawer_1_Cassette_2_Position_3 := 2952,
	LabelAdjustment_Magazine_Drawer_1_Cassette_3_Position_1 := 2953,
	LabelAdjustment_Magazine_Drawer_1_Cassette_3_Position_2 := 2954,
	LabelAdjustment_Magazine_Drawer_1_Cassette_3_Position_3 := 2955,
	LabelAdjustment_Magazine_Drawer_1_Cassette_4_Position_1 := 2956,
	LabelAdjustment_Magazine_Drawer_1_Cassette_4_Position_2 := 2957,
	LabelAdjustment_Magazine_Drawer_1_Cassette_4_Position_3 := 2958,
	LabelAdjustment_Magazine_Drawer_1_Cassette_5_Position_1 := 2959,
	LabelAdjustment_Magazine_Drawer_1_Cassette_5_Position_2 := 2960,
	LabelAdjustment_Magazine_Drawer_1_Cassette_5_Position_3 := 2961,
	LabelAdjustment_Magazine_Drawer_1_Cassette_6_Position_1 := 2962,
	LabelAdjustment_Magazine_Drawer_1_Cassette_6_Position_2 := 2963,
	LabelAdjustment_Magazine_Drawer_1_Cassette_6_Position_3 := 2964,
	LabelAdjustment_Magazine_Drawer_1_Cassette_7_Position_1 := 2965,
	LabelAdjustment_Magazine_Drawer_1_Cassette_7_Position_2 := 2966,
	LabelAdjustment_Magazine_Drawer_1_Cassette_7_Position_3 := 2967,
	LabelAdjustment_Magazine_Drawer_1_Cassette_8_Position_1 := 2968,
	LabelAdjustment_Magazine_Drawer_1_Cassette_8_Position_2 := 2969,
	LabelAdjustment_Magazine_Drawer_1_Cassette_8_Position_3 := 2970,
	LabelAdjustment_Magazine_Drawer_1_Cassette_9_Position_1 := 2971,
	LabelAdjustment_Magazine_Drawer_1_Cassette_9_Position_2 := 2972,
	LabelAdjustment_Magazine_Drawer_1_Cassette_9_Position_3 := 2973,
	LabelAdjustment_Magazine_Drawer_1_Cassette_10_Position_1 := 2974,
	LabelAdjustment_Magazine_Drawer_1_Cassette_10_Position_2 := 2975,
	LabelAdjustment_Magazine_Drawer_1_Cassette_10_Position_3 := 2976,
	LabelAdjustment_Magazine_Drawer_1_Cassette_11_Position_1 := 2977,
	LabelAdjustment_Magazine_Drawer_1_Cassette_11_Position_2 := 2978,
	LabelAdjustment_Magazine_Drawer_1_Cassette_11_Position_3 := 2979,
	LabelAdjustment_Magazine_Drawer_1_Cassette_12_Position_1 := 2980,
	LabelAdjustment_Magazine_Drawer_1_Cassette_12_Position_2 := 2981,
	LabelAdjustment_Magazine_Drawer_1_Cassette_12_Position_3 := 2982,
	LabelAdjustment_Magazine_Drawer_1_Cassette_13_Position_1 := 2983,
	LabelAdjustment_Magazine_Drawer_1_Cassette_13_Position_2 := 2984,
	LabelAdjustment_Magazine_Drawer_1_Cassette_13_Position_3 := 2985,
	LabelAdjustment_Magazine_Drawer_1_Cassette_14_Position_1 := 2986,
	LabelAdjustment_Magazine_Drawer_1_Cassette_14_Position_2 := 2987,
	LabelAdjustment_Magazine_Drawer_1_Cassette_14_Position_3 := 2988,
	LabelAdjustment_Magazine_Drawer_1_Cassette_15_Position_1 := 2989,
	LabelAdjustment_Magazine_Drawer_1_Cassette_15_Position_2 := 2990,
	LabelAdjustment_Magazine_Drawer_1_Cassette_15_Position_3 := 2991,
	LabelAdjustment_Magazine_Drawer_1_Cassette_16_Position_1 := 2992,
	LabelAdjustment_Magazine_Drawer_1_Cassette_16_Position_2 := 2993,
	LabelAdjustment_Magazine_Drawer_1_Cassette_16_Position_3 := 2994,
	LabelAdjustment_Magazine_Drawer_1_Cassette_17_Position_1 := 2995,
	LabelAdjustment_Magazine_Drawer_1_Cassette_17_Position_2 := 2996,
	LabelAdjustment_Magazine_Drawer_1_Cassette_17_Position_3 := 2997,
	LabelAdjustment_Magazine_Drawer_1_Cassette_18_Position_1 := 2998,
	LabelAdjustment_Magazine_Drawer_1_Cassette_18_Position_2 := 2999,
	LabelAdjustment_Magazine_Drawer_1_Cassette_18_Position_3 := 3000,
	LabelAdjustment_Magazine_Drawer_1_Cassette_19_Position_1 := 3001,
	LabelAdjustment_Magazine_Drawer_1_Cassette_19_Position_2 := 3002,
	LabelAdjustment_Magazine_Drawer_1_Cassette_19_Position_3 := 3003,
	LabelAdjustment_Magazine_Drawer_1_Cassette_20_Position_1 := 3004,
	LabelAdjustment_Magazine_Drawer_1_Cassette_20_Position_2 := 3005,
	LabelAdjustment_Magazine_Drawer_1_Cassette_20_Position_3 := 3006,
	LabelAdjustment_Magazine_Drawer_1_Cassette_21_Position_1 := 3007,
	LabelAdjustment_Magazine_Drawer_1_Cassette_21_Position_2 := 3008,
	LabelAdjustment_Magazine_Drawer_1_Cassette_21_Position_3 := 3009,
	LabelAdjustment_Magazine_Drawer_1_Cassette_22_Position_1 := 3010,
	LabelAdjustment_Magazine_Drawer_1_Cassette_22_Position_2 := 3011,
	LabelAdjustment_Magazine_Drawer_1_Cassette_22_Position_3 := 3012,
	LabelAdjustment_Magazine_Drawer_1_Cassette_23_Position_1 := 3013,
	LabelAdjustment_Magazine_Drawer_1_Cassette_23_Position_2 := 3014,
	LabelAdjustment_Magazine_Drawer_1_Cassette_23_Position_3 := 3015,
	LabelAdjustment_Magazine_Drawer_1_Cassette_24_Position_1 := 3016,
	LabelAdjustment_Magazine_Drawer_1_Cassette_24_Position_2 := 3017,
	LabelAdjustment_Magazine_Drawer_1_Cassette_24_Position_3 := 3018,
	LabelAdjustment_Magazine_Drawer_1_Cassette_25_Position_1 := 3019,
	LabelAdjustment_Magazine_Drawer_1_Cassette_25_Position_2 := 3020,
	LabelAdjustment_Magazine_Drawer_1_Cassette_25_Position_3 := 3021,
	LabelAdjustment_Magazine_Drawer_1_Cassette_26_Position_1 := 3022,
	LabelAdjustment_Magazine_Drawer_1_Cassette_26_Position_2 := 3023,
	LabelAdjustment_Magazine_Drawer_1_Cassette_26_Position_3 := 3024,
	LabelAdjustment_Magazine_Drawer_1_Cassette_27_Position_1 := 3025,
	LabelAdjustment_Magazine_Drawer_1_Cassette_27_Position_2 := 3026,
	LabelAdjustment_Magazine_Drawer_1_Cassette_27_Position_3 := 3027,
	LabelAdjustment_Magazine_Drawer_1_Cassette_28_Position_1 := 3028,
	LabelAdjustment_Magazine_Drawer_1_Cassette_28_Position_2 := 3029,
	LabelAdjustment_Magazine_Drawer_1_Cassette_28_Position_3 := 3030,
	LabelAdjustment_Magazine_Drawer_1_Cassette_29_Position_1 := 3031,
	LabelAdjustment_Magazine_Drawer_1_Cassette_29_Position_2 := 3032,
	LabelAdjustment_Magazine_Drawer_1_Cassette_29_Position_3 := 3033,
	LabelAdjustment_Magazine_Drawer_1_Cassette_30_Position_1 := 3034,
	LabelAdjustment_Magazine_Drawer_1_Cassette_30_Position_2 := 3035,
	LabelAdjustment_Magazine_Drawer_1_Cassette_30_Position_3 := 3036,
	LabelAdjustment_Magazine_Drawer_1_Cassette_31_Position_1 := 3037,
	LabelAdjustment_Magazine_Drawer_1_Cassette_31_Position_2 := 3038,
	LabelAdjustment_Magazine_Drawer_1_Cassette_31_Position_3 := 3039,
	LabelAdjustment_Magazine_Drawer_1_Cassette_32_Position_1 := 3040,
	LabelAdjustment_Magazine_Drawer_1_Cassette_32_Position_2 := 3041,
	LabelAdjustment_Magazine_Drawer_1_Cassette_32_Position_3 := 3042,
	LabelAdjustment_Magazine_Drawer_2_Cassette_1_Position_1 := 3043,
	LabelAdjustment_Magazine_Drawer_2_Cassette_1_Position_2 := 3044,
	LabelAdjustment_Magazine_Drawer_2_Cassette_1_Position_3 := 3045,
	LabelAdjustment_Magazine_Drawer_2_Cassette_2_Position_1 := 3046,
	LabelAdjustment_Magazine_Drawer_2_Cassette_2_Position_2 := 3047,
	LabelAdjustment_Magazine_Drawer_2_Cassette_2_Position_3 := 3048,
	LabelAdjustment_Magazine_Drawer_2_Cassette_3_Position_1 := 3049,
	LabelAdjustment_Magazine_Drawer_2_Cassette_3_Position_2 := 3050,
	LabelAdjustment_Magazine_Drawer_2_Cassette_3_Position_3 := 3051,
	LabelAdjustment_Magazine_Drawer_2_Cassette_4_Position_1 := 3052,
	LabelAdjustment_Magazine_Drawer_2_Cassette_4_Position_2 := 3053,
	LabelAdjustment_Magazine_Drawer_2_Cassette_4_Position_3 := 3054,
	LabelAdjustment_Magazine_Drawer_2_Cassette_5_Position_1 := 3055,
	LabelAdjustment_Magazine_Drawer_2_Cassette_5_Position_2 := 3056,
	LabelAdjustment_Magazine_Drawer_2_Cassette_5_Position_3 := 3057,
	LabelAdjustment_Magazine_Drawer_2_Cassette_6_Position_1 := 3058,
	LabelAdjustment_Magazine_Drawer_2_Cassette_6_Position_2 := 3059,
	LabelAdjustment_Magazine_Drawer_2_Cassette_6_Position_3 := 3060,
	LabelAdjustment_Magazine_Drawer_2_Cassette_7_Position_1 := 3061,
	LabelAdjustment_Magazine_Drawer_2_Cassette_7_Position_2 := 3062,
	LabelAdjustment_Magazine_Drawer_2_Cassette_7_Position_3 := 3063,
	LabelAdjustment_Magazine_Drawer_2_Cassette_8_Position_1 := 3064,
	LabelAdjustment_Magazine_Drawer_2_Cassette_8_Position_2 := 3065,
	LabelAdjustment_Magazine_Drawer_2_Cassette_8_Position_3 := 3066,
	LabelAdjustment_Magazine_Drawer_2_Cassette_9_Position_1 := 3067,
	LabelAdjustment_Magazine_Drawer_2_Cassette_9_Position_2 := 3068,
	LabelAdjustment_Magazine_Drawer_2_Cassette_9_Position_3 := 3069,
	LabelAdjustment_Magazine_Drawer_2_Cassette_10_Position_1 := 3070,
	LabelAdjustment_Magazine_Drawer_2_Cassette_10_Position_2 := 3071,
	LabelAdjustment_Magazine_Drawer_2_Cassette_10_Position_3 := 3072,
	LabelAdjustment_Magazine_Drawer_2_Cassette_11_Position_1 := 3073,
	LabelAdjustment_Magazine_Drawer_2_Cassette_11_Position_2 := 3074,
	LabelAdjustment_Magazine_Drawer_2_Cassette_11_Position_3 := 3075,
	LabelAdjustment_Magazine_Drawer_2_Cassette_12_Position_1 := 3076,
	LabelAdjustment_Magazine_Drawer_2_Cassette_12_Position_2 := 3077,
	LabelAdjustment_Magazine_Drawer_2_Cassette_12_Position_3 := 3078,
	LabelAdjustment_Magazine_Drawer_2_Cassette_13_Position_1 := 3079,
	LabelAdjustment_Magazine_Drawer_2_Cassette_13_Position_2 := 3080,
	LabelAdjustment_Magazine_Drawer_2_Cassette_13_Position_3 := 3081,
	LabelAdjustment_Magazine_Drawer_2_Cassette_14_Position_1 := 3082,
	LabelAdjustment_Magazine_Drawer_2_Cassette_14_Position_2 := 3083,
	LabelAdjustment_Magazine_Drawer_2_Cassette_14_Position_3 := 3084,
	LabelAdjustment_Magazine_Drawer_2_Cassette_15_Position_1 := 3085,
	LabelAdjustment_Magazine_Drawer_2_Cassette_15_Position_2 := 3086,
	LabelAdjustment_Magazine_Drawer_2_Cassette_15_Position_3 := 3087,
	LabelAdjustment_Magazine_Drawer_2_Cassette_16_Position_1 := 3088,
	LabelAdjustment_Magazine_Drawer_2_Cassette_16_Position_2 := 3089,
	LabelAdjustment_Magazine_Drawer_2_Cassette_16_Position_3 := 3090,
	LabelAdjustment_Magazine_Drawer_2_Cassette_17_Position_1 := 3091,
	LabelAdjustment_Magazine_Drawer_2_Cassette_17_Position_2 := 3092,
	LabelAdjustment_Magazine_Drawer_2_Cassette_17_Position_3 := 3093,
	LabelAdjustment_Magazine_Drawer_2_Cassette_18_Position_1 := 3094,
	LabelAdjustment_Magazine_Drawer_2_Cassette_18_Position_2 := 3095,
	LabelAdjustment_Magazine_Drawer_2_Cassette_18_Position_3 := 3096,
	LabelAdjustment_Magazine_Drawer_2_Cassette_19_Position_1 := 3097,
	LabelAdjustment_Magazine_Drawer_2_Cassette_19_Position_2 := 3098,
	LabelAdjustment_Magazine_Drawer_2_Cassette_19_Position_3 := 3099,
	LabelAdjustment_Magazine_Drawer_2_Cassette_20_Position_1 := 3100,
	LabelAdjustment_Magazine_Drawer_2_Cassette_20_Position_2 := 3101,
	LabelAdjustment_Magazine_Drawer_2_Cassette_20_Position_3 := 3102,
	LabelAdjustment_Magazine_Drawer_2_Cassette_21_Position_1 := 3103,
	LabelAdjustment_Magazine_Drawer_2_Cassette_21_Position_2 := 3104,
	LabelAdjustment_Magazine_Drawer_2_Cassette_21_Position_3 := 3105,
	LabelAdjustment_Magazine_Drawer_2_Cassette_22_Position_1 := 3106,
	LabelAdjustment_Magazine_Drawer_2_Cassette_22_Position_2 := 3107,
	LabelAdjustment_Magazine_Drawer_2_Cassette_22_Position_3 := 3108,
	LabelAdjustment_Magazine_Drawer_2_Cassette_23_Position_1 := 3109,
	LabelAdjustment_Magazine_Drawer_2_Cassette_23_Position_2 := 3110,
	LabelAdjustment_Magazine_Drawer_2_Cassette_23_Position_3 := 3111,
	LabelAdjustment_Magazine_Drawer_2_Cassette_24_Position_1 := 3112,
	LabelAdjustment_Magazine_Drawer_2_Cassette_24_Position_2 := 3113,
	LabelAdjustment_Magazine_Drawer_2_Cassette_24_Position_3 := 3114,
	LabelAdjustment_Magazine_Drawer_2_Cassette_25_Position_1 := 3115,
	LabelAdjustment_Magazine_Drawer_2_Cassette_25_Position_2 := 3116,
	LabelAdjustment_Magazine_Drawer_2_Cassette_25_Position_3 := 3117,
	LabelAdjustment_Magazine_Drawer_2_Cassette_26_Position_1 := 3118,
	LabelAdjustment_Magazine_Drawer_2_Cassette_26_Position_2 := 3119,
	LabelAdjustment_Magazine_Drawer_2_Cassette_26_Position_3 := 3120,
	LabelAdjustment_Magazine_Drawer_2_Cassette_27_Position_1 := 3121,
	LabelAdjustment_Magazine_Drawer_2_Cassette_27_Position_2 := 3122,
	LabelAdjustment_Magazine_Drawer_2_Cassette_27_Position_3 := 3123,
	LabelAdjustment_Magazine_Drawer_2_Cassette_28_Position_1 := 3124,
	LabelAdjustment_Magazine_Drawer_2_Cassette_28_Position_2 := 3125,
	LabelAdjustment_Magazine_Drawer_2_Cassette_28_Position_3 := 3126,
	LabelAdjustment_Magazine_Drawer_2_Cassette_29_Position_1 := 3127,
	LabelAdjustment_Magazine_Drawer_2_Cassette_29_Position_2 := 3128,
	LabelAdjustment_Magazine_Drawer_2_Cassette_29_Position_3 := 3129,
	LabelAdjustment_Magazine_Drawer_2_Cassette_30_Position_1 := 3130,
	LabelAdjustment_Magazine_Drawer_2_Cassette_30_Position_2 := 3131,
	LabelAdjustment_Magazine_Drawer_2_Cassette_30_Position_3 := 3132,
	LabelAdjustment_Magazine_Drawer_2_Cassette_31_Position_1 := 3133,
	LabelAdjustment_Magazine_Drawer_2_Cassette_31_Position_2 := 3134,
	LabelAdjustment_Magazine_Drawer_2_Cassette_31_Position_3 := 3135,
	LabelAdjustment_Magazine_Drawer_2_Cassette_32_Position_1 := 3136,
	LabelAdjustment_Magazine_Drawer_2_Cassette_32_Position_2 := 3137,
	LabelAdjustment_Magazine_Drawer_2_Cassette_32_Position_3 := 3138,
	LabelAdjustment_Magazine_2_Drawer_1_Cassette_1_Position_1 := 3139,
	LabelAdjustment_Magazine_2_Drawer_1_Cassette_1_Position_2 := 3140,
	LabelAdjustment_Magazine_2_Drawer_1_Cassette_1_Position_3 := 3141,
	LabelAdjustment_Magazine_2_Drawer_1_Cassette_2_Position_1 := 3142,
	LabelAdjustment_Magazine_2_Drawer_1_Cassette_2_Position_2 := 3143,
	LabelAdjustment_Magazine_2_Drawer_1_Cassette_2_Position_3 := 3144,
	LabelAdjustment_Magazine_2_Drawer_1_Cassette_3_Position_1 := 3145,
	LabelAdjustment_Magazine_2_Drawer_1_Cassette_3_Position_2 := 3146,
	LabelAdjustment_Magazine_2_Drawer_1_Cassette_3_Position_3 := 3147,
	LabelAdjustment_Magazine_2_Drawer_1_Cassette_4_Position_1 := 3148,
	LabelAdjustment_Magazine_2_Drawer_1_Cassette_4_Position_2 := 3149,
	LabelAdjustment_Magazine_2_Drawer_1_Cassette_4_Position_3 := 3150,
	LabelAdjustment_Magazine_2_Drawer_1_Cassette_5_Position_1 := 3151,
	LabelAdjustment_Magazine_2_Drawer_1_Cassette_5_Position_2 := 3152,
	LabelAdjustment_Magazine_2_Drawer_1_Cassette_5_Position_3 := 3153,
	LabelAdjustment_Magazine_2_Drawer_1_Cassette_6_Position_1 := 3154,
	LabelAdjustment_Magazine_2_Drawer_1_Cassette_6_Position_2 := 3155,
	LabelAdjustment_Magazine_2_Drawer_1_Cassette_6_Position_3 := 3156,
	LabelAdjustment_Magazine_2_Drawer_1_Cassette_7_Position_1 := 3157,
	LabelAdjustment_Magazine_2_Drawer_1_Cassette_7_Position_2 := 3158,
	LabelAdjustment_Magazine_2_Drawer_1_Cassette_7_Position_3 := 3159,
	LabelAdjustment_Magazine_2_Drawer_1_Cassette_8_Position_1 := 3160,
	LabelAdjustment_Magazine_2_Drawer_1_Cassette_8_Position_2 := 3161,
	LabelAdjustment_Magazine_2_Drawer_1_Cassette_8_Position_3 := 3162,
	LabelAdjustment_Magazine_2_Drawer_1_Cassette_9_Position_1 := 3163,
	LabelAdjustment_Magazine_2_Drawer_1_Cassette_9_Position_2 := 3164,
	LabelAdjustment_Magazine_2_Drawer_1_Cassette_9_Position_3 := 3165,
	LabelAdjustment_Magazine_2_Drawer_1_Cassette_10_Position_1 := 3166,
	LabelAdjustment_Magazine_2_Drawer_1_Cassette_10_Position_2 := 3167,
	LabelAdjustment_Magazine_2_Drawer_1_Cassette_10_Position_3 := 3168,
	LabelAdjustment_Magazine_2_Drawer_1_Cassette_11_Position_1 := 3169,
	LabelAdjustment_Magazine_2_Drawer_1_Cassette_11_Position_2 := 3170,
	LabelAdjustment_Magazine_2_Drawer_1_Cassette_11_Position_3 := 3171,
	LabelAdjustment_Magazine_2_Drawer_1_Cassette_12_Position_1 := 3172,
	LabelAdjustment_Magazine_2_Drawer_1_Cassette_12_Position_2 := 3173,
	LabelAdjustment_Magazine_2_Drawer_1_Cassette_12_Position_3 := 3174,
	LabelAdjustment_Magazine_2_Drawer_1_Cassette_13_Position_1 := 3175,
	LabelAdjustment_Magazine_2_Drawer_1_Cassette_13_Position_2 := 3176,
	LabelAdjustment_Magazine_2_Drawer_1_Cassette_13_Position_3 := 3177,
	LabelAdjustment_Magazine_2_Drawer_1_Cassette_14_Position_1 := 3178,
	LabelAdjustment_Magazine_2_Drawer_1_Cassette_14_Position_2 := 3179,
	LabelAdjustment_Magazine_2_Drawer_1_Cassette_14_Position_3 := 3180,
	LabelAdjustment_Magazine_2_Drawer_1_Cassette_15_Position_1 := 3181,
	LabelAdjustment_Magazine_2_Drawer_1_Cassette_15_Position_2 := 3182,
	LabelAdjustment_Magazine_2_Drawer_1_Cassette_15_Position_3 := 3183,
	LabelAdjustment_Magazine_2_Drawer_1_Cassette_16_Position_1 := 3184,
	LabelAdjustment_Magazine_2_Drawer_1_Cassette_16_Position_2 := 3185,
	LabelAdjustment_Magazine_2_Drawer_1_Cassette_16_Position_3 := 3186,
	LabelAdjustment_Magazine_2_Drawer_1_Cassette_17_Position_1 := 3187,
	LabelAdjustment_Magazine_2_Drawer_1_Cassette_17_Position_2 := 3188,
	LabelAdjustment_Magazine_2_Drawer_1_Cassette_17_Position_3 := 3189,
	LabelAdjustment_Magazine_2_Drawer_1_Cassette_18_Position_1 := 3190,
	LabelAdjustment_Magazine_2_Drawer_1_Cassette_18_Position_2 := 3191,
	LabelAdjustment_Magazine_2_Drawer_1_Cassette_18_Position_3 := 3192,
	LabelAdjustment_Magazine_2_Drawer_1_Cassette_19_Position_1 := 3193,
	LabelAdjustment_Magazine_2_Drawer_1_Cassette_19_Position_2 := 3194,
	LabelAdjustment_Magazine_2_Drawer_1_Cassette_19_Position_3 := 3195,
	LabelAdjustment_Magazine_2_Drawer_1_Cassette_20_Position_1 := 3196,
	LabelAdjustment_Magazine_2_Drawer_1_Cassette_20_Position_2 := 3197,
	LabelAdjustment_Magazine_2_Drawer_1_Cassette_20_Position_3 := 3198,
	LabelAdjustment_Magazine_2_Drawer_1_Cassette_21_Position_1 := 3199,
	LabelAdjustment_Magazine_2_Drawer_1_Cassette_21_Position_2 := 3200,
	LabelAdjustment_Magazine_2_Drawer_1_Cassette_21_Position_3 := 3201,
	LabelAdjustment_Magazine_2_Drawer_1_Cassette_22_Position_1 := 3202,
	LabelAdjustment_Magazine_2_Drawer_1_Cassette_22_Position_2 := 3203,
	LabelAdjustment_Magazine_2_Drawer_1_Cassette_22_Position_3 := 3204,
	LabelAdjustment_Magazine_2_Drawer_1_Cassette_23_Position_1 := 3205,
	LabelAdjustment_Magazine_2_Drawer_1_Cassette_23_Position_2 := 3206,
	LabelAdjustment_Magazine_2_Drawer_1_Cassette_23_Position_3 := 3207,
	LabelAdjustment_Magazine_2_Drawer_1_Cassette_24_Position_1 := 3208,
	LabelAdjustment_Magazine_2_Drawer_1_Cassette_24_Position_2 := 3209,
	LabelAdjustment_Magazine_2_Drawer_1_Cassette_24_Position_3 := 3210,
	LabelAdjustment_Magazine_2_Drawer_1_Cassette_25_Position_1 := 3211,
	LabelAdjustment_Magazine_2_Drawer_1_Cassette_25_Position_2 := 3212,
	LabelAdjustment_Magazine_2_Drawer_1_Cassette_25_Position_3 := 3213,
	LabelAdjustment_Magazine_2_Drawer_1_Cassette_26_Position_1 := 3214,
	LabelAdjustment_Magazine_2_Drawer_1_Cassette_26_Position_2 := 3215,
	LabelAdjustment_Magazine_2_Drawer_1_Cassette_26_Position_3 := 3216,
	LabelAdjustment_Magazine_2_Drawer_1_Cassette_27_Position_1 := 3217,
	LabelAdjustment_Magazine_2_Drawer_1_Cassette_27_Position_2 := 3218,
	LabelAdjustment_Magazine_2_Drawer_1_Cassette_27_Position_3 := 3219,
	LabelAdjustment_Magazine_2_Drawer_1_Cassette_28_Position_1 := 3220,
	LabelAdjustment_Magazine_2_Drawer_1_Cassette_28_Position_2 := 3221,
	LabelAdjustment_Magazine_2_Drawer_1_Cassette_28_Position_3 := 3222,
	LabelAdjustment_Magazine_2_Drawer_1_Cassette_29_Position_1 := 3223,
	LabelAdjustment_Magazine_2_Drawer_1_Cassette_29_Position_2 := 3224,
	LabelAdjustment_Magazine_2_Drawer_1_Cassette_29_Position_3 := 3225,
	LabelAdjustment_Magazine_2_Drawer_1_Cassette_30_Position_1 := 3226,
	LabelAdjustment_Magazine_2_Drawer_1_Cassette_30_Position_2 := 3227,
	LabelAdjustment_Magazine_2_Drawer_1_Cassette_30_Position_3 := 3228,
	LabelAdjustment_Magazine_2_Drawer_1_Cassette_31_Position_1 := 3229,
	LabelAdjustment_Magazine_2_Drawer_1_Cassette_31_Position_2 := 3230,
	LabelAdjustment_Magazine_2_Drawer_1_Cassette_31_Position_3 := 3231,
	LabelAdjustment_Magazine_2_Drawer_1_Cassette_32_Position_1 := 3232,
	LabelAdjustment_Magazine_2_Drawer_1_Cassette_32_Position_2 := 3233,
	LabelAdjustment_Magazine_2_Drawer_1_Cassette_32_Position_3 := 3234,
	LabelAdjustment_Magazine_2_Drawer_2_Cassette_1_Position_1 := 3235,
	LabelAdjustment_Magazine_2_Drawer_2_Cassette_1_Position_2 := 3236,
	LabelAdjustment_Magazine_2_Drawer_2_Cassette_1_Position_3 := 3237,
	LabelAdjustment_Magazine_2_Drawer_2_Cassette_2_Position_1 := 3238,
	LabelAdjustment_Magazine_2_Drawer_2_Cassette_2_Position_2 := 3239,
	LabelAdjustment_Magazine_2_Drawer_2_Cassette_2_Position_3 := 3240,
	LabelAdjustment_Magazine_2_Drawer_2_Cassette_3_Position_1 := 3241,
	LabelAdjustment_Magazine_2_Drawer_2_Cassette_3_Position_2 := 3242,
	LabelAdjustment_Magazine_2_Drawer_2_Cassette_3_Position_3 := 3243,
	LabelAdjustment_Magazine_2_Drawer_2_Cassette_4_Position_1 := 3244,
	LabelAdjustment_Magazine_2_Drawer_2_Cassette_4_Position_2 := 3245,
	LabelAdjustment_Magazine_2_Drawer_2_Cassette_4_Position_3 := 3246,
	LabelAdjustment_Magazine_2_Drawer_2_Cassette_5_Position_1 := 3247,
	LabelAdjustment_Magazine_2_Drawer_2_Cassette_5_Position_2 := 3248,
	LabelAdjustment_Magazine_2_Drawer_2_Cassette_5_Position_3 := 3249,
	LabelAdjustment_Magazine_2_Drawer_2_Cassette_6_Position_1 := 3250,
	LabelAdjustment_Magazine_2_Drawer_2_Cassette_6_Position_2 := 3251,
	LabelAdjustment_Magazine_2_Drawer_2_Cassette_6_Position_3 := 3252,
	LabelAdjustment_Magazine_2_Drawer_2_Cassette_7_Position_1 := 3253,
	LabelAdjustment_Magazine_2_Drawer_2_Cassette_7_Position_2 := 3254,
	LabelAdjustment_Magazine_2_Drawer_2_Cassette_7_Position_3 := 3255,
	LabelAdjustment_Magazine_2_Drawer_2_Cassette_8_Position_1 := 3256,
	LabelAdjustment_Magazine_2_Drawer_2_Cassette_8_Position_2 := 3257,
	LabelAdjustment_Magazine_2_Drawer_2_Cassette_8_Position_3 := 3258,
	LabelAdjustment_Magazine_2_Drawer_2_Cassette_9_Position_1 := 3259,
	LabelAdjustment_Magazine_2_Drawer_2_Cassette_9_Position_2 := 3260,
	LabelAdjustment_Magazine_2_Drawer_2_Cassette_9_Position_3 := 3261,
	LabelAdjustment_Magazine_2_Drawer_2_Cassette_10_Position_1 := 3262,
	LabelAdjustment_Magazine_2_Drawer_2_Cassette_10_Position_2 := 3263,
	LabelAdjustment_Magazine_2_Drawer_2_Cassette_10_Position_3 := 3264,
	LabelAdjustment_Magazine_2_Drawer_2_Cassette_11_Position_1 := 3265,
	LabelAdjustment_Magazine_2_Drawer_2_Cassette_11_Position_2 := 3266,
	LabelAdjustment_Magazine_2_Drawer_2_Cassette_11_Position_3 := 3267,
	LabelAdjustment_Magazine_2_Drawer_2_Cassette_12_Position_1 := 3268,
	LabelAdjustment_Magazine_2_Drawer_2_Cassette_12_Position_2 := 3269,
	LabelAdjustment_Magazine_2_Drawer_2_Cassette_12_Position_3 := 3270,
	LabelAdjustment_Magazine_2_Drawer_2_Cassette_13_Position_1 := 3271,
	LabelAdjustment_Magazine_2_Drawer_2_Cassette_13_Position_2 := 3272,
	LabelAdjustment_Magazine_2_Drawer_2_Cassette_13_Position_3 := 3273,
	LabelAdjustment_Magazine_2_Drawer_2_Cassette_14_Position_1 := 3274,
	LabelAdjustment_Magazine_2_Drawer_2_Cassette_14_Position_2 := 3275,
	LabelAdjustment_Magazine_2_Drawer_2_Cassette_14_Position_3 := 3276,
	LabelAdjustment_Magazine_2_Drawer_2_Cassette_15_Position_1 := 3277,
	LabelAdjustment_Magazine_2_Drawer_2_Cassette_15_Position_2 := 3278,
	LabelAdjustment_Magazine_2_Drawer_2_Cassette_15_Position_3 := 3279,
	LabelAdjustment_Magazine_2_Drawer_2_Cassette_16_Position_1 := 3280,
	LabelAdjustment_Magazine_2_Drawer_2_Cassette_16_Position_2 := 3281,
	LabelAdjustment_Magazine_2_Drawer_2_Cassette_16_Position_3 := 3282,
	LabelAdjustment_Magazine_2_Drawer_2_Cassette_17_Position_1 := 3283,
	LabelAdjustment_Magazine_2_Drawer_2_Cassette_17_Position_2 := 3284,
	LabelAdjustment_Magazine_2_Drawer_2_Cassette_17_Position_3 := 3285,
	LabelAdjustment_Magazine_2_Drawer_2_Cassette_18_Position_1 := 3286,
	LabelAdjustment_Magazine_2_Drawer_2_Cassette_18_Position_2 := 3287,
	LabelAdjustment_Magazine_2_Drawer_2_Cassette_18_Position_3 := 3288,
	LabelAdjustment_Magazine_2_Drawer_2_Cassette_19_Position_1 := 3289,
	LabelAdjustment_Magazine_2_Drawer_2_Cassette_19_Position_2 := 3290,
	LabelAdjustment_Magazine_2_Drawer_2_Cassette_19_Position_3 := 3291,
	LabelAdjustment_Magazine_2_Drawer_2_Cassette_20_Position_1 := 3292,
	LabelAdjustment_Magazine_2_Drawer_2_Cassette_20_Position_2 := 3293,
	LabelAdjustment_Magazine_2_Drawer_2_Cassette_20_Position_3 := 3294,
	LabelAdjustment_Magazine_2_Drawer_2_Cassette_21_Position_1 := 3295,
	LabelAdjustment_Magazine_2_Drawer_2_Cassette_21_Position_2 := 3296,
	LabelAdjustment_Magazine_2_Drawer_2_Cassette_21_Position_3 := 3297,
	LabelAdjustment_Magazine_2_Drawer_2_Cassette_22_Position_1 := 3298,
	LabelAdjustment_Magazine_2_Drawer_2_Cassette_22_Position_2 := 3299,
	LabelAdjustment_Magazine_2_Drawer_2_Cassette_22_Position_3 := 3300,
	LabelAdjustment_Magazine_2_Drawer_2_Cassette_23_Position_1 := 3301,
	LabelAdjustment_Magazine_2_Drawer_2_Cassette_23_Position_2 := 3302,
	LabelAdjustment_Magazine_2_Drawer_2_Cassette_23_Position_3 := 3303,
	LabelAdjustment_Magazine_2_Drawer_2_Cassette_24_Position_1 := 3304,
	LabelAdjustment_Magazine_2_Drawer_2_Cassette_24_Position_2 := 3305,
	LabelAdjustment_Magazine_2_Drawer_2_Cassette_24_Position_3 := 3306,
	LabelAdjustment_Magazine_2_Drawer_2_Cassette_25_Position_1 := 3307,
	LabelAdjustment_Magazine_2_Drawer_2_Cassette_25_Position_2 := 3308,
	LabelAdjustment_Magazine_2_Drawer_2_Cassette_25_Position_3 := 3309,
	LabelAdjustment_Magazine_2_Drawer_2_Cassette_26_Position_1 := 3310,
	LabelAdjustment_Magazine_2_Drawer_2_Cassette_26_Position_2 := 3311,
	LabelAdjustment_Magazine_2_Drawer_2_Cassette_26_Position_3 := 3312,
	LabelAdjustment_Magazine_2_Drawer_2_Cassette_27_Position_1 := 3313,
	LabelAdjustment_Magazine_2_Drawer_2_Cassette_27_Position_2 := 3314,
	LabelAdjustment_Magazine_2_Drawer_2_Cassette_27_Position_3 := 3315,
	LabelAdjustment_Magazine_2_Drawer_2_Cassette_28_Position_1 := 3316,
	LabelAdjustment_Magazine_2_Drawer_2_Cassette_28_Position_2 := 3317,
	LabelAdjustment_Magazine_2_Drawer_2_Cassette_28_Position_3 := 3318,
	LabelAdjustment_Magazine_2_Drawer_2_Cassette_29_Position_1 := 3319,
	LabelAdjustment_Magazine_2_Drawer_2_Cassette_29_Position_2 := 3320,
	LabelAdjustment_Magazine_2_Drawer_2_Cassette_29_Position_3 := 3321,
	LabelAdjustment_Magazine_2_Drawer_2_Cassette_30_Position_1 := 3322,
	LabelAdjustment_Magazine_2_Drawer_2_Cassette_30_Position_2 := 3323,
	LabelAdjustment_Magazine_2_Drawer_2_Cassette_30_Position_3 := 3324,
	LabelAdjustment_Magazine_2_Drawer_2_Cassette_31_Position_1 := 3325,
	LabelAdjustment_Magazine_2_Drawer_2_Cassette_31_Position_2 := 3326,
	LabelAdjustment_Magazine_2_Drawer_2_Cassette_31_Position_3 := 3327,
	LabelAdjustment_Magazine_2_Drawer_2_Cassette_32_Position_1 := 3328,
	LabelAdjustment_Magazine_2_Drawer_2_Cassette_32_Position_2 := 3329,
	LabelAdjustment_Magazine_2_Drawer_2_Cassette_32_Position_3 := 3330,
	ProductVerification_Alarms := 3331,
	Main_HighVacuumTankFull := 3332,
	Main_LowVacuumTankFull := 3333,
	ReverseUnit_Alarms := 3334,
	ReverseUnit_SensorTimes_Vacuum_1 := 3335,
	ReverseUnit_SensorTimes_ExtendIn := 3336,
	ReverseUnit_SensorTimes_ExtendOut := 3337,
	ReverseUnit_SensorTimes_RotateIn := 3338,
	ReverseUnit_SensorTimes_RotateOut := 3339,
	ZUnit_SensorTimes_Extend5In := 3340,
	ZUnit_SensorTimes_Extend6In := 3341,
	ZUnit_SensorTimes_Extend7In := 3342,
	ZUnit_SensorTimes_Extend8In := 3343,
	ZUnit_SensorTimes_Vacuum_5 := 3344,
	ZUnit_SensorTimes_Vacuum_6 := 3345,
	ZUnit_SensorTimes_Vacuum_7 := 3346,
	ZUnit_SensorTimes_Vacuum_8 := 3347,
	TZUnit_Alarms := 3348,
	TZUnit_CoveredDistance := 3349,
	TZUnit_ErrorID := 3350,
	TZUnit_AxisErrorId := 3351,
	TZUnit_DriveErrorId := 3352,
	TZUnit_DriveUtilisation := 3353,
	TZUnit_MotorUtilisation := 3354,
	RejectStation_SensorTimes_ProductCarrierReject1In := 3355,
	RejectStation_SensorTimes_ProductCarrierReject2In := 3356,
	RejectStation_SensorTimes_ProductCarrierReject3In := 3357,
	RejectStation_SensorTimes_ProductCarrierReject4In := 3358,
	TUnit_SensorTimes_Vacuum_1_5 := 3359,
	TUnit_SensorTimes_Vacuum_1_6 := 3360,
	TUnit_SensorTimes_Vacuum_1_7 := 3361,
	TUnit_SensorTimes_Vacuum_1_8 := 3362,
	ZUnit_SensorTimes_ProductCarrierStacking1In := 3363,
	ZUnit_SensorTimes_ProductCarrierStacking2In := 3364,
	ZUnit_SensorTimes_ProductCarrierStacking3In := 3365,
	ZUnit_SensorTimes_ProductCarrierStacking4In := 3366,
	ZUnit_SensorTimes_ProductCarrierStacking5In := 3367,
	ZUnit_SensorTimes_ProductCarrierStacking6In := 3368,
	ZUnit_SensorTimes_ProductCarrierStacking7In := 3369,
	ZUnit_SensorTimes_ProductCarrierStacking8In := 3370,
	TUnit_SensorTimes_ProductCarrierTransfer1In := 3371,
	TUnit_SensorTimes_ProductCarrierTransfer1Out := 3379,
	TZUnit_Time_Idle := 3387,
	TXUnit_Time_Idle := 3388,
	TZUnit_Time_Active := 3389,
	TXUnit_Time_Active := 3390,
	LZUnit_Alarms := 3391,
	LZUnit_CoveredDistance := 3392,
	LZUnit_ErrorID := 3393,
	LZUnit_AxisErrorId := 3394,
	LZUnit_DriveUtilisation := 3395,
	LZUnit_MotorUtilisation := 3396,
	LZUnit_Time_Idle := 3397,
	LZUnit_Time_Active := 3398,
	LUnit_L5_Alarms := 3399,
	LUnit_L6_Alarms := 3400,
	LUnit_L7_Alarms := 3401,
	LUnit_L8_Alarms := 3402,
	TCO_Alarms := 3403,
	TCO_CoveredDistance := 3404,
	TCO_ErrorID := 3405,
	TCO_AxisErrorId := 3406,
	TCO_DriveUtilisation := 3407,
	TCO_MotorUtilisation := 3408,
	TCO_Time_Idle := 3409,
	TCO_Time_Active := 3410,
	LZ2Unit_Alarms := 3411,
	LZ2Unit_CoveredDistance := 3412,
	LZ2Unit_ErrorID := 3413,
	LZ2Unit_AxisErrorId := 3414,
	LZ2Unit_DriveUtilisation := 3415,
	LZ2Unit_MotorUtilisation := 3416,
	LZ2Unit_Time_Idle := 3417,
	LZ2Unit_Time_Active := 3418,
	LUnit_L5_CoveredDistance := 3419,
	LUnit_L6_CoveredDistance := 3420,
	LUnit_L7_CoveredDistance := 3421,
	LUnit_L8_CoveredDistance := 3422,
	LUnit_L5_ErrorId := 3423,
	LUnit_L6_ErrorId := 3424,
	LUnit_L7_ErrorId := 3425,
	LUnit_L8_ErrorId := 3426,
	LUnit_L5_AxisErrorId := 3427,
	LUnit_L6_AxisErrorId := 3428,
	LUnit_L7_AxisErrorId := 3429,
	LUnit_L8_AxisErrorId := 3430,
	LUnit_L5_DriveErrorId := 3431,
	LUnit_L6_DriveErrorId := 3432,
	LUnit_L7_DriveErrorId := 3433,
	LUnit_L8_DriveErrorId := 3434,
	LUnit_L5_DriveUtilisation := 3435,
	LUnit_L6_DriveUtilisation := 3436,
	LUnit_L7_DriveUtilisation := 3437,
	LUnit_L8_DriveUtilisation := 3438,
	LUnit_L5_MotorUtilisation := 3439,
	LUnit_L6_MotorUtilisation := 3440,
	LUnit_L7_MotorUtilisation := 3441,
	LUnit_L8_MotorUtilisation := 3442,
	LZUnit_DriveErrorId := 3443,
	LZ2Unit_DriveErrorId := 3444,
	TCO_DriveErrorId := 3445,
	Xu2Unit_SensorTimes_ShiftIn := 3446,
	Xu2Unit_SensorTimes_ShiftOut := 3447,
	LZUnit_SensorTimes_Vacuum_1 := 3448,
	LZUnit_SensorTimes_Vacuum_2 := 3449,
	LZUnit_SensorTimes_Vacuum_3 := 3450,
	LZUnit_SensorTimes_Vacuum_4 := 3451,
	LZUnit_SensorTimes_Vacuum_5 := 3452,
	LZUnit_SensorTimes_Vacuum_6 := 3453,
	LZUnit_SensorTimes_Vacuum_7 := 3454,
	LZUnit_SensorTimes_Vacuum_8 := 3455,
	LZ2Unit_SensorTimes_Vacuum_1 := 3456,
	LZ2Unit_SensorTimes_Vacuum_2 := 3457,
	LZ2Unit_SensorTimes_Vacuum_3 := 3458,
	LZ2Unit_SensorTimes_Vacuum_4 := 3459,
	LZ2Unit_SensorTimes_Vacuum_5 := 3460,
	LZ2Unit_SensorTimes_Vacuum_6 := 3461,
	LZ2Unit_SensorTimes_Vacuum_7 := 3462,
	LZ2Unit_SensorTimes_Vacuum_8 := 3463,
	BFU_PickAndPlace_SensorTimes_RotateBoxFillGripperIn := 3464,
	BFU_PickAndPlace_SensorTimes_RotateBoxFillGripperOut := 3465,
	BFU_PickAndPlace_SensorTimes_Vacuum1In := 3466,
	BFU_PickAndPlace_SensorTimes_Vacuum2In := 3467,
	BFU_PickAndPlace_SensorTimes_Vacuum1Out := 3468,
	BFU_PickAndPlace_SensorTimes_Vacuum2Out := 3469,
	TCO_SensorTimes_ClampBottom1In := 3470,
	TCO_SensorTimes_ClampBottom2In := 3471,
	TCO_SensorTimes_ClampBottom3In := 3472,
	TCO_SensorTimes_ClampBottom4In := 3473,
	TCO_SensorTimes_ClampBottom5In := 3474,
	TCO_SensorTimes_ClampBottom6In := 3475,
	TCO_SensorTimes_ClampBottom7In := 3476,
	TCO_SensorTimes_ClampBottom8In := 3477,
	TCO_SensorTimes_ClampTop1In := 3478,
	TCO_SensorTimes_ClampTop2In := 3479,
	TCO_SensorTimes_ClampTop3In := 3480,
	TCO_SensorTimes_ClampTop4In := 3481,
	TCO_SensorTimes_ClampTop5In := 3482,
	TCO_SensorTimes_ClampTop6In := 3483,
	TCO_SensorTimes_ClampTop7In := 3484,
	TCO_SensorTimes_ClampTop8In := 3485,
	LUnit_L5_Time_Active := 3486,
	LUnit_L6_Time_Active := 3487,
	LUnit_L7_Time_Active := 3488,
	LUnit_L8_Time_Active := 3489,
	XUnit_BFU_Time_Idle := 3490,
	ZUnit_BFU_Time_Idle := 3491,
	LUnit_L5_Time_Idle := 3492,
	LUnit_L6_Time_Idle := 3493,
	LUnit_L7_Time_Idle := 3494,
	LUnit_L8_Time_Idle := 3495,
	BDE_BDE_Output1 := 3496,
	BDE_BDE_Output2 := 3497,
	BDE_BDE_Output3 := 3498,
	Main_Relays_BlowerVacuumPumpRunning := 3499,
	BFU_PickAndPlace_Relays_Vacuum1 := 3500,
	BFU_PickAndPlace_Relays_Vacuum2 := 3501,
	XiUnit_SensorTimes_Shift1In := 3502,
	XiUnit_SensorTimes_Shift1Out := 3503,
	XuUnit_SensorTimes_Shift1In := 3504,
	XuUnit_SensorTimes_Shift1Out := 3505,
	PTZ_ZUnit_Alarms := 3506,
	PTZ_YUnit_Alarms := 3507,
	PTZ_Transfer_Alarms := 3508,
	PTZ_PalletCenterUnit_1_Alarms := 3509,
	PTZ_PalletCenterUnit_2_Alarms := 3510,
	PTZ_Messages := 3511,
	PTZ_SheetDrawer_Alarms := 3512,
	PTZ_Transfer_CoveredDistance := 3513,
	PTZ_YUnit_CoveredDistance := 3514,
	PTZ_ZUnit_CoveredDistance := 3515,
	PTZ_PalletCenterUnit_1_CoveredDistance := 3516,
	PTZ_PalletCenterUnit_2_CoveredDistance := 3517,
	PTZ_Transfer_ErrorId := 3518,
	PTZ_YUnit_ErrorId := 3519,
	PTZ_ZUnit_ErrorId := 3520,
	PTZ_PalletCenterUnit_1_ErrorId := 3521,
	PTZ_PalletCenterUnit_2_ErrorId := 3522,
	PTZ_Transfer_AxisErrorId := 3523,
	PTZ_YUnit_AxisErrorId := 3524,
	PTZ_ZUnit_AxisErrorId := 3525,
	PTZ_PalletCenterUnit_1_AxisErrorId := 3526,
	PTZ_PalletCenterUnit_2_AxisErrorId := 3527,
	PTZ_Transfer_DriveErrorId := 3528,
	PTZ_YUnit_DriveErrorId := 3529,
	PTZ_ZUnit_DriveErrorId := 3530,
	PTZ_PalletCenterUnit_1_DriveErrorId := 3531,
	PTZ_PalletCenterUnit_2_DriveErrorId := 3532,
	PTZ_Transfer_DriveUtilisation := 3533,
	PTZ_YUnit_DriveUtilisation := 3534,
	PTZ_ZUnit_DriveUtilisation := 3535,
	PTZ_PalletCenterUnit_1_DriveUtilisation := 3536,
	PTZ_PalletCenterUnit_2_DriveUtilisation := 3537,
	PTZ_Transfer_MotorUtilisation := 3538,
	PTZ_YUnit_MotorUtilisation := 3539,
	PTZ_ZUnit_MotorUtilisation := 3540,
	PTZ_PalletCenterUnit_1_MotorUtilisation := 3541,
	PTZ_PalletCenterUnit_2_MotorUtilisation := 3542,
	PTZ_PalletCenterUnit_1_SensorTimes_ClampIn := 3543,
	PTZ_PalletCenterUnit_1_SensorTimes_ClampOut := 3544,
	PTZ_PalletCenterUnit_2_SensorTimes_ClampIn := 3545,
	PTZ_PalletCenterUnit_2_SensorTimes_ClampOut := 3546,
	PTZ_Transfer_SensorTimes_ExtendIn := 3547,
	PTZ_Transfer_SensorTimes_ExtendOut := 3548,
	PTZ_ZUnit_SensorTimes_ExtendIn := 3549,
	PTZ_ZUnit_SensorTimes_ExtendSafetyFencingIn := 3550,
	PTZ_Transfer_SensorTimes_Vacuum_1 := 3551,
	PTZ_Transfer_SensorTimes_Vacuum_2 := 3552,
	PTZ_ZUnit_SensorTimes_Vacuum_1 := 3553,
	PTZ_ZUnit_SensorTimes_Vacuum_2 := 3554,
	PTZ_ZUnit_SensorTimes_Vacuum_3 := 3555,
	PTZ_ZUnit_SensorTimes_Vacuum_4 := 3556,
	PTZ_ZUnit_SensorTimes_Vacuum_5 := 3557,
	PTZ_ZUnit_SensorTimes_Vacuum_6 := 3558,
	PTZ_ZUnit_SensorTimes_Vacuum_7 := 3559,
	PTZ_ZUnit_SensorTimes_Vacuum_Sheet := 3560,
	PTZ_AirPressureOk := 3561,
	PTZ_HighVacuumTankFull := 3562,
	Transfer_Alarms := 3563,
	Traverse_CoveredDistance := 3564,
	Traverse_ErrorId := 3565,
	Traverse_AxisErrorId := 3566,
	Traverse_DriveErrorId := 3567,
	Traverse_DriveUtilisation := 3568,
	Traverse_MotorUtilisation := 3569,
	Magazine_SensorTimes_VacuumBottom_1 := 3570,
	Magazine_SensorTimes_VacuumBottom_2 := 3571,
	Magazine_SensorTimes_VacuumBottom_3 := 3572,
	Magazine_SensorTimes_VacuumBottom_4 := 3573,
	Magazine_SensorTimes_VacuumSide_1 := 3574,
	Magazine_SensorTimes_VacuumSide_2 := 3575,
	Magazine_SensorTimes_VacuumAdditional_2 := 3576,
	Magazine_SensorTimes_VacuumAdditional_1 := 3577,
	Transfer_SensorTimes_ProductCarrierTransfer1In := 3578,
	Transfer_SensorTimes_ProductCarrierTransfer1Out := 3579,
	Transfer_SensorTimes_Extend1In := 3580,
	Transfer_SensorTimes_Extend1Out := 3581,
	Transfer_SensorTimes_Vacuum_1 := 3582,
	Transfer_SensorTimes_Vacuum_2 := 3583,
	Transfer_SensorTimes_Vacuum_3 := 3584,
	Transfer_SensorTimes_Vacuum_4 := 3585,
	Transfer_SensorTimes_Vacuum_5 := 3586,
	Transfer_SensorTimes_Vacuum_6 := 3587,
	Transfer_SensorTimes_Vacuum_7 := 3588,
	Transfer_SensorTimes_Vacuum_8 := 3589,
	Transfer_SensorTimes_Vacuum_9 := 3590,
	Transfer_SensorTimes_Vacuum_10 := 3591,
	Transfer_SensorTimes_Vacuum_11 := 3592,
	Transfer_SensorTimes_RotateIn := 3593,
	Transfer_SensorTimes_RotateOut := 3594,
	ZUnit_SensorTimes_Vacuum_9 := 3595,
	ZUnit_SensorTimes_Vacuum_10 := 3596,
	ZUnit_SensorTimes_Vacuum_11 := 3597,
	Z2Unit_SensorTimes_ChainProductCarrier_1_Pos1 := 3598,
	Z2Unit_SensorTimes_ChainProductCarrier_2_Pos1 := 3599,
	Z2Unit_SensorTimes_ChainProductCarrier_3_Pos1 := 3600,
	Z2Unit_SensorTimes_ChainProductCarrier_4_Pos1 := 3601,
	Z2Unit_SensorTimes_ChainProductCarrier_5_Pos1 := 3602,
	Z2Unit_SensorTimes_ChainProductCarrier_6_Pos1 := 3603,
	Z2Unit_SensorTimes_ChainProductCarrier_7_Pos1 := 3604,
	Z2Unit_SensorTimes_ChainProductCarrier_8_Pos1 := 3605,
	Z2Unit_SensorTimes_ChainProductCarrier_9_Pos1 := 3606,
	Z2Unit_SensorTimes_ChainProductCarrier_10_Pos1 := 3607,
	Z2Unit_SensorTimes_ChainProductCarrier_11_Pos1 := 3608,
	Z2Unit_SensorTimes_ChainProductCarrier_1_Pos2 := 3609,
	Z2Unit_SensorTimes_ChainProductCarrier_2_Pos2 := 3610,
	Z2Unit_SensorTimes_ChainProductCarrier_3_Pos2 := 3611,
	Z2Unit_SensorTimes_ChainProductCarrier_4_Pos2 := 3612,
	Z2Unit_SensorTimes_ChainProductCarrier_5_Pos2 := 3613,
	Z2Unit_SensorTimes_ChainProductCarrier_6_Pos2 := 3614,
	Z2Unit_SensorTimes_ChainProductCarrier_7_Pos2 := 3615,
	Z2Unit_SensorTimes_ChainProductCarrier_8_Pos2 := 3616,
	Z2Unit_SensorTimes_ChainProductCarrier_9_Pos2 := 3617,
	Z2Unit_SensorTimes_ChainProductCarrier_10_Pos2 := 3618,
	Z2Unit_SensorTimes_ChainProductCarrier_11_Pos2 := 3619,
	Z2Unit_SensorTimes_Extend1In := 3620,
	Z2Unit_SensorTimes_Extend1Out := 3621,
	Z2Unit_SensorTimes_Extend2In := 3622,
	Z2Unit_SensorTimes_Extend2Out := 3623,
	Z2Unit_SensorTimes_Extend3In := 3624,
	Z2Unit_SensorTimes_Extend3Out := 3625,
	Z2Unit_SensorTimes_Extend4In := 3626,
	Z2Unit_SensorTimes_Extend4Out := 3627,
	Z2Unit_SensorTimes_Extend5Out := 3628,
	Z2Unit_SensorTimes_Extend5In := 3629,
	Z2Unit_SensorTimes_Extend6In := 3630,
	Z2Unit_SensorTimes_Extend6Out := 3631,
	Z2Unit_SensorTimes_Extend7In := 3632,
	Z2Unit_SensorTimes_Extend7Out := 3633,
	Z2Unit_SensorTimes_Extend8In := 3634,
	Z2Unit_SensorTimes_Extend8Out := 3635,
	Z2Unit_SensorTimes_Extend9In := 3636,
	Z2Unit_SensorTimes_Extend9Out := 3637,
	Z2Unit_SensorTimes_Extend10In := 3638,
	Z2Unit_SensorTimes_Extend10Out := 3639,
	Z2Unit_SensorTimes_Extend11In := 3640,
	Z2Unit_SensorTimes_Extend11Out := 3641,
	Z2Unit_SensorTimes_Vacuum_5 := 3642,
	Z2Unit_SensorTimes_Vacuum_6 := 3643,
	Z2Unit_SensorTimes_Vacuum_7 := 3644,
	Z2Unit_SensorTimes_Vacuum_8 := 3645,
	Z2Unit_SensorTimes_Vacuum_9 := 3646,
	Z2Unit_SensorTimes_Vacuum_10 := 3647,
	Z2Unit_SensorTimes_Vacuum_11 := 3648,
	RejectStation_SensorTimes_ChainProductCarrier_1_Pos2 := 3649,
	ZUnit_SensorTimes_ProductCarrierStacking9In := 3650,
	ZUnit_SensorTimes_ProductCarrierStacking10In := 3651,
	ZUnit_SensorTimes_ProductCarrierStacking11In := 3652,
	Transfer_Time_Idle := 3653,
	Transfer_Time_Active := 3654,
	Z2Unit_SensorTimes_ProductCarrierStacking1In := 3655,
	Z2Unit_SensorTimes_ProductCarrierStacking2In := 3656,
	Z2Unit_SensorTimes_ProductCarrierStacking3In := 3657,
	Z2Unit_SensorTimes_ProductCarrierStacking4In := 3658,
	Z2Unit_SensorTimes_ProductCarrierStacking5In := 3659,
	Z2Unit_SensorTimes_ProductCarrierStacking6In := 3660,
	Z2Unit_SensorTimes_ProductCarrierStacking7In := 3661,
	Z2Unit_SensorTimes_ProductCarrierStacking8In := 3662,
	Z2Unit_SensorTimes_ProductCarrierStacking9In := 3663,
	Z2Unit_SensorTimes_ProductCarrierStacking10In := 3664,
	Z2Unit_SensorTimes_ProductCarrierStacking11In := 3665,
	Z2Unit_SensorTimes_RotateIn := 3666,
	Z2Unit_SensorTimes_RotateOut := 3667,
	Traverse_Alarms := 3668,
	IMM_DoorsClosed := 3669,
	IMM_RejectMoulding := 3670,
	IMM_MouldClosed := 3671,
	IMM_MouldOpenPosition := 3672,
	IMM_IntermediateMouldOpenPosition := 3673,
	IMM_AutoOperation := 3674,
	IMM_EjectorBack := 3675,
	IMM_EjectorForward := 3676,
	IMM_CorePos1Back := 3677,
	IMM_CorePos2Forward := 3678,
	BFU_RobotStatus := 3679,
	Fanuc_SensorTimes_Clamp1In := 3680,
	Fanuc_SensorTimes_Clamp2In := 3681,
	Fanuc_SensorTimes_Clamp2Out := 3682,
	Fanuc_SensorTimes_Clamp1Out := 3683,
	Fanuc_SensorTimes_LockStackIn := 3684,
	Fanuc_SensorTimes_LockStackOut := 3685,
	Main_IgnoreReject := 3686,
	Main_IgnoreMouldReject := 3687,
	Main_IgnoreRunmode := 3688,
	Camera_RunMode := 3689,
	YUnit_ClearMould := 3690,
	YUnit_MouldOpen := 3691,
	YUnit_IntermediateMouldOpen := 3692,
	Camera_EnableMeasuringVision := 3693,
	Main_ActiveProg := 3694,
	Main_ActiveLabel := 3695,
	I1Unit_Alarms := 3696,
	I2Unit_Alarms := 3697,
	Main_DoorStatusOpen := 3698,
	PTZ_PalletCenterUnit_1_PalletAreaFree := 3699,
	PTZ_PalletCenterUnit_2_PalletAreaFree := 3700,
	PTZ_Patternizer_TransferAreaFree1 := 3701,
	PTZ_Patternizer_TransferAreaFree2 := 3702,
	PTZ_Patternizer_TransferAreaFree3 := 3703,
	PTZ_ZUnit_AirPressureOk := 3704,
	PTZ_SheetDrawer_GateClosed := 3705,
	PTZ_SheetDrawer_GateOpened := 3706,
	PTZ_PalletCenterUnit_1_PalletInPosition := 3707,
	PTZ_PalletCenterUnit_2_PalletInPosition := 3708,
	PTZ_ZUnit_CrashDetection := 3709,
	Conveyors_ActTorque := 3710,
	PTZ_YUnit_ActTorque := 3711,
	PTZ_ZUnit_ActTorque := 3712,
	PTZ_Transfer_ActTorque := 3713,
	PTZ_PalletCenterUnit_1_ActTorque := 3714,
	PTZ_PalletCenterUnit_2_ActTorque := 3715,
	XuUnit_Vacuum_1_Output := 3716,
	XuUnit_Vacuum_2_Output := 3717,
	XuUnit_Vacuum_3_Output := 3718,
	XuUnit_Vacuum_4_Output := 3719,
	XuUnit_Vacuum_5_Output := 3720,
	XuUnit_Vacuum_6_Output := 3721,
	XuUnit_Vacuum_7_Output := 3722,
	XuUnit_Vacuum_8_Output := 3723,
	XiUnit_Vacuum_1_Output := 3724,
	XiUnit_Vacuum_2_Output := 3725,
	XiUnit_Vacuum_3_Output := 3726,
	XiUnit_Vacuum_4_Output := 3727,
	XiUnit_Vacuum_5_Output := 3728,
	XiUnit_Vacuum_6_Output := 3729,
	XiUnit_Vacuum_7_Output := 3730,
	XiUnit_Vacuum_8_Output := 3731,
	XiUnit_BufferAir_Output := 3732,
	XuUnit_BufferAir_Output := 3733,
	XiUnit_LockCore_Output := 3734,
	Conveyors_PusherIn_Output := 3735,
	Conveyors_PusherOut_Output := 3736,
	ZUnit_Vacuum_1_Output := 3737,
	ZUnit_Vacuum_2_Output := 3738,
	ZUnit_Vacuum_3_Output := 3739,
	ZUnit_Vacuum_4_Output := 3740,
	ZUnit_Vacuum_5_Output := 3741,
	ZUnit_Vacuum_6_Output := 3742,
	ZUnit_Vacuum_7_Output := 3743,
	ZUnit_Vacuum_8_Output := 3744,
	ZUnit_RotateIn_Output := 3745,
	ZUnit_RotateOut_Output := 3746,
	PTZ_PalletCenterUnit_1_ClampIn_Output := 3747,
	PTZ_PalletCenterUnit_1_ClampOut_Output := 3748,
	PTZ_PalletCenterUnit_2_ClampIn_Output := 3749,
	PTZ_PalletCenterUnit_2_ClampOut_Output := 3750,
	PTZ_Transfer_ExtendIn_Output := 3751,
	PTZ_Transfer_ExtendOut_Output := 3752,
	PTZ_Transfer_Vacuum_1_Output := 3753,
	PTZ_Transfer_Vacuum_2_Output := 3754,
	PTZ_ZUnit_ExtendSheetIn_Output := 3755,
	PTZ_ZUnit_ExtendSheetOut_Output := 3756,
	PTZ_ZUnit_ExtendSafetyCoverOut_Output := 3757,
	ZUnit_BufferAir_Output := 3758,
	PTZ_ZUnit_BufferAir_Output := 3759,
	PTZ_ZUnit_Vacuum_1_Output := 3760,
	PTZ_ZUnit_Vacuum_2_Output := 3761,
	PTZ_ZUnit_Vacuum_3_Output := 3762,
	PTZ_ZUnit_Vacuum_4_Output := 3763,
	PTZ_ZUnit_Vacuum_5_Output := 3764,
	PTZ_ZUnit_Vacuum_6_Output := 3765,
	PTZ_ZUnit_Vacuum_7_Output := 3766,
	PTZ_ZUnit_Vacuum_8_Output := 3767,
	PTZ_ZUnit_BufferAirSheet_Output := 3768,
	Magazine_Vacuum_1_Output := 3769,
	Magazine_Vacuum_2_Output := 3770,
	Magazine_Vacuum_3_Output := 3771,
	Magazine_Vacuum_4_Output := 3772,
	Magazine_Vacuum_5_Output := 3773,
	Magazine_Vacuum_6_Output := 3774,
	Magazine_VacuumAdditional_1_Output := 3775,
	Magazine_VacuumAdditional_2_Output := 3776,
	Magazine_VacuumAdditional_3_Output := 3777,
	Magazine_VacuumAdditional_4_Output := 3778,
	Magazine_BufferAir_Output := 3779,
	Magazine_RotateIn_Output := 3780,
	Magazine_RotateOut_Output := 3781,
	ZUnit_Extend_1_Output := 3782,
	ZUnit_Extend_2_Output := 3783,
	ZUnit_Extend_3_Output := 3784,
	ZUnit_Extend_4_Output := 3785,
	ZUnit_Extend_5_Output := 3786,
	ZUnit_Extend_6_Output := 3787,
	ZUnit_Extend_7_Output := 3788,
	ZUnit_Extend_8_Output := 3789,
	PTZ_Transfer_BufferAir_Output := 3790,
	PTZ_Transfer_Time_Idle := 3791,
	PTZ_ZUnit_Time_Idle := 3792,
	PTZ_YUnit_Time_Idle := 3793,
	PTZ_PalletCenterUnit_1_Time_Idle := 3794,
	PTZ_PalletCenterUnit_2_Time_Idle := 3795,
	PTZ_Transfer_Time_Active := 3796,
	PTZ_ZUnit_Time_Active := 3797,
	PTZ_YUnit_Time_Active := 3798,
	PTZ_PalletCenterUnit_1_Time_Active := 3799,
	PTZ_PalletCenterUnit_2_Time_Active := 3800,
	ZrUnit_Zr2_CoveredDistance := 3805,
	ZrUnit_Zr3_CoveredDistance := 3806,
	ZrUnit_Zr4_CoveredDistance := 3807,
	Conveyors_Conveyor1_Alarms := 3808,
	Conveyors_Conveyor2_Alarms := 3809,
	Conveyors_Conveyor3_Alarms := 3810,
	Conveyors_Conveyor4_Alarms := 3811,
	LabelAdjustment_Main_EnableMeasuringVision := 3812,
	IMM_I_Euromap_RejectMoulding := 3813,
	IMM_I_Euromap_MouldClosed := 3814,
	IMM_I_Euromap_MouldOpen := 3815,
	IMM_I_Euromap_IntermediateOpen := 3816,
	IMM_I_Euromap_AutoOperation := 3817,
	IMM_I_Euromap_EjectorBack := 3818,
	IMM_I_Euromap_EjectorForward := 3819,
	IMM_I_Euromap_CorePos1Back := 3820,
	IMM_I_Euromap_CorePos2Forward := 3821,
	IMM_I_Euromap_DoorClosed := 3822,
	ZUnit_SensorTimes_Vacuum_12 := 3831
) DINT;
END_TYPE
